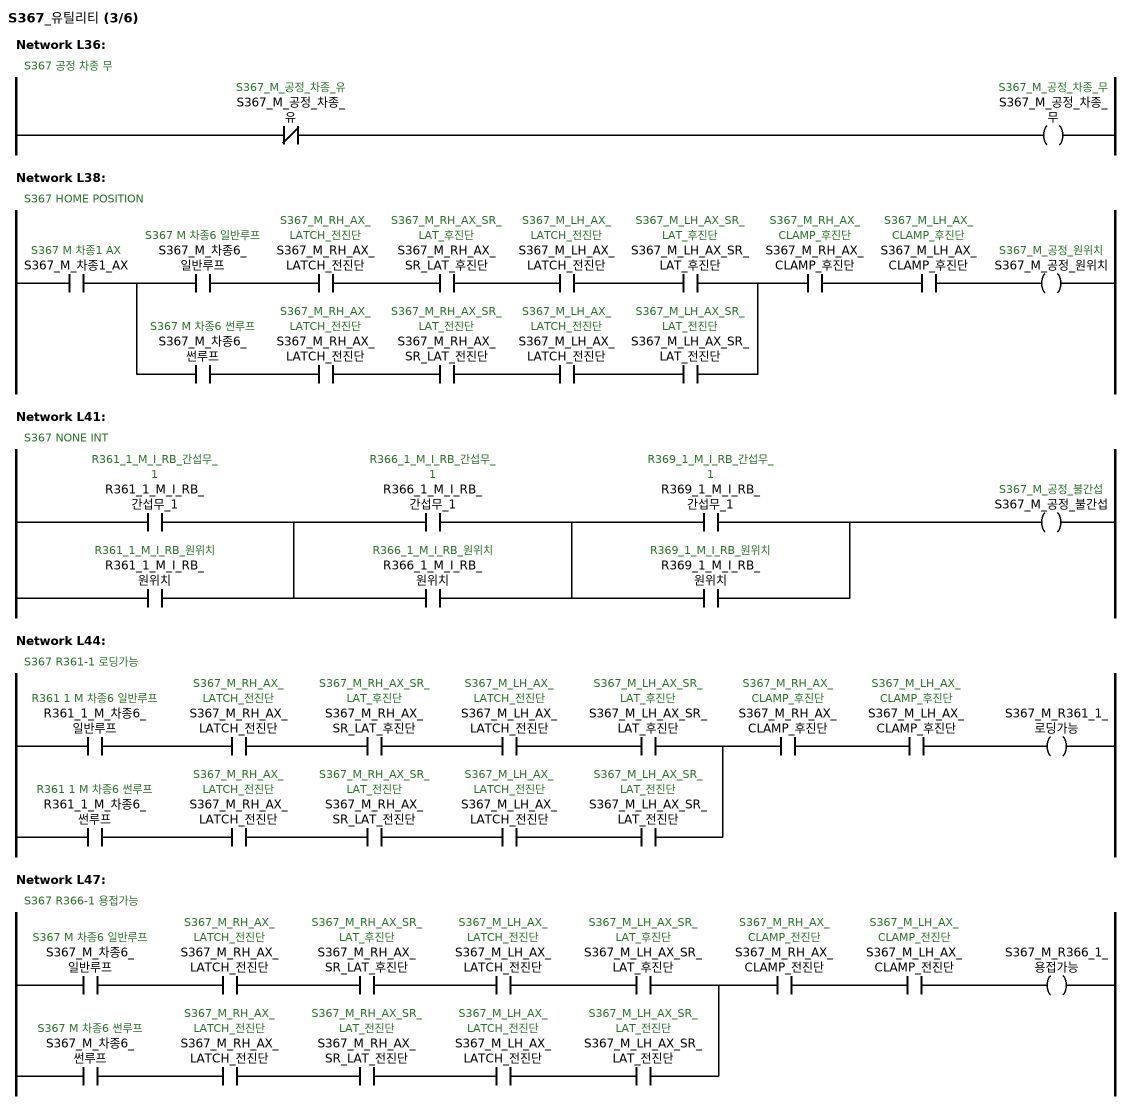
(* [picture p216: S367_유틸리티 rungs L36-L47] *)
(* S367 공정 차종 무 *)
(* Rung L36 *)
S367_M_공정_차종_무 := NOT S367_M_공정_차종_유;
(* S367 HOME POSITION *)
(* Rung L38 *)
S367_M_공정_원위치 := S367_M_차종1_AX AND ((S367_M_차종6_일반루프 AND S367_M_RH_AX_LATCH_전진단 AND S367_M_RH_AX_SR_LAT_후진단 AND S367_M_LH_AX_LATCH_전진단 AND S367_M_LH_AX_SR_LAT_후진단) OR (S367_M_차종6_썬루프 AND S367_M_RH_AX_LATCH_전진단 AND S367_M_RH_AX_SR_LAT_전진단 AND S367_M_LH_AX_LATCH_전진단 AND S367_M_LH_AX_SR_LAT_전진단)) AND S367_M_RH_AX_CLAMP_후진단 AND S367_M_LH_AX_CLAMP_후진단;
(* S367 NONE INT *)
(* Rung L41 *)
S367_M_공정_불간섭 := (R361_1_M_I_RB_간섭무_1 OR R361_1_M_I_RB_원위치) AND (R366_1_M_I_RB_간섭무_1 OR R366_1_M_I_RB_원위치) AND (R369_1_M_I_RB_간섭무_1 OR R369_1_M_I_RB_원위치);
(* S367 R361-1 로딩가능 *)
(* Rung L44 *)
S367_M_R361_1_로딩가능 := ((R361_1_M_차종6_일반루프 AND S367_M_RH_AX_LATCH_전진단 AND S367_M_RH_AX_SR_LAT_후진단 AND S367_M_LH_AX_LATCH_전진단 AND S367_M_LH_AX_SR_LAT_후진단) OR (R361_1_M_차종6_썬루프 AND S367_M_RH_AX_LATCH_전진단 AND S367_M_RH_AX_SR_LAT_전진단 AND S367_M_LH_AX_LATCH_전진단 AND S367_M_LH_AX_SR_LAT_전진단)) AND S367_M_RH_AX_CLAMP_후진단 AND S367_M_LH_AX_CLAMP_후진단;
(* S367 R366-1 용접가능 *)
(* Rung L47 *)
S367_M_R366_1_용접가능 := ((S367_M_차종6_일반루프 AND S367_M_RH_AX_LATCH_전진단 AND S367_M_RH_AX_SR_LAT_후진단 AND S367_M_LH_AX_LATCH_전진단 AND S367_M_LH_AX_SR_LAT_후진단) OR (S367_M_차종6_썬루프 AND S367_M_RH_AX_LATCH_전진단 AND S367_M_RH_AX_SR_LAT_전진단 AND S367_M_LH_AX_LATCH_전진단 AND S367_M_LH_AX_SR_LAT_전진단)) AND S367_M_RH_AX_CLAMP_전진단 AND S367_M_LH_AX_CLAMP_전진단;

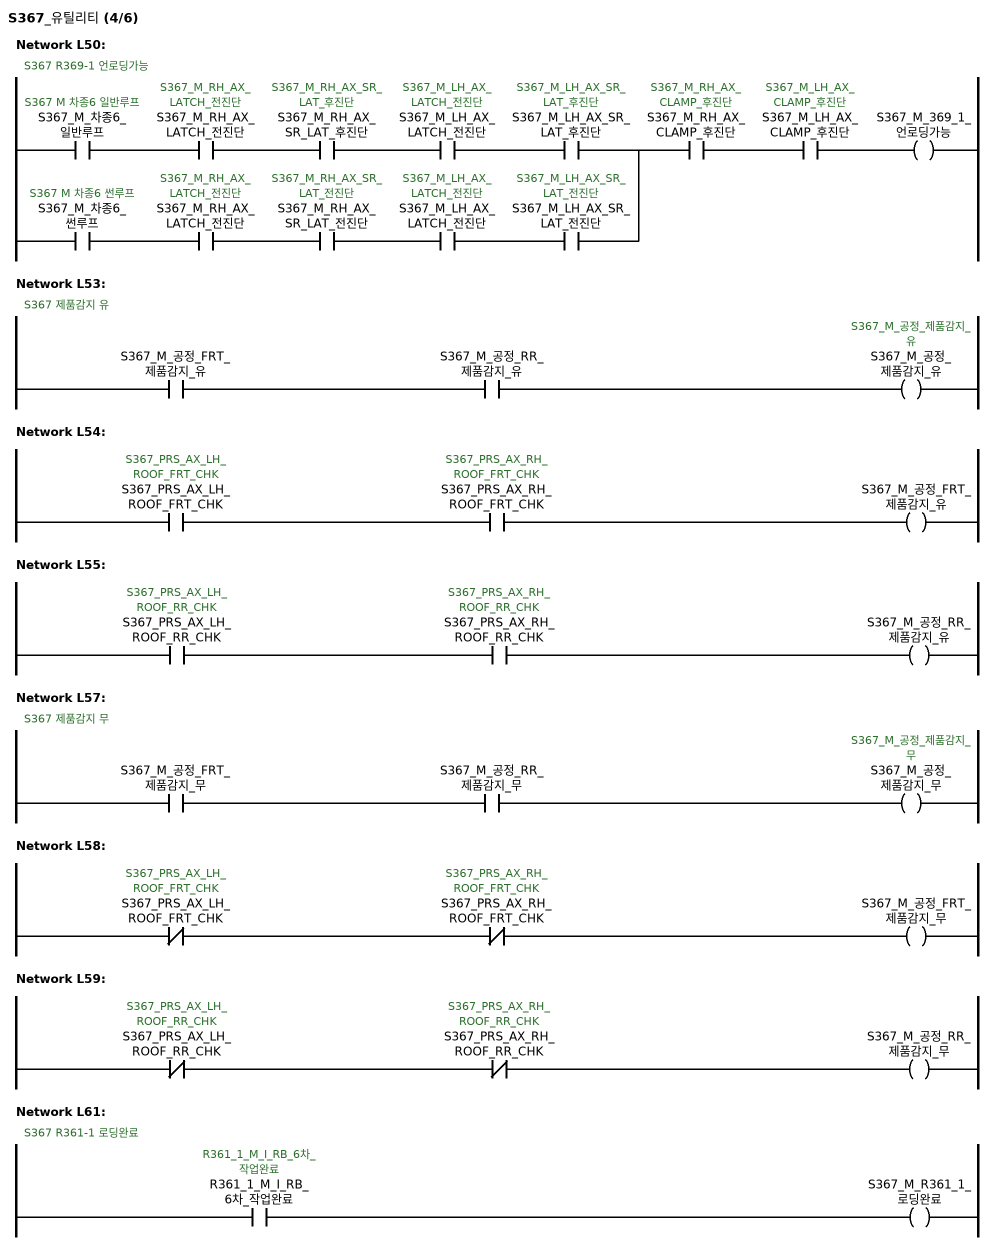
(* S367 R369-1 언로딩가능 *)
(* Rung L50 *)
S367_M_369_1_언로딩가능 := ((S367_M_차종6_일반루프 AND S367_M_RH_AX_LATCH_전진단 AND S367_M_RH_AX_SR_LAT_후진단 AND S367_M_LH_AX_LATCH_전진단 AND S367_M_LH_AX_SR_LAT_후진단) OR (S367_M_차종6_썬루프 AND S367_M_RH_AX_LATCH_전진단 AND S367_M_RH_AX_SR_LAT_전진단 AND S367_M_LH_AX_LATCH_전진단 AND S367_M_LH_AX_SR_LAT_전진단)) AND S367_M_RH_AX_CLAMP_후진단 AND S367_M_LH_AX_CLAMP_후진단;
(* S367 제품감지 유 *)
(* Rung L53 *)
S367_M_공정_제품감지_유 := S367_M_공정_FRT_제품감지_유 AND S367_M_공정_RR_제품감지_유;
(* Rung L54 *)
S367_M_공정_FRT_제품감지_유 := S367_PRS_AX_LH_ROOF_FRT_CHK AND S367_PRS_AX_RH_ROOF_FRT_CHK;
(* Rung L55 *)
S367_M_공정_RR_제품감지_유 := S367_PRS_AX_LH_ROOF_RR_CHK AND S367_PRS_AX_RH_ROOF_RR_CHK;
(* S367 제품감지 무 *)
(* Rung L57 *)
S367_M_공정_제품감지_무 := S367_M_공정_FRT_제품감지_무 AND S367_M_공정_RR_제품감지_무;
(* Rung L58 *)
S367_M_공정_FRT_제품감지_무 := NOT S367_PRS_AX_LH_ROOF_FRT_CHK AND NOT S367_PRS_AX_RH_ROOF_FRT_CHK;
(* Rung L59 *)
S367_M_공정_RR_제품감지_무 := NOT S367_PRS_AX_LH_ROOF_RR_CHK AND NOT S367_PRS_AX_RH_ROOF_RR_CHK;
(* S367 R361-1 로딩완료 *)
(* Rung L61 *)
S367_M_R361_1_로딩완료 := R361_1_M_I_RB_6차_작업완료;

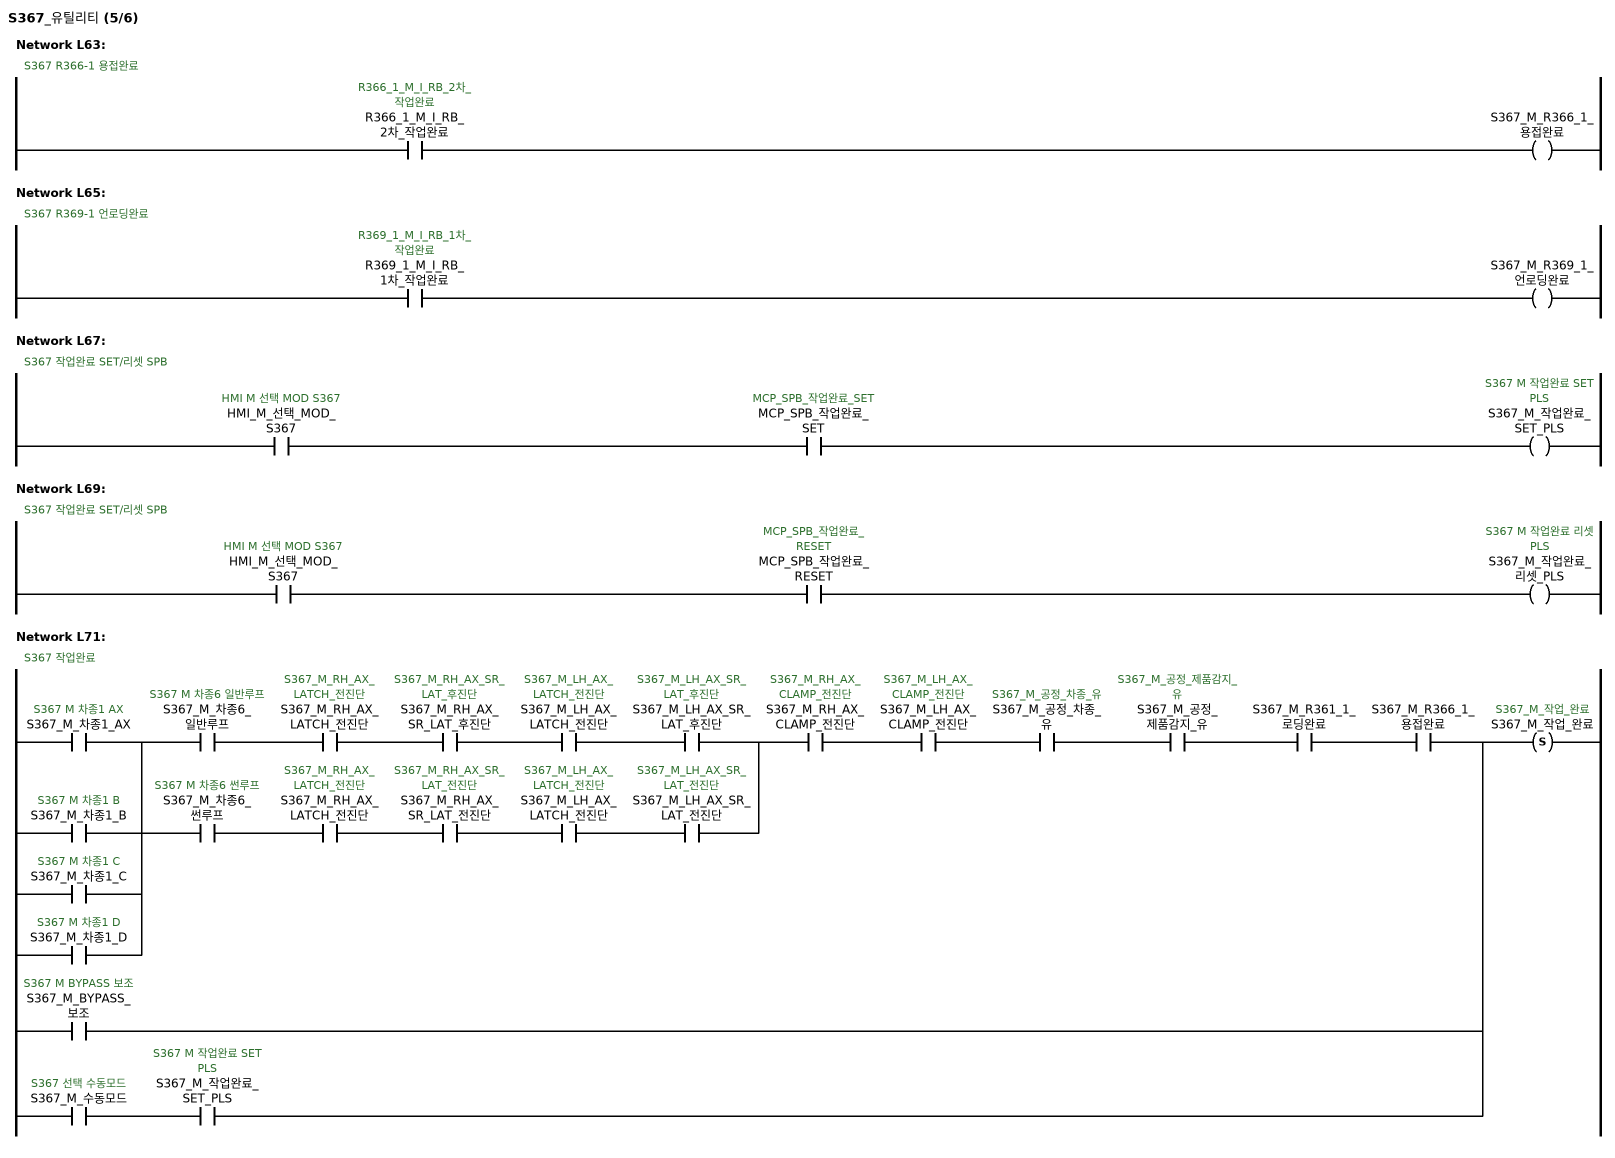
(* S367 R366-1 용접완료 *)
(* Rung L63 *)
S367_M_R366_1_용접완료 := R366_1_M_I_RB_2차_작업완료;
(* S367 R369-1 언로딩완료 *)
(* Rung L65 *)
S367_M_R369_1_언로딩완료 := R369_1_M_I_RB_1차_작업완료;
(* S367 작업완료 SET/리셋 SPB *)
(* Rung L67 *)
S367_M_작업완료_SET_PLS := HMI_M_선택_MOD_S367 AND MCP_SPB_작업완료_SET;
(* S367 작업완료 SET/리셋 SPB *)
(* Rung L69 *)
S367_M_작업완료_리셋_PLS := HMI_M_선택_MOD_S367 AND MCP_SPB_작업완료_RESET;
(* S367 작업완료 *)
(* Rung L71 *)
IF ((S367_M_차종1_AX OR S367_M_차종1_B OR S367_M_차종1_C OR S367_M_차종1_D) AND ((S367_M_차종6_일반루프 AND S367_M_RH_AX_LATCH_전진단 AND S367_M_RH_AX_SR_LAT_후진단 AND S367_M_LH_AX_LATCH_전진단 AND S367_M_LH_AX_SR_LAT_후진단) OR (S367_M_차종6_썬루프 AND S367_M_RH_AX_LATCH_전진단 AND S367_M_RH_AX_SR_LAT_전진단 AND S367_M_LH_AX_LATCH_전진단 AND S367_M_LH_AX_SR_LAT_전진단)) AND S367_M_RH_AX_CLAMP_전진단 AND S367_M_LH_AX_CLAMP_전진단 AND S367_M_공정_차종_유 AND S367_M_공정_제품감지_유 AND S367_M_R361_1_로딩완료 AND S367_M_R366_1_용접완료) OR S367_M_BYPASS_보조 OR (S367_M_수동모드 AND S367_M_작업완료_SET_PLS) THEN
    S367_M_작업_완료 := TRUE;
END_IF;

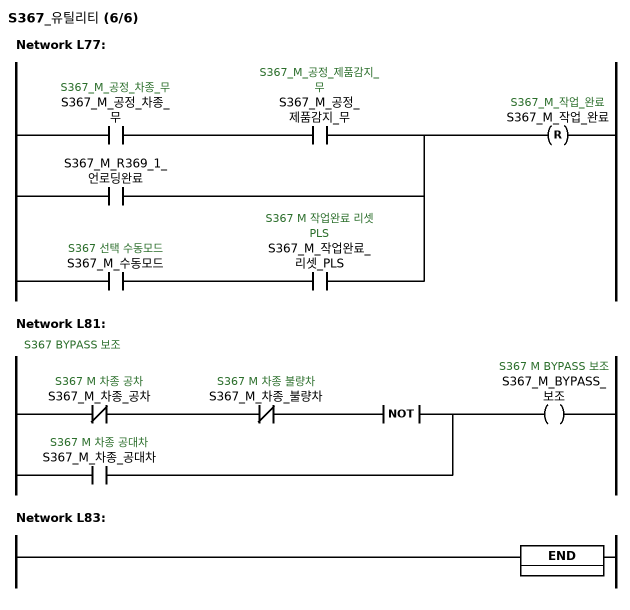
(* Rung L77 *)
IF (S367_M_공정_차종_무 AND S367_M_공정_제품감지_무) OR S367_M_R369_1_언로딩완료 OR (S367_M_수동모드 AND S367_M_작업완료_리셋_PLS) THEN
    S367_M_작업_완료 := FALSE;
END_IF;
(* S367 BYPASS 보조 *)
(* Rung L81 *)
S367_M_BYPASS_보조 := NOT (NOT S367_M_차종_공차 AND NOT S367_M_차종_불량차) OR S367_M_차종_공대차;
(* Rung L83 *)
END();
END_PROGRAM

PROGRAM S367_동작 (* task: 스캔 프로그램 *)
VAR_EXTERNAL RETAIN
    ALWAYS_ON : BOOL; (* AT %MW3.1 *) (* 항시 ON *)
    R361_1_M_차종1_AX : BOOL; (* AT %MW10001.0 *) (* R361 1 M 차종1 AX *)
    R361_1_M_차종6_썬루프 : BOOL; (* AT %MW10003.4 *) (* R361 1 M 차종6 썬루프 *)
    R361_1_M_차종_유 : BOOL; (* AT %MW1502.0 *)
    S367_HOME : BOOL; (* AT %MW3548.0 *) (* S367_HOME *)
    S367_M_LH_AX_CLAMP_전진_LS_이상 : BOOL; (* AT %MW3602.5 *) (* S367_M_LH_AX_CLAMP_전진_LS_이상 *)
    S367_M_LH_AX_CLAMP_전진_보조 : BOOL; (* AT %MW3602.1 *) (* S367_M_LH_AX_CLAMP_전진_보조 *)
    S367_M_LH_AX_CLAMP_전진단 : BOOL; (* AT %MW3602.3 *) (* S367_M_LH_AX_CLAMP_전진단 *)
    S367_M_LH_AX_CLAMP_조건 : BOOL; (* AT %MW3602.0 *) (* S367_M_LH_AX_CLAMP_조건 *)
    S367_M_LH_AX_CLAMP_후진_LS_이상 : BOOL; (* AT %MW3602.6 *) (* S367_M_LH_AX_CLAMP_후진_LS_이상 *)
    S367_M_LH_AX_CLAMP_후진_보조 : BOOL; (* AT %MW3602.2 *) (* S367_M_LH_AX_CLAMP_후진_보조 *)
    S367_M_LH_AX_CLAMP_후진단 : BOOL; (* AT %MW3602.4 *) (* S367_M_LH_AX_CLAMP_후진단 *)
    S367_M_LH_AX_LATCH_전진_LS_이상 : BOOL; (* AT %MW3600.5 *) (* S367_M_LH_AX_LATCH_전진_LS_이상 *)
    S367_M_LH_AX_LATCH_전진_보조 : BOOL; (* AT %MW3600.1 *) (* S367_M_LH_AX_LATCH_전진_보조 *)
    S367_M_LH_AX_LATCH_전진단 : BOOL; (* AT %MW3600.3 *) (* S367_M_LH_AX_LATCH_전진단 *)
    S367_M_LH_AX_LATCH_조건 : BOOL; (* AT %MW3600.0 *) (* S367_M_LH_AX_LATCH_조건 *)
    S367_M_LH_AX_LATCH_후진_LS_이상 : BOOL; (* AT %MW3600.6 *) (* S367_M_LH_AX_LATCH_후진_LS_이상 *)
    S367_M_LH_AX_LATCH_후진_보조 : BOOL; (* AT %MW3600.2 *) (* S367_M_LH_AX_LATCH_후진_보조 *)
    S367_M_LH_AX_LATCH_후진단 : BOOL; (* AT %MW3600.4 *) (* S367_M_LH_AX_LATCH_후진단 *)
    S367_M_LH_AX_SR_LAT_전진_LS_이상 : BOOL; (* AT %MW3601.5 *) (* S367_M_LH_AX_SR_LAT_전진_LS_이상 *)
    S367_M_LH_AX_SR_LAT_전진_보조 : BOOL; (* AT %MW3601.1 *) (* S367_M_LH_AX_SR_LAT_전진_보조 *)
    S367_M_LH_AX_SR_LAT_전진단 : BOOL; (* AT %MW3601.3 *) (* S367_M_LH_AX_SR_LAT_전진단 *)
    S367_M_LH_AX_SR_LAT_조건 : BOOL; (* AT %MW3601.0 *) (* S367_M_LH_AX_SR_LAT_조건 *)
    S367_M_LH_AX_SR_LAT_후진_LS_이상 : BOOL; (* AT %MW3601.6 *) (* S367_M_LH_AX_SR_LAT_후진_LS_이상 *)
    S367_M_LH_AX_SR_LAT_후진_보조 : BOOL; (* AT %MW3601.2 *) (* S367_M_LH_AX_SR_LAT_후진_보조 *)
    S367_M_LH_AX_SR_LAT_후진단 : BOOL; (* AT %MW3601.4 *) (* S367_M_LH_AX_SR_LAT_후진단 *)
    S367_M_R361_1_로딩완료 : BOOL; (* AT %MW3501.1 *)
    S367_M_RH_AX_CLAMP_전진_LS_이상 : BOOL; (* AT %MW3610.5 *) (* S367_M_RH_AX_CLAMP_전진_LS_이상 *)
    S367_M_RH_AX_CLAMP_전진_보조 : BOOL; (* AT %MW3610.1 *) (* S367_M_RH_AX_CLAMP_전진_보조 *)
    S367_M_RH_AX_CLAMP_전진단 : BOOL; (* AT %MW3610.3 *) (* S367_M_RH_AX_CLAMP_전진단 *)
    S367_M_RH_AX_CLAMP_조건 : BOOL; (* AT %MW3610.0 *) (* S367_M_RH_AX_CLAMP_조건 *)
    S367_M_RH_AX_CLAMP_후진_LS_이상 : BOOL; (* AT %MW3610.6 *) (* S367_M_RH_AX_CLAMP_후진_LS_이상 *)
    S367_M_RH_AX_CLAMP_후진_보조 : BOOL; (* AT %MW3610.2 *) (* S367_M_RH_AX_CLAMP_후진_보조 *)
    S367_M_RH_AX_CLAMP_후진단 : BOOL; (* AT %MW3610.4 *) (* S367_M_RH_AX_CLAMP_후진단 *)
    S367_M_RH_AX_LATCH_전진_LS_이상 : BOOL; (* AT %MW3608.5 *) (* S367_M_RH_AX_LATCH_전진_LS_이상 *)
    S367_M_RH_AX_LATCH_전진_보조 : BOOL; (* AT %MW3608.1 *) (* S367_M_RH_AX_LATCH_전진_보조 *)
    S367_M_RH_AX_LATCH_전진단 : BOOL; (* AT %MW3608.3 *) (* S367_M_RH_AX_LATCH_전진단 *)
    S367_M_RH_AX_LATCH_조건 : BOOL; (* AT %MW3608.0 *) (* S367_M_RH_AX_LATCH_조건 *)
    S367_M_RH_AX_LATCH_후진_LS_이상 : BOOL; (* AT %MW3608.6 *) (* S367_M_RH_AX_LATCH_후진_LS_이상 *)
    S367_M_RH_AX_LATCH_후진_보조 : BOOL; (* AT %MW3608.2 *) (* S367_M_RH_AX_LATCH_후진_보조 *)
    S367_M_RH_AX_LATCH_후진단 : BOOL; (* AT %MW3608.4 *) (* S367_M_RH_AX_LATCH_후진단 *)
    S367_M_RH_AX_SR_LAT_전진_LS_이상 : BOOL; (* AT %MW3609.5 *) (* S367_M_RH_AX_SR_LAT_전진_LS_이상 *)
    S367_M_RH_AX_SR_LAT_전진_보조 : BOOL; (* AT %MW3609.1 *) (* S367_M_RH_AX_SR_LAT_전진_보조 *)
    S367_M_RH_AX_SR_LAT_전진단 : BOOL; (* AT %MW3609.3 *) (* S367_M_RH_AX_SR_LAT_전진단 *)
    S367_M_RH_AX_SR_LAT_조건 : BOOL; (* AT %MW3609.0 *) (* S367_M_RH_AX_SR_LAT_조건 *)
    S367_M_RH_AX_SR_LAT_후진_LS_이상 : BOOL; (* AT %MW3609.6 *) (* S367_M_RH_AX_SR_LAT_후진_LS_이상 *)
    S367_M_RH_AX_SR_LAT_후진_보조 : BOOL; (* AT %MW3609.2 *) (* S367_M_RH_AX_SR_LAT_후진_보조 *)
    S367_M_RH_AX_SR_LAT_후진단 : BOOL; (* AT %MW3609.4 *) (* S367_M_RH_AX_SR_LAT_후진단 *)
    S367_M_공정_불간섭 : BOOL; (* AT %MW3504.1 *) (* S367_M_공정_불간섭 *)
    S367_M_공정_제품감지_무 : BOOL; (* AT %MW3501.6 *) (* S367_M_공정_제품감지_무 *)
    S367_M_공정_제품감지_유 : BOOL; (* AT %MW3501.5 *) (* S367_M_공정_제품감지_유 *)
    S367_M_공정_차종_무 : BOOL; (* AT %MW3502.1 *) (* S367_M_공정_차종_무 *)
    S367_M_공정_차종_유 : BOOL; (* AT %MW3502.0 *) (* S367_M_공정_차종_유 *)
    S367_M_동작_선택_1 : BOOL; (* AT %MW3540.0 *) (* S367_M_동작_선택_1 *)
    S367_M_동작_선택_10 : BOOL; (* AT %MW3540.9 *) (* S367_M_동작_선택_10 *)
    S367_M_동작_선택_11 : BOOL; (* AT %MW3540.10 *) (* S367_M_동작_선택_11 *)
    S367_M_동작_선택_2 : BOOL; (* AT %MW3540.1 *) (* S367_M_동작_선택_2 *)
    S367_M_동작_선택_3 : BOOL; (* AT %MW3540.2 *) (* S367_M_동작_선택_3 *)
    S367_M_동작_선택_9 : BOOL; (* AT %MW3540.8 *) (* S367_M_동작_선택_9 *)
    S367_M_수동모드 : BOOL; (* AT %MW3500.3 *) (* S367 선택 수동모드 *)
    S367_M_운전준비_ON : BOOL; (* AT %MW3500.0 *) (* S367 운전준비 ON *)
    S367_M_자동_운전중 : BOOL; (* AT %MW3500.4 *) (* S367 자동운전중 *)
    S367_M_작업_완료 : BOOL; (* AT %MW3501.0 *) (* S367_M_작업_완료 *)
    S367_M_차종1_AX : BOOL; (* AT %MW10181.0 *) (* S367 M 차종1 AX *)
    S367_전진_ON : BOOL; (* AT %MW3548.1 *) (* S367_전진_ON *)
    S367_후진_ON : BOOL; (* AT %MW3548.2 *) (* S367_후진_ON *)
    전체_M_이상_리셋 : BOOL; (* AT %MW308.2 *) (* ALL공정 PB 이상리셋 *)
END_VAR
VAR_EXTERNAL
    EGIS_CWS : BOOL;
    S367_M_LH_AX_CLAMP_전진_LAMP : WORD; (* AT %MW13104 *) (* S367_M_LH_AX_CLAMP_전진_LAMP *)
    S367_M_LH_AX_CLAMP_후진_LAMP : WORD; (* AT %MW13105 *) (* S367_M_LH_AX_CLAMP_후진_LAMP *)
    S367_M_LH_AX_LATCH_전진_LAMP : WORD; (* AT %MW13100 *) (* S367_M_LH_AX_LATCH_전진_LAMP *)
    S367_M_LH_AX_LATCH_후진_LAMP : WORD; (* AT %MW13101 *) (* S367_M_LH_AX_LATCH_후진_LAMP *)
    S367_M_LH_AX_SR_LAT_전진_LAMP : WORD; (* AT %MW13102 *) (* S367_M_LH_AX_SR_LAT_전진_LAMP *)
    S367_M_LH_AX_SR_LAT_후진_LAMP : WORD; (* AT %MW13103 *) (* S367_M_LH_AX_SR_LAT_후진_LAMP *)
    S367_M_RH_AX_CLAMP_전진_LAMP : WORD; (* AT %MW13120 *) (* S367_M_RH_AX_CLAMP_전진_LAMP *)
    S367_M_RH_AX_CLAMP_후진_LAMP : WORD; (* AT %MW13121 *) (* S367_M_RH_AX_CLAMP_후진_LAMP *)
    S367_M_RH_AX_LATCH_전진_LAMP : WORD; (* AT %MW13116 *) (* S367_M_RH_AX_LATCH_전진_LAMP *)
    S367_M_RH_AX_LATCH_후진_LAMP : WORD; (* AT %MW13117 *) (* S367_M_RH_AX_LATCH_후진_LAMP *)
    S367_M_RH_AX_SR_LAT_전진_LAMP : WORD; (* AT %MW13118 *) (* S367_M_RH_AX_SR_LAT_전진_LAMP *)
    S367_M_RH_AX_SR_LAT_후진_LAMP : WORD; (* AT %MW13119 *) (* S367_M_RH_AX_SR_LAT_후진_LAMP *)
    S367_RS_AX_LH_CLAMP_전진 : BOOL; (* AT %MW86210.8 *) (* S367_RS_AX_LH_CLAMP_전진 *)
    S367_RS_AX_LH_CLAMP_후진1 : BOOL; (* AT %MW86210.9 *) (* S367_RS_AX_LH_CLAMP_후진1 *)
    S367_RS_AX_LH_CLAMP_후진2 : BOOL; (* AT %MW86210.10 *) (* S367_RS_AX_LH_CLAMP_후진2 *)
    S367_RS_AX_LH_CLAMP_후진3 : BOOL; (* AT %MW86210.11 *) (* S367_RS_AX_LH_CLAMP_후진3 *)
    S367_RS_AX_LH_CLAMP_후진4 : BOOL; (* AT %MW86210.12 *) (* S367_RS_AX_LH_CLAMP_후진4 *)
    S367_RS_AX_LH_CLAMP_후진5 : BOOL; (* AT %MW86210.13 *) (* S367_RS_AX_LH_CLAMP_후진5 *)
    S367_RS_AX_LH_GR_LATCH_전진 : BOOL; (* AT %MW86210.0 *) (* S367_RS_AX_LH_GR_LATCH_전진 *)
    S367_RS_AX_LH_GR_LATCH_후진1 : BOOL; (* AT %MW86210.1 *) (* S367_RS_AX_LH_GR_LATCH_후진1 *)
    S367_RS_AX_LH_GR_LATCH_후진2 : BOOL; (* AT %MW86210.2 *) (* S367_RS_AX_LH_GR_LATCH_후진2 *)
    S367_RS_AX_LH_GR_LATCH_후진3 : BOOL; (* AT %MW86210.3 *) (* S367_RS_AX_LH_GR_LATCH_후진3 *)
    S367_RS_AX_LH_GR_LATCH_후진4 : BOOL; (* AT %MW86210.4 *) (* S367_RS_AX_LH_GR_LATCH_후진4 *)
    S367_RS_AX_LH_GR_LATCH_후진5 : BOOL; (* AT %MW86210.5 *) (* S367_RS_AX_LH_GR_LATCH_후진5 *)
    S367_RS_AX_LH_SR_LATCH_전진 : BOOL; (* AT %MW86211.0 *) (* S367_RS_AX_LH_SR_LATCH_전진 *)
    S367_RS_AX_LH_SR_LATCH_후진1 : BOOL; (* AT %MW86211.1 *) (* S367_RS_AX_LH_SR_LATCH_후진1 *)
    S367_RS_AX_LH_SR_LATCH_후진2 : BOOL; (* AT %MW86211.2 *) (* S367_RS_AX_LH_SR_LATCH_후진2 *)
    S367_RS_AX_LH_SR_LATCH_후진3 : BOOL; (* AT %MW86211.3 *) (* S367_RS_AX_LH_SR_LATCH_후진3 *)
    S367_RS_AX_RH_CLAMP_전진 : BOOL; (* AT %MW86200.8 *) (* S367_RS_AX_RH_CLAMP_전진 *)
    S367_RS_AX_RH_CLAMP_후진1 : BOOL; (* AT %MW86200.9 *) (* S367_RS_AX_RH_CLAMP_후진1 *)
    S367_RS_AX_RH_CLAMP_후진2 : BOOL; (* AT %MW86200.10 *) (* S367_RS_AX_RH_CLAMP_후진2 *)
    S367_RS_AX_RH_CLAMP_후진3 : BOOL; (* AT %MW86200.11 *) (* S367_RS_AX_RH_CLAMP_후진3 *)
    S367_RS_AX_RH_CLAMP_후진4 : BOOL; (* AT %MW86200.12 *) (* S367_RS_AX_RH_CLAMP_후진4 *)
    S367_RS_AX_RH_CLAMP_후진5 : BOOL; (* AT %MW86200.13 *) (* S367_RS_AX_RH_CLAMP_후진5 *)
    S367_RS_AX_RH_GR_LATCH_전진 : BOOL; (* AT %MW86200.0 *) (* S367_RS_AX_RH_GR_LATCH_전진 *)
    S367_RS_AX_RH_GR_LATCH_후진1 : BOOL; (* AT %MW86200.1 *) (* S367_RS_AX_RH_GR_LATCH_후진1 *)
    S367_RS_AX_RH_GR_LATCH_후진2 : BOOL; (* AT %MW86200.2 *) (* S367_RS_AX_RH_GR_LATCH_후진2 *)
    S367_RS_AX_RH_GR_LATCH_후진3 : BOOL; (* AT %MW86200.3 *) (* S367_RS_AX_RH_GR_LATCH_후진3 *)
    S367_RS_AX_RH_GR_LATCH_후진4 : BOOL; (* AT %MW86200.4 *) (* S367_RS_AX_RH_GR_LATCH_후진4 *)
    S367_RS_AX_RH_GR_LATCH_후진5 : BOOL; (* AT %MW86200.5 *) (* S367_RS_AX_RH_GR_LATCH_후진5 *)
    S367_RS_AX_RH_SR_LATCH_전진 : BOOL; (* AT %MW86201.0 *) (* S367_RS_AX_RH_SR_LATCH_전진 *)
    S367_RS_AX_RH_SR_LATCH_후진1 : BOOL; (* AT %MW86201.1 *) (* S367_RS_AX_RH_SR_LATCH_후진1 *)
    S367_RS_AX_RH_SR_LATCH_후진2 : BOOL; (* AT %MW86201.2 *) (* S367_RS_AX_RH_SR_LATCH_후진2 *)
    S367_RS_AX_RH_SR_LATCH_후진3 : BOOL; (* AT %MW86201.3 *) (* S367_RS_AX_RH_SR_LATCH_후진3 *)
    S367_SOL_AX_LH_CLAMP_전진 : BOOL; (* AT %MW96213.6 *) (* S367_SOL_AX_LH_CLAMP_전진 *)
    S367_SOL_AX_LH_CLAMP_후진 : BOOL; (* AT %MW96213.7 *) (* S367_SOL_AX_LH_CLAMP_후진 *)
    S367_SOL_AX_LH_GR_LATCH_전진 : BOOL; (* AT %MW96213.2 *) (* S367_SOL_AX_LH_GR_LATCH_전진 *)
    S367_SOL_AX_LH_GR_LATCH_후진 : BOOL; (* AT %MW96213.3 *) (* S367_SOL_AX_LH_GR_LATCH_후진 *)
    S367_SOL_AX_LH_SR_LATCH_전진 : BOOL; (* AT %MW96213.10 *) (* S367_SOL_AX_LH_SR_LATCH_전진 *)
    S367_SOL_AX_LH_SR_LATCH_후진 : BOOL; (* AT %MW96213.11 *) (* S367_SOL_AX_LH_SR_LATCH_후진 *)
    S367_SOL_AX_RH_CLAMP_전진 : BOOL; (* AT %MW96213.4 *) (* S367_SOL_AX_RH_CLAMP_전진 *)
    S367_SOL_AX_RH_CLAMP_후진 : BOOL; (* AT %MW96213.5 *) (* S367_SOL_AX_RH_CLAMP_후진 *)
    S367_SOL_AX_RH_GR_LATCH_전진 : BOOL; (* AT %MW96213.0 *) (* S367_SOL_AX_RH_GR_LATCH_전진 *)
    S367_SOL_AX_RH_GR_LATCH_후진 : BOOL; (* AT %MW96213.1 *) (* S367_SOL_AX_RH_GR_LATCH_후진 *)
    S367_SOL_AX_RH_SR_LATCH_전진 : BOOL; (* AT %MW96213.8 *) (* S367_SOL_AX_RH_SR_LATCH_전진 *)
    S367_SOL_AX_RH_SR_LATCH_후진 : BOOL; (* AT %MW96213.9 *) (* S367_SOL_AX_RH_SR_LATCH_후진 *)
END_VAR
VAR
    S367_LH_AX_CLAMP : ACT_6_CYL;
    S367_LH_AX_LATCH : ACT_6_CYL;
    S367_LH_AX_SR_LAT : ACT_6_CYL;
    S367_RH_AX_CLAMP : ACT_6_CYL;
    S367_RH_AX_LATCH : ACT_6_CYL;
    S368_RH_AX_SR_LAT : ACT_6_CYL;
END_VAR

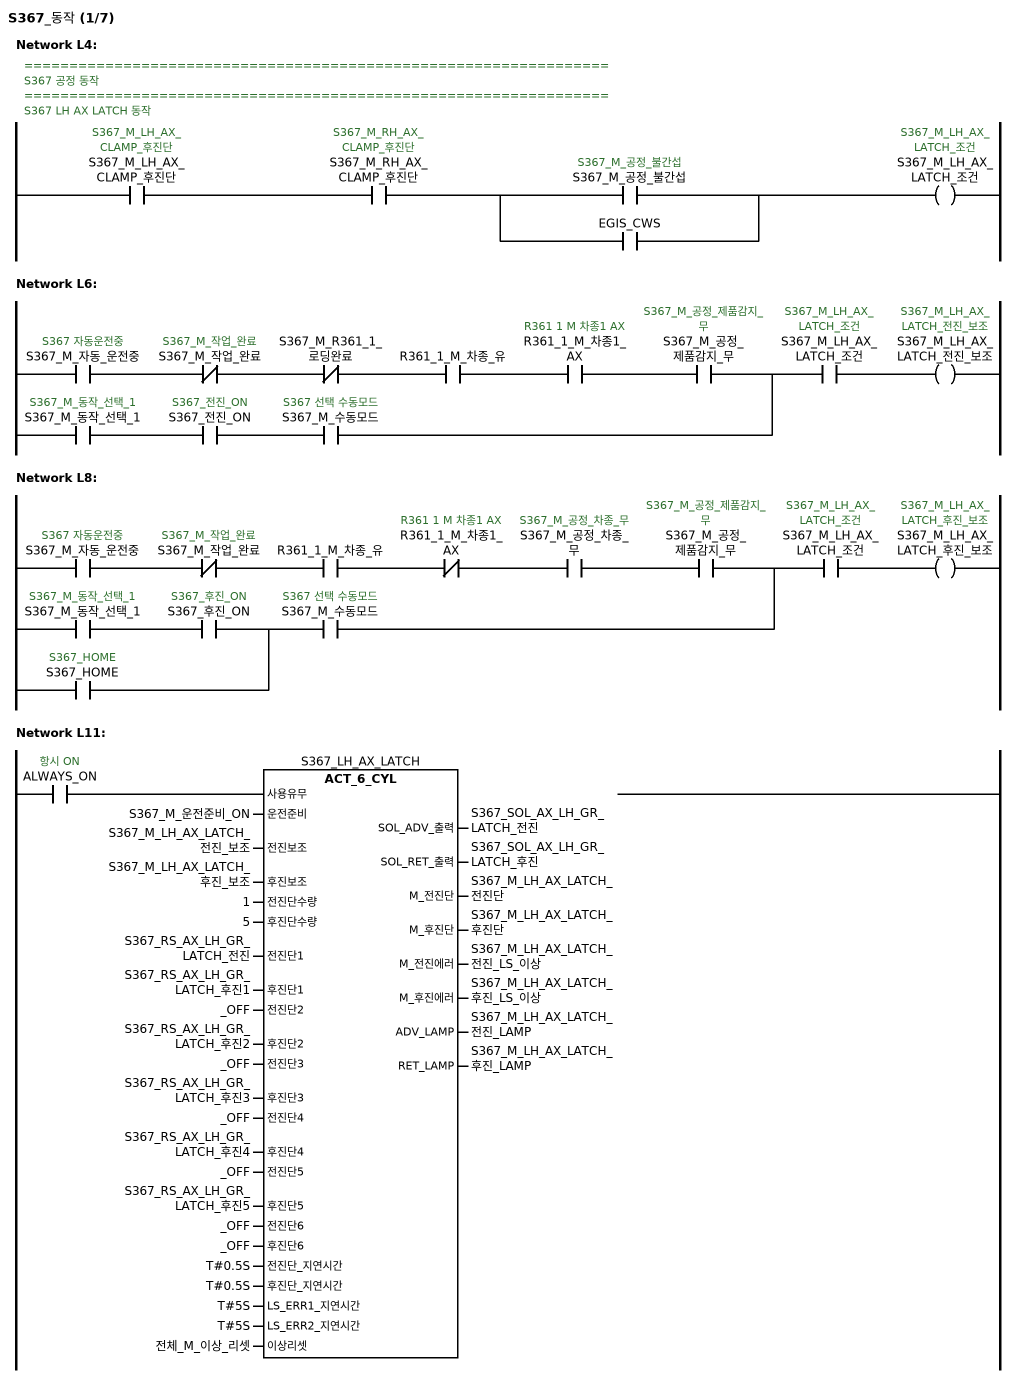
(* ================================================================= *)
(* S367 공정 동작 *)
(* ================================================================= *)
(* S367 LH AX LATCH 동작 *)
(* Rung L4 *)
S367_M_LH_AX_LATCH_조건 := S367_M_LH_AX_CLAMP_후진단 AND S367_M_RH_AX_CLAMP_후진단 AND (S367_M_공정_불간섭 OR EGIS_CWS);
(* Rung L6 *)
S367_M_LH_AX_LATCH_전진_보조 := ((S367_M_자동_운전중 AND NOT S367_M_작업_완료 AND NOT S367_M_R361_1_로딩완료 AND R361_1_M_차종_유 AND R361_1_M_차종1_AX AND S367_M_공정_제품감지_무) OR (S367_M_동작_선택_1 AND S367_전진_ON AND S367_M_수동모드)) AND S367_M_LH_AX_LATCH_조건;
(* Rung L8 *)
S367_M_LH_AX_LATCH_후진_보조 := ((S367_M_자동_운전중 AND NOT S367_M_작업_완료 AND R361_1_M_차종_유 AND NOT R361_1_M_차종1_AX AND S367_M_공정_차종_무 AND S367_M_공정_제품감지_무) OR (((S367_M_동작_선택_1 AND S367_후진_ON) OR S367_HOME) AND S367_M_수동모드)) AND S367_M_LH_AX_LATCH_조건;
(* Rung L11 *)
S367_LH_AX_LATCH(사용유무 := ALWAYS_ON, 운전준비 := S367_M_운전준비_ON, 전진보조 := S367_M_LH_AX_LATCH_전진_보조, 후진보조 := S367_M_LH_AX_LATCH_후진_보조, 전진단수량 := 1, 후진단수량 := 5, 전진단1 := S367_RS_AX_LH_GR_LATCH_전진, 후진단1 := S367_RS_AX_LH_GR_LATCH_후진1, 전진단2 := _OFF, 후진단2 := S367_RS_AX_LH_GR_LATCH_후진2, 전진단3 := _OFF, 후진단3 := S367_RS_AX_LH_GR_LATCH_후진3, 전진단4 := _OFF, 후진단4 := S367_RS_AX_LH_GR_LATCH_후진4, 전진단5 := _OFF, 후진단5 := S367_RS_AX_LH_GR_LATCH_후진5, 전진단6 := _OFF, 후진단6 := _OFF, 전진단_지연시간 := T#0.5S, 후진단_지연시간 := T#0.5S, LS_ERR1_지연시간 := T#5S, LS_ERR2_지연시간 := T#5S, 이상리셋 := 전체_M_이상_리셋, SOL_ADV_출력 => S367_SOL_AX_LH_GR_LATCH_전진, SOL_RET_출력 => S367_SOL_AX_LH_GR_LATCH_후진, M_전진단 => S367_M_LH_AX_LATCH_전진단, M_후진단 => S367_M_LH_AX_LATCH_후진단, M_전진에러 => S367_M_LH_AX_LATCH_전진_LS_이상, M_후진에러 => S367_M_LH_AX_LATCH_후진_LS_이상, ADV_LAMP => S367_M_LH_AX_LATCH_전진_LAMP, RET_LAMP => S367_M_LH_AX_LATCH_후진_LAMP);

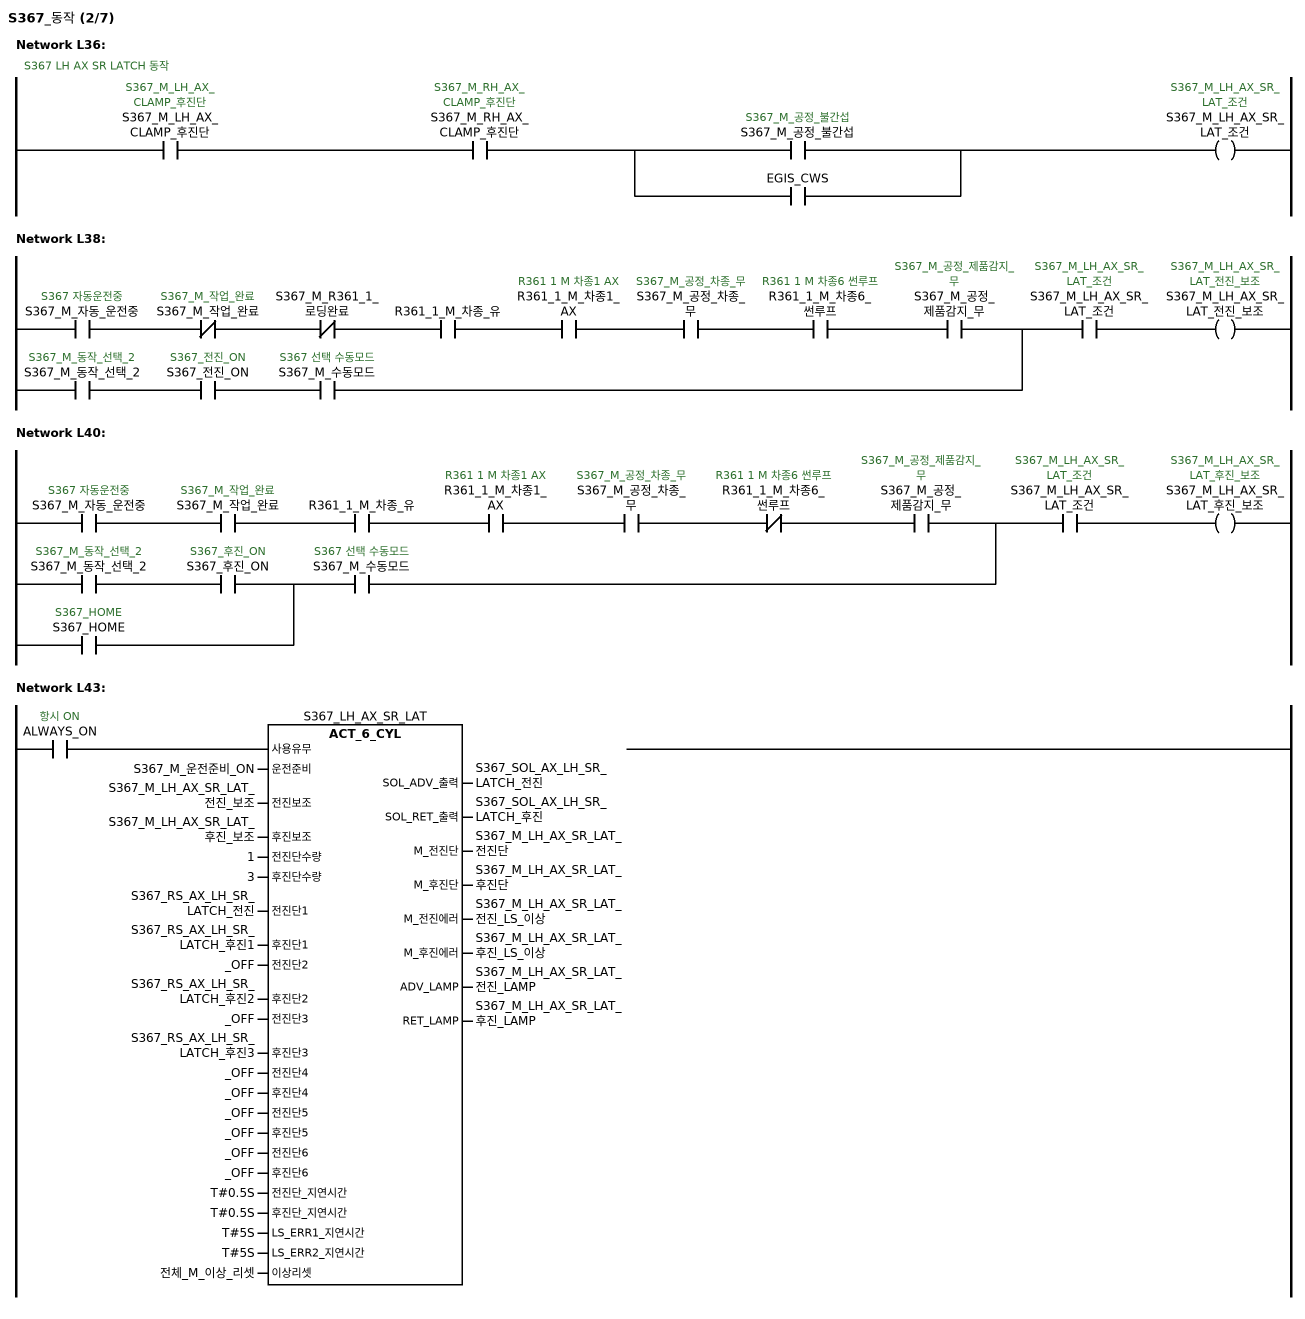
(* S367 LH AX SR LATCH 동작 *)
(* Rung L36 *)
S367_M_LH_AX_SR_LAT_조건 := S367_M_LH_AX_CLAMP_후진단 AND S367_M_RH_AX_CLAMP_후진단 AND (S367_M_공정_불간섭 OR EGIS_CWS);
(* Rung L38 *)
S367_M_LH_AX_SR_LAT_전진_보조 := ((S367_M_자동_운전중 AND NOT S367_M_작업_완료 AND NOT S367_M_R361_1_로딩완료 AND R361_1_M_차종_유 AND R361_1_M_차종1_AX AND S367_M_공정_차종_무 AND R361_1_M_차종6_썬루프 AND S367_M_공정_제품감지_무) OR (S367_M_동작_선택_2 AND S367_전진_ON AND S367_M_수동모드)) AND S367_M_LH_AX_SR_LAT_조건;
(* Rung L40 *)
S367_M_LH_AX_SR_LAT_후진_보조 := ((S367_M_자동_운전중 AND S367_M_작업_완료 AND R361_1_M_차종_유 AND R361_1_M_차종1_AX AND S367_M_공정_차종_무 AND NOT R361_1_M_차종6_썬루프 AND S367_M_공정_제품감지_무) OR (((S367_M_동작_선택_2 AND S367_후진_ON) OR S367_HOME) AND S367_M_수동모드)) AND S367_M_LH_AX_SR_LAT_조건;
(* Rung L43 *)
S367_LH_AX_SR_LAT(사용유무 := ALWAYS_ON, 운전준비 := S367_M_운전준비_ON, 전진보조 := S367_M_LH_AX_SR_LAT_전진_보조, 후진보조 := S367_M_LH_AX_SR_LAT_후진_보조, 전진단수량 := 1, 후진단수량 := 3, 전진단1 := S367_RS_AX_LH_SR_LATCH_전진, 후진단1 := S367_RS_AX_LH_SR_LATCH_후진1, 전진단2 := _OFF, 후진단2 := S367_RS_AX_LH_SR_LATCH_후진2, 전진단3 := _OFF, 후진단3 := S367_RS_AX_LH_SR_LATCH_후진3, 전진단4 := _OFF, 후진단4 := _OFF, 전진단5 := _OFF, 후진단5 := _OFF, 전진단6 := _OFF, 후진단6 := _OFF, 전진단_지연시간 := T#0.5S, 후진단_지연시간 := T#0.5S, LS_ERR1_지연시간 := T#5S, LS_ERR2_지연시간 := T#5S, 이상리셋 := 전체_M_이상_리셋, SOL_ADV_출력 => S367_SOL_AX_LH_SR_LATCH_전진, SOL_RET_출력 => S367_SOL_AX_LH_SR_LATCH_후진, M_전진단 => S367_M_LH_AX_SR_LAT_전진단, M_후진단 => S367_M_LH_AX_SR_LAT_후진단, M_전진에러 => S367_M_LH_AX_SR_LAT_전진_LS_이상, M_후진에러 => S367_M_LH_AX_SR_LAT_후진_LS_이상, ADV_LAMP => S367_M_LH_AX_SR_LAT_전진_LAMP, RET_LAMP => S367_M_LH_AX_SR_LAT_후진_LAMP);

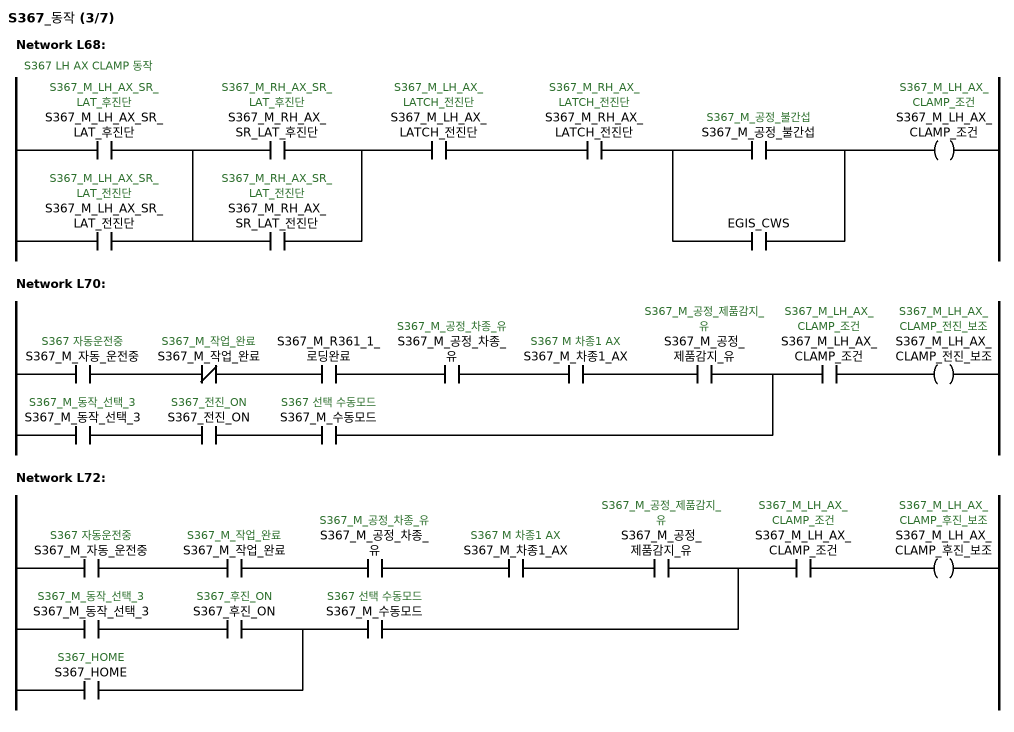
(* S367 LH AX CLAMP 동작 *)
(* Rung L68 *)
S367_M_LH_AX_CLAMP_조건 := (S367_M_LH_AX_SR_LAT_후진단 OR S367_M_LH_AX_SR_LAT_전진단) AND (S367_M_RH_AX_SR_LAT_후진단 OR S367_M_RH_AX_SR_LAT_전진단) AND S367_M_LH_AX_LATCH_전진단 AND S367_M_RH_AX_LATCH_전진단 AND (S367_M_공정_불간섭 OR EGIS_CWS);
(* Rung L70 *)
S367_M_LH_AX_CLAMP_전진_보조 := ((S367_M_자동_운전중 AND NOT S367_M_작업_완료 AND S367_M_R361_1_로딩완료 AND S367_M_공정_차종_유 AND S367_M_차종1_AX AND S367_M_공정_제품감지_유) OR (S367_M_동작_선택_3 AND S367_전진_ON AND S367_M_수동모드)) AND S367_M_LH_AX_CLAMP_조건;
(* Rung L72 *)
S367_M_LH_AX_CLAMP_후진_보조 := ((S367_M_자동_운전중 AND S367_M_작업_완료 AND S367_M_공정_차종_유 AND S367_M_차종1_AX AND S367_M_공정_제품감지_유) OR (((S367_M_동작_선택_3 AND S367_후진_ON) OR S367_HOME) AND S367_M_수동모드)) AND S367_M_LH_AX_CLAMP_조건;

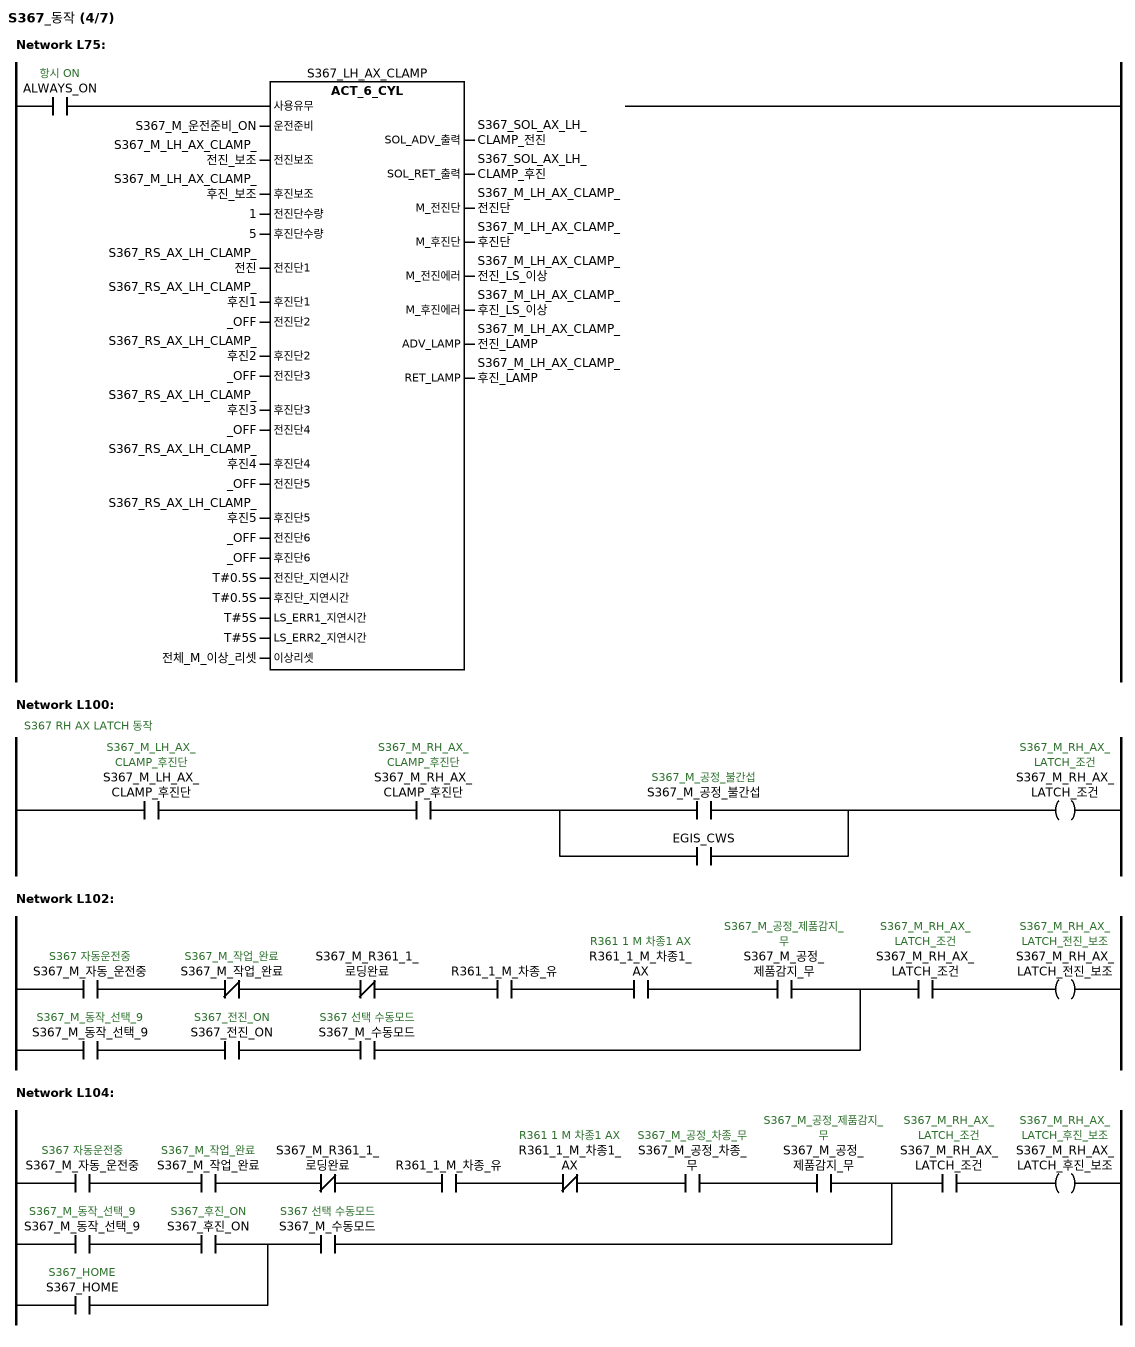
(* Rung L75 *)
S367_LH_AX_CLAMP(사용유무 := ALWAYS_ON, 운전준비 := S367_M_운전준비_ON, 전진보조 := S367_M_LH_AX_CLAMP_전진_보조, 후진보조 := S367_M_LH_AX_CLAMP_후진_보조, 전진단수량 := 1, 후진단수량 := 5, 전진단1 := S367_RS_AX_LH_CLAMP_전진, 후진단1 := S367_RS_AX_LH_CLAMP_후진1, 전진단2 := _OFF, 후진단2 := S367_RS_AX_LH_CLAMP_후진2, 전진단3 := _OFF, 후진단3 := S367_RS_AX_LH_CLAMP_후진3, 전진단4 := _OFF, 후진단4 := S367_RS_AX_LH_CLAMP_후진4, 전진단5 := _OFF, 후진단5 := S367_RS_AX_LH_CLAMP_후진5, 전진단6 := _OFF, 후진단6 := _OFF, 전진단_지연시간 := T#0.5S, 후진단_지연시간 := T#0.5S, LS_ERR1_지연시간 := T#5S, LS_ERR2_지연시간 := T#5S, 이상리셋 := 전체_M_이상_리셋, SOL_ADV_출력 => S367_SOL_AX_LH_CLAMP_전진, SOL_RET_출력 => S367_SOL_AX_LH_CLAMP_후진, M_전진단 => S367_M_LH_AX_CLAMP_전진단, M_후진단 => S367_M_LH_AX_CLAMP_후진단, M_전진에러 => S367_M_LH_AX_CLAMP_전진_LS_이상, M_후진에러 => S367_M_LH_AX_CLAMP_후진_LS_이상, ADV_LAMP => S367_M_LH_AX_CLAMP_전진_LAMP, RET_LAMP => S367_M_LH_AX_CLAMP_후진_LAMP);
(* S367 RH AX LATCH 동작 *)
(* Rung L100 *)
S367_M_RH_AX_LATCH_조건 := S367_M_LH_AX_CLAMP_후진단 AND S367_M_RH_AX_CLAMP_후진단 AND (S367_M_공정_불간섭 OR EGIS_CWS);
(* Rung L102 *)
S367_M_RH_AX_LATCH_전진_보조 := ((S367_M_자동_운전중 AND NOT S367_M_작업_완료 AND NOT S367_M_R361_1_로딩완료 AND R361_1_M_차종_유 AND R361_1_M_차종1_AX AND S367_M_공정_제품감지_무) OR (S367_M_동작_선택_9 AND S367_전진_ON AND S367_M_수동모드)) AND S367_M_RH_AX_LATCH_조건;
(* Rung L104 *)
S367_M_RH_AX_LATCH_후진_보조 := ((S367_M_자동_운전중 AND S367_M_작업_완료 AND NOT S367_M_R361_1_로딩완료 AND R361_1_M_차종_유 AND NOT R361_1_M_차종1_AX AND S367_M_공정_차종_무 AND S367_M_공정_제품감지_무) OR (((S367_M_동작_선택_9 AND S367_후진_ON) OR S367_HOME) AND S367_M_수동모드)) AND S367_M_RH_AX_LATCH_조건;

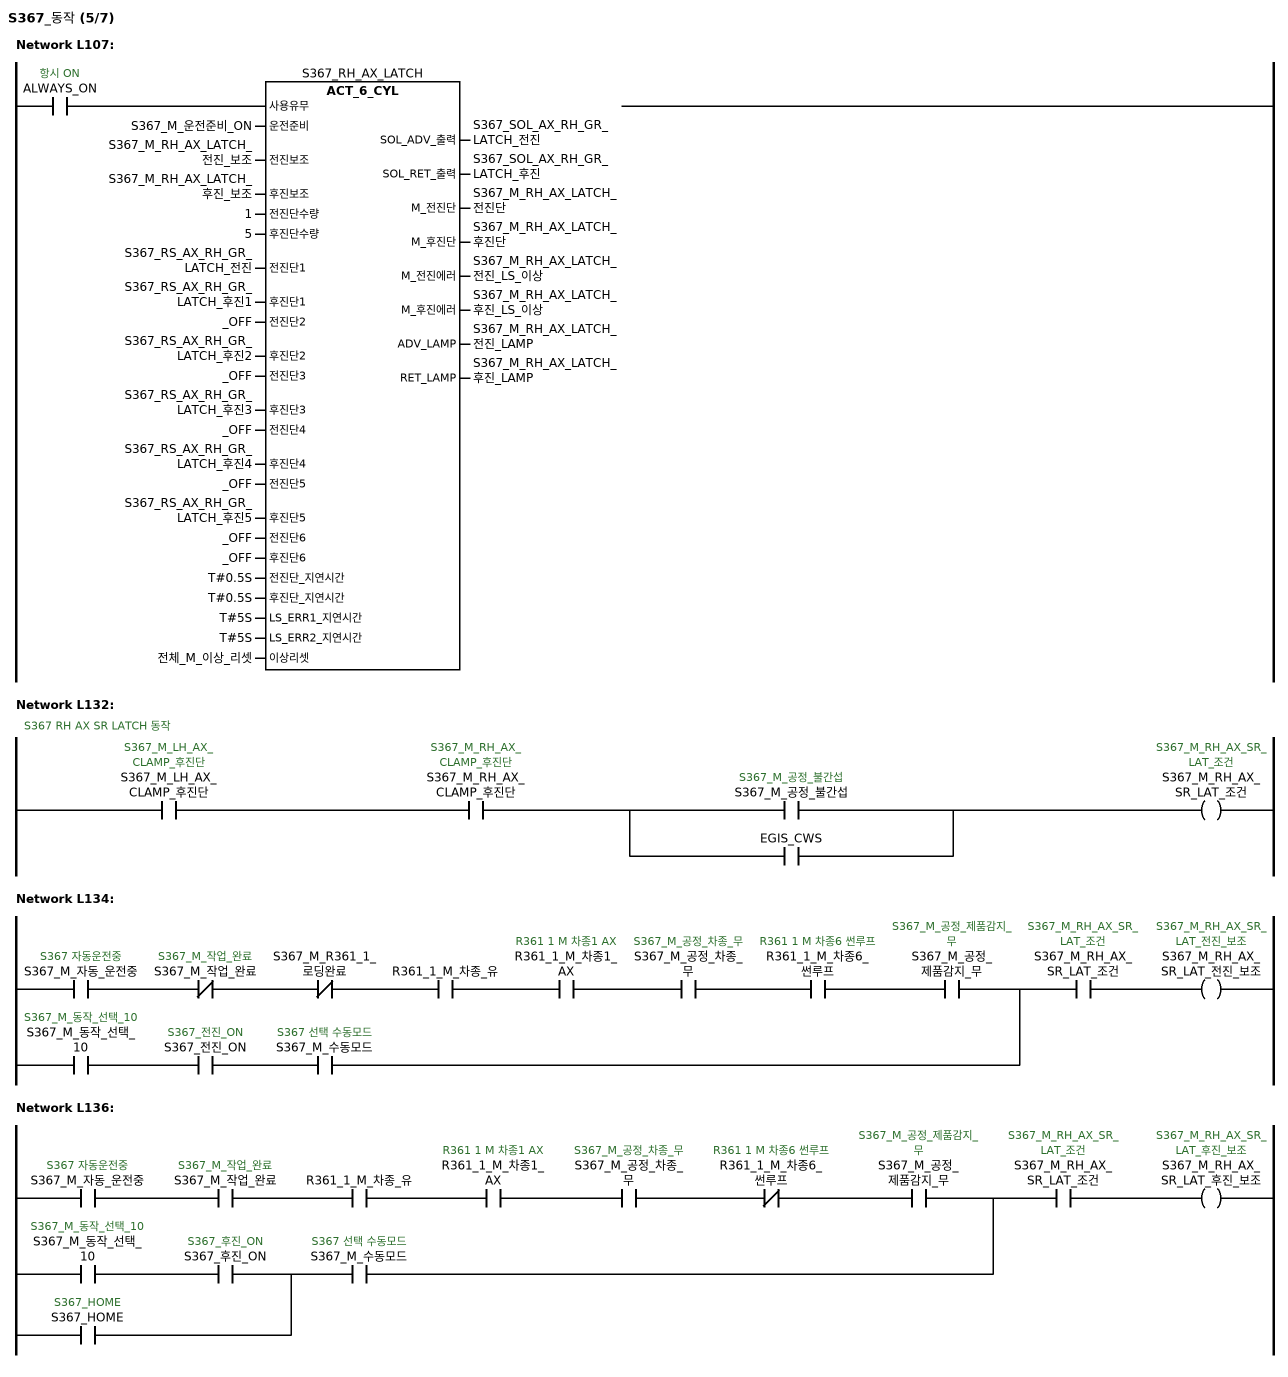
(* Rung L107 *)
S367_RH_AX_LATCH(사용유무 := ALWAYS_ON, 운전준비 := S367_M_운전준비_ON, 전진보조 := S367_M_RH_AX_LATCH_전진_보조, 후진보조 := S367_M_RH_AX_LATCH_후진_보조, 전진단수량 := 1, 후진단수량 := 5, 전진단1 := S367_RS_AX_RH_GR_LATCH_전진, 후진단1 := S367_RS_AX_RH_GR_LATCH_후진1, 전진단2 := _OFF, 후진단2 := S367_RS_AX_RH_GR_LATCH_후진2, 전진단3 := _OFF, 후진단3 := S367_RS_AX_RH_GR_LATCH_후진3, 전진단4 := _OFF, 후진단4 := S367_RS_AX_RH_GR_LATCH_후진4, 전진단5 := _OFF, 후진단5 := S367_RS_AX_RH_GR_LATCH_후진5, 전진단6 := _OFF, 후진단6 := _OFF, 전진단_지연시간 := T#0.5S, 후진단_지연시간 := T#0.5S, LS_ERR1_지연시간 := T#5S, LS_ERR2_지연시간 := T#5S, 이상리셋 := 전체_M_이상_리셋, SOL_ADV_출력 => S367_SOL_AX_RH_GR_LATCH_전진, SOL_RET_출력 => S367_SOL_AX_RH_GR_LATCH_후진, M_전진단 => S367_M_RH_AX_LATCH_전진단, M_후진단 => S367_M_RH_AX_LATCH_후진단, M_전진에러 => S367_M_RH_AX_LATCH_전진_LS_이상, M_후진에러 => S367_M_RH_AX_LATCH_후진_LS_이상, ADV_LAMP => S367_M_RH_AX_LATCH_전진_LAMP, RET_LAMP => S367_M_RH_AX_LATCH_후진_LAMP);
(* S367 RH AX SR LATCH 동작 *)
(* Rung L132 *)
S367_M_RH_AX_SR_LAT_조건 := S367_M_LH_AX_CLAMP_후진단 AND S367_M_RH_AX_CLAMP_후진단 AND (S367_M_공정_불간섭 OR EGIS_CWS);
(* Rung L134 *)
S367_M_RH_AX_SR_LAT_전진_보조 := ((S367_M_자동_운전중 AND NOT S367_M_작업_완료 AND NOT S367_M_R361_1_로딩완료 AND R361_1_M_차종_유 AND R361_1_M_차종1_AX AND S367_M_공정_차종_무 AND R361_1_M_차종6_썬루프 AND S367_M_공정_제품감지_무) OR (S367_M_동작_선택_10 AND S367_전진_ON AND S367_M_수동모드)) AND S367_M_RH_AX_SR_LAT_조건;
(* Rung L136 *)
S367_M_RH_AX_SR_LAT_후진_보조 := ((S367_M_자동_운전중 AND S367_M_작업_완료 AND R361_1_M_차종_유 AND R361_1_M_차종1_AX AND S367_M_공정_차종_무 AND NOT R361_1_M_차종6_썬루프 AND S367_M_공정_제품감지_무) OR (((S367_M_동작_선택_10 AND S367_후진_ON) OR S367_HOME) AND S367_M_수동모드)) AND S367_M_RH_AX_SR_LAT_조건;

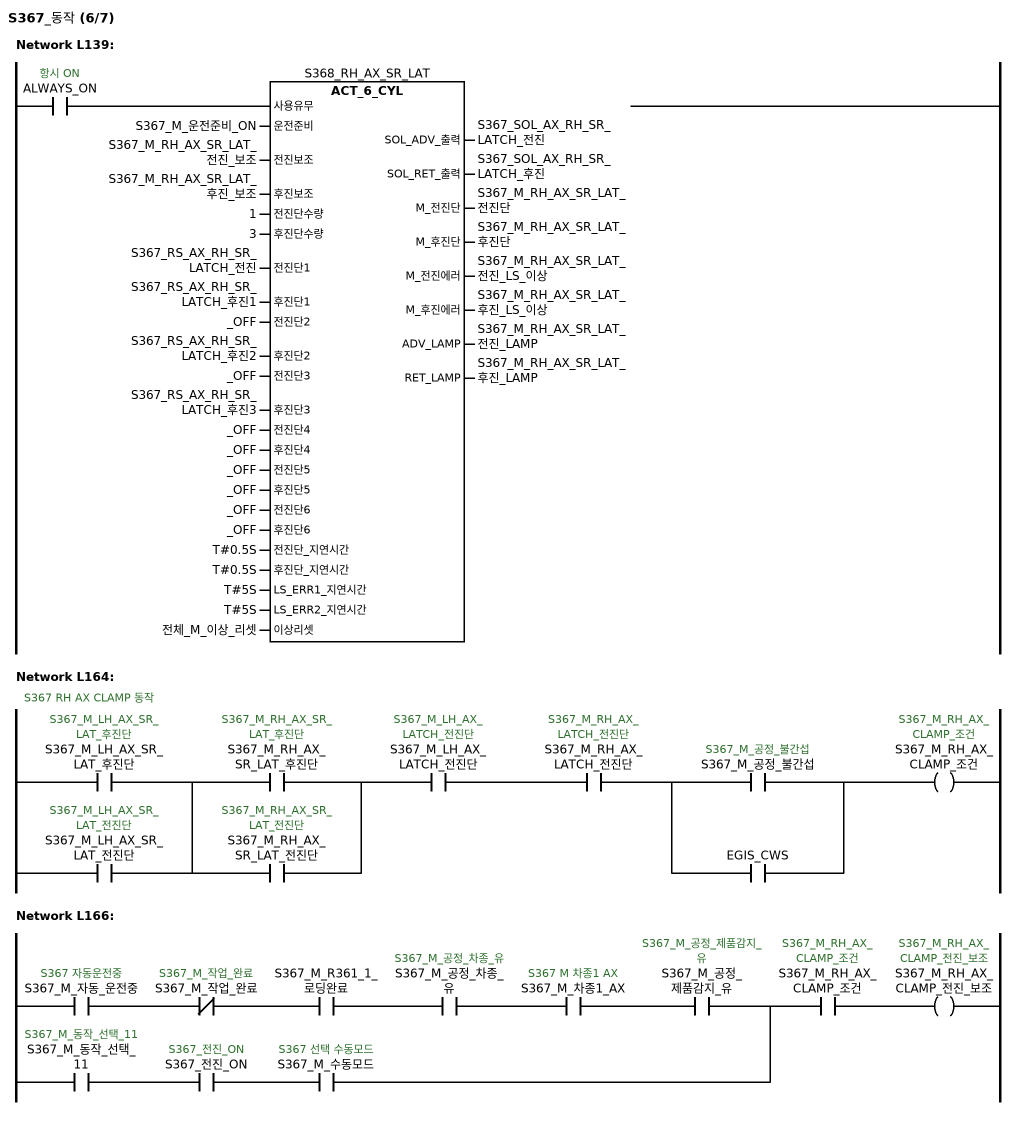
(* Rung L139 *)
S368_RH_AX_SR_LAT(사용유무 := ALWAYS_ON, 운전준비 := S367_M_운전준비_ON, 전진보조 := S367_M_RH_AX_SR_LAT_전진_보조, 후진보조 := S367_M_RH_AX_SR_LAT_후진_보조, 전진단수량 := 1, 후진단수량 := 3, 전진단1 := S367_RS_AX_RH_SR_LATCH_전진, 후진단1 := S367_RS_AX_RH_SR_LATCH_후진1, 전진단2 := _OFF, 후진단2 := S367_RS_AX_RH_SR_LATCH_후진2, 전진단3 := _OFF, 후진단3 := S367_RS_AX_RH_SR_LATCH_후진3, 전진단4 := _OFF, 후진단4 := _OFF, 전진단5 := _OFF, 후진단5 := _OFF, 전진단6 := _OFF, 후진단6 := _OFF, 전진단_지연시간 := T#0.5S, 후진단_지연시간 := T#0.5S, LS_ERR1_지연시간 := T#5S, LS_ERR2_지연시간 := T#5S, 이상리셋 := 전체_M_이상_리셋, SOL_ADV_출력 => S367_SOL_AX_RH_SR_LATCH_전진, SOL_RET_출력 => S367_SOL_AX_RH_SR_LATCH_후진, M_전진단 => S367_M_RH_AX_SR_LAT_전진단, M_후진단 => S367_M_RH_AX_SR_LAT_후진단, M_전진에러 => S367_M_RH_AX_SR_LAT_전진_LS_이상, M_후진에러 => S367_M_RH_AX_SR_LAT_후진_LS_이상, ADV_LAMP => S367_M_RH_AX_SR_LAT_전진_LAMP, RET_LAMP => S367_M_RH_AX_SR_LAT_후진_LAMP);
(* S367 RH AX CLAMP 동작 *)
(* Rung L164 *)
S367_M_RH_AX_CLAMP_조건 := (S367_M_LH_AX_SR_LAT_후진단 OR S367_M_LH_AX_SR_LAT_전진단) AND (S367_M_RH_AX_SR_LAT_후진단 OR S367_M_RH_AX_SR_LAT_전진단) AND S367_M_LH_AX_LATCH_전진단 AND S367_M_RH_AX_LATCH_전진단 AND (S367_M_공정_불간섭 OR EGIS_CWS);
(* Rung L166 *)
S367_M_RH_AX_CLAMP_전진_보조 := ((S367_M_자동_운전중 AND NOT S367_M_작업_완료 AND S367_M_R361_1_로딩완료 AND S367_M_공정_차종_유 AND S367_M_차종1_AX AND S367_M_공정_제품감지_유) OR (S367_M_동작_선택_11 AND S367_전진_ON AND S367_M_수동모드)) AND S367_M_RH_AX_CLAMP_조건;

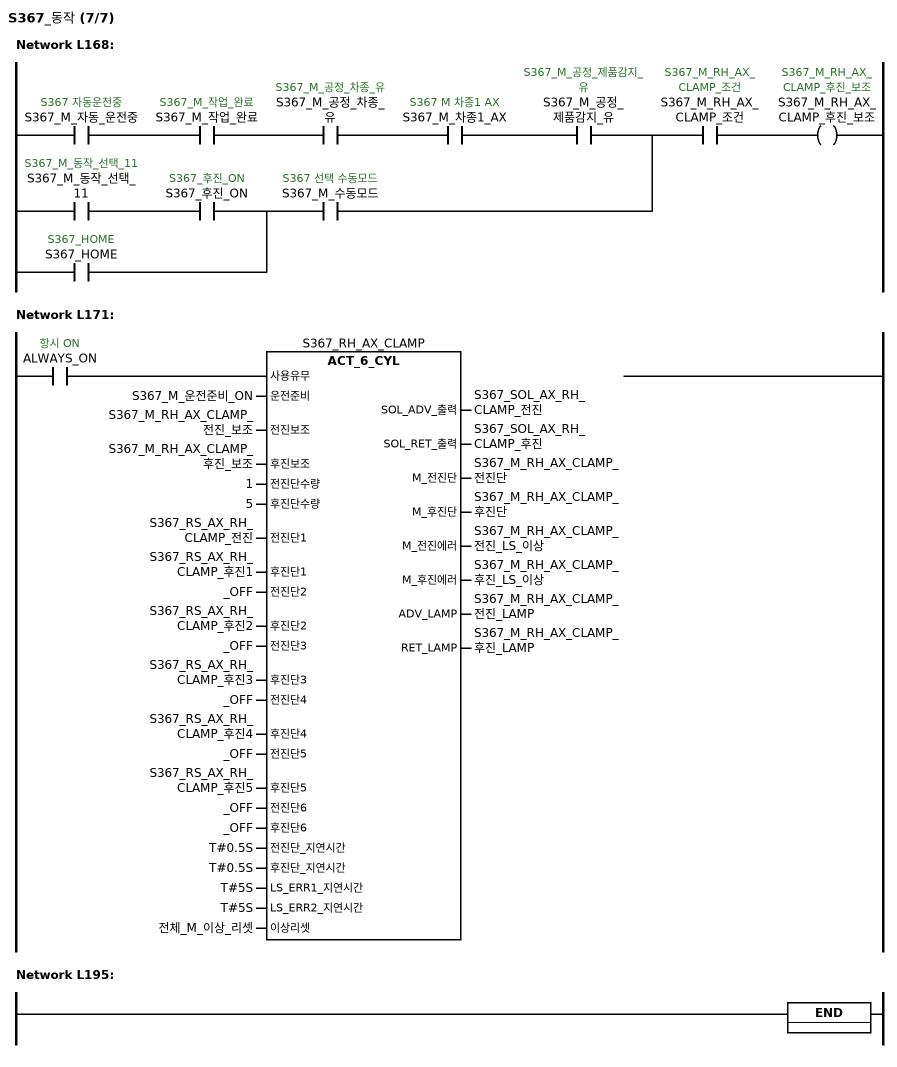
(* Rung L168 *)
S367_M_RH_AX_CLAMP_후진_보조 := ((S367_M_자동_운전중 AND S367_M_작업_완료 AND S367_M_공정_차종_유 AND S367_M_차종1_AX AND S367_M_공정_제품감지_유) OR (((S367_M_동작_선택_11 AND S367_후진_ON) OR S367_HOME) AND S367_M_수동모드)) AND S367_M_RH_AX_CLAMP_조건;
(* Rung L171 *)
S367_RH_AX_CLAMP(사용유무 := ALWAYS_ON, 운전준비 := S367_M_운전준비_ON, 전진보조 := S367_M_RH_AX_CLAMP_전진_보조, 후진보조 := S367_M_RH_AX_CLAMP_후진_보조, 전진단수량 := 1, 후진단수량 := 5, 전진단1 := S367_RS_AX_RH_CLAMP_전진, 후진단1 := S367_RS_AX_RH_CLAMP_후진1, 전진단2 := _OFF, 후진단2 := S367_RS_AX_RH_CLAMP_후진2, 전진단3 := _OFF, 후진단3 := S367_RS_AX_RH_CLAMP_후진3, 전진단4 := _OFF, 후진단4 := S367_RS_AX_RH_CLAMP_후진4, 전진단5 := _OFF, 후진단5 := S367_RS_AX_RH_CLAMP_후진5, 전진단6 := _OFF, 후진단6 := _OFF, 전진단_지연시간 := T#0.5S, 후진단_지연시간 := T#0.5S, LS_ERR1_지연시간 := T#5S, LS_ERR2_지연시간 := T#5S, 이상리셋 := 전체_M_이상_리셋, SOL_ADV_출력 => S367_SOL_AX_RH_CLAMP_전진, SOL_RET_출력 => S367_SOL_AX_RH_CLAMP_후진, M_전진단 => S367_M_RH_AX_CLAMP_전진단, M_후진단 => S367_M_RH_AX_CLAMP_후진단, M_전진에러 => S367_M_RH_AX_CLAMP_전진_LS_이상, M_후진에러 => S367_M_RH_AX_CLAMP_후진_LS_이상, ADV_LAMP => S367_M_RH_AX_CLAMP_전진_LAMP, RET_LAMP => S367_M_RH_AX_CLAMP_후진_LAMP);
(* Rung L195 *)
END();
END_PROGRAM

PROGRAM S367_이상 (* task: 스캔 프로그램 *)
VAR
    INST : TON;
    INST1 : TON;
    INST10 : TON;
    INST11 : TON;
    INST12 : TON;
    INST13 : TON;
    INST14 : TON;
    INST15 : TON;
    INST16 : TON;
    INST17 : TON;
    INST18 : TON;
    INST19 : TON;
    INST2 : TON;
    INST20 : TON;
    INST21 : TON;
    INST22 : TON;
    INST23 : TON;
    INST24 : TON;
    INST25 : TON;
    INST26 : TON;
    INST3 : TON;
    INST8 : TON;
    INST9 : TON;
END_VAR
VAR_EXTERNAL
    S367_6_20_PLC_BOX_CP_TRIP : BOOL; (* AT %MW86202.15 *) (* S367_6_20_PLC_BOX_CP_TRIP *)
    S367_6_21_PLC_BOX_CP_TRIP : BOOL; (* AT %MW86212.15 *) (* S367_6_21_PLC_BOX_CP_TRIP *)
    S367_공기압_AIR_CHECK : BOOL; (* AT %MW86202.14 *) (* S367_공기압_AIR_CHECK *)
    _0006_EB20_CFG_ER : BOOL; (* AT %MW186034.0 *) (* EB 구성 에러 *)
    _0006_EB20_DEER : BOOL; (* AT %MW186034.1 *) (* EB 운전 중 탈락 *)
    _0006_EB20_IO_DEER : BOOL; (* AT %MW186035.2 *) (* EB IO 탈락 에러 *)
    _0006_EB20_IO_TYER : BOOL; (* AT %MW186035.1 *) (* EB IO 타입 에러 *)
    _0006_EB21_CFG_ER : BOOL; (* AT %MW186040.0 *) (* EB 구성 에러 *)
    _0006_EB21_DEER : BOOL; (* AT %MW186040.1 *) (* EB 운전 중 탈락 *)
    _0006_EB21_IO_DEER : BOOL; (* AT %MW186041.2 *) (* EB IO 탈락 에러 *)
    _0006_EB21_IO_TYER : BOOL; (* AT %MW186041.1 *) (* EB IO 타입 에러 *)
    _0007_EB10_CFG_ER : BOOL; (* AT %MW187040.0 *) (* EB 구성 에러 *)
    _0007_EB10_DEER : BOOL; (* AT %MW187040.1 *) (* EB 운전 중 탈락 *)
    _0007_EB10_IO_DEER : BOOL; (* AT %MW187041.2 *) (* EB IO 탈락 에러 *)
    _0007_EB10_IO_TYER : BOOL; (* AT %MW187041.1 *) (* EB IO 타입 에러 *)
END_VAR
VAR_EXTERNAL RETAIN
    S367_LH_M_NODE_6_21_통신_이상 : BOOL; (* AT %MW3524.0 *)
    S367_M_LH_AX_CLAMP_전진_LS_이상 : BOOL; (* AT %MW3602.5 *) (* S367_M_LH_AX_CLAMP_전진_LS_이상 *)
    S367_M_LH_AX_CLAMP_후진_LS_이상 : BOOL; (* AT %MW3602.6 *) (* S367_M_LH_AX_CLAMP_후진_LS_이상 *)
    S367_M_LH_AX_LATCH_전진_LS_이상 : BOOL; (* AT %MW3600.5 *) (* S367_M_LH_AX_LATCH_전진_LS_이상 *)
    S367_M_LH_AX_LATCH_후진_LS_이상 : BOOL; (* AT %MW3600.6 *) (* S367_M_LH_AX_LATCH_후진_LS_이상 *)
    S367_M_LH_AX_SR_LAT_전진_LS_이상 : BOOL; (* AT %MW3601.5 *) (* S367_M_LH_AX_SR_LAT_전진_LS_이상 *)
    S367_M_LH_AX_SR_LAT_후진_LS_이상 : BOOL; (* AT %MW3601.6 *) (* S367_M_LH_AX_SR_LAT_후진_LS_이상 *)
    S367_M_LH_CP_OFF : BOOL; (* AT %MW3517.0 *) (* S367_M_LH_CP_OFF *)
    S367_M_R361_1_로딩완료 : BOOL; (* AT %MW3501.1 *)
    S367_M_RH_AX_CLAMP_전진_LS_이상 : BOOL; (* AT %MW3610.5 *) (* S367_M_RH_AX_CLAMP_전진_LS_이상 *)
    S367_M_RH_AX_CLAMP_후진_LS_이상 : BOOL; (* AT %MW3610.6 *) (* S367_M_RH_AX_CLAMP_후진_LS_이상 *)
    S367_M_RH_AX_LATCH_전진_LS_이상 : BOOL; (* AT %MW3608.5 *) (* S367_M_RH_AX_LATCH_전진_LS_이상 *)
    S367_M_RH_AX_LATCH_후진_LS_이상 : BOOL; (* AT %MW3608.6 *) (* S367_M_RH_AX_LATCH_후진_LS_이상 *)
    S367_M_RH_AX_SR_LAT_전진_LS_이상 : BOOL; (* AT %MW3609.5 *) (* S367_M_RH_AX_SR_LAT_전진_LS_이상 *)
    S367_M_RH_AX_SR_LAT_후진_LS_이상 : BOOL; (* AT %MW3609.6 *) (* S367_M_RH_AX_SR_LAT_후진_LS_이상 *)
    S367_M_RH_CP_OFF : BOOL; (* AT %MW3517.1 *) (* S367_M_RH_CP_OFF *)
    S367_M_공정_FRT_제품감지_무 : BOOL; (* AT %MW3501.8 *)
    S367_M_공정_FRT_제품감지_유 : BOOL; (* AT %MW3501.7 *)
    S367_M_공정_FRT_제품감지_이상 : BOOL; (* AT %MW3514.0 *) (* S367_M_LH_제품감지_이상 *)
    S367_M_공정_RR_제품감지_무 : BOOL; (* AT %MW3501.10 *)
    S367_M_공정_RR_제품감지_유 : BOOL; (* AT %MW3501.9 *)
    S367_M_공정_RR_제품감지_이상 : BOOL; (* AT %MW3514.1 *) (* S367_M_RH_제품감지_이상 *)
    S367_M_공정_불간섭 : BOOL; (* AT %MW3504.1 *) (* S367_M_공정_불간섭 *)
    S367_M_공정_제품감지_무 : BOOL; (* AT %MW3501.6 *) (* S367_M_공정_제품감지_무 *)
    S367_M_공정_제품감지_유 : BOOL; (* AT %MW3501.5 *) (* S367_M_공정_제품감지_유 *)
    S367_M_공정_차종_유 : BOOL; (* AT %MW3502.0 *) (* S367_M_공정_차종_유 *)
    S367_M_자동_운전중 : BOOL; (* AT %MW3500.4 *) (* S367 자동운전중 *)
    S367_M_총괄_CP_이상 : BOOL; (* AT %MW3509.7 *) (* S367 CP OFF 이상 *)
    S367_M_총괄_CT_이상 : BOOL; (* AT %MW3510.4 *) (* S367   TACK TIME 이상 *)
    S367_M_총괄_EOCR_이상 : BOOL; (* AT %MW3509.8 *) (* S367_M_총괄_EOCR_이상 *)
    S367_M_총괄_INV_이상 : BOOL; (* AT %MW3509.9 *) (* S367_M_총괄_INV_이상 *)
    S367_M_총괄_LS_이상 : BOOL; (* AT %MW3509.15 *) (* S367 LS 이상 *)
    S367_M_총괄_MATCH_이상 : BOOL; (* AT %MW3510.0 *) (* S367 매트SW 이상 *)
    S367_M_총괄_MC_이상 : BOOL; (* AT %MW3509.13 *) (* S367_M_총괄_MC_이상 *)
    S367_M_총괄_NFB_이상 : BOOL; (* AT %MW3509.11 *) (* S367_M_총괄_NFB_이상 *)
    S367_M_총괄_ROBOT_이상 : BOOL; (* AT %MW3510.1 *) (* S367 ROBOT 이상 *)
    S367_M_총괄_SAFETY_이상 : BOOL; (* AT %MW3509.2 *) (* S367_M_총괄_SAFETY_이상 *)
    S367_M_총괄_공기압_이상 : BOOL; (* AT %MW3509.3 *) (* S367 공기압 이상 *)
    S367_M_총괄_사양_이상 : BOOL; (* AT %MW3509.6 *) (* S367 사양 이상 *)
    S367_M_총괄_오버런_이상 : BOOL; (* AT %MW3509.12 *) (* S367_M_총괄_오버런_이상 *)
    S367_M_총괄_용접타점수_이상 : BOOL; (* AT %MW3510.2 *) (* S367 용접타점수 이상 *)
    S367_M_총괄_이상 : BOOL; (* AT %MW3509.0 *) (* S367_M_총괄_이상 *)
    S367_M_총괄_제품감지_이상 : BOOL; (* AT %MW3509.4 *) (* S367 제품감지 이상 *)
    S367_M_총괄_차종_이상 : BOOL; (* AT %MW3509.5 *) (* S367 차종 이상 *)
    S367_M_총괄_통신_이상 : BOOL; (* AT %MW3509.14 *) (* S367 통신이상 *)
    S367_RH_M_NODE_6_20_통신_이상 : BOOL; (* AT %MW3524.1 *)
    전체_M_이상_리셋 : BOOL; (* AT %MW308.2 *) (* ALL공정 PB 이상리셋 *)
END_VAR

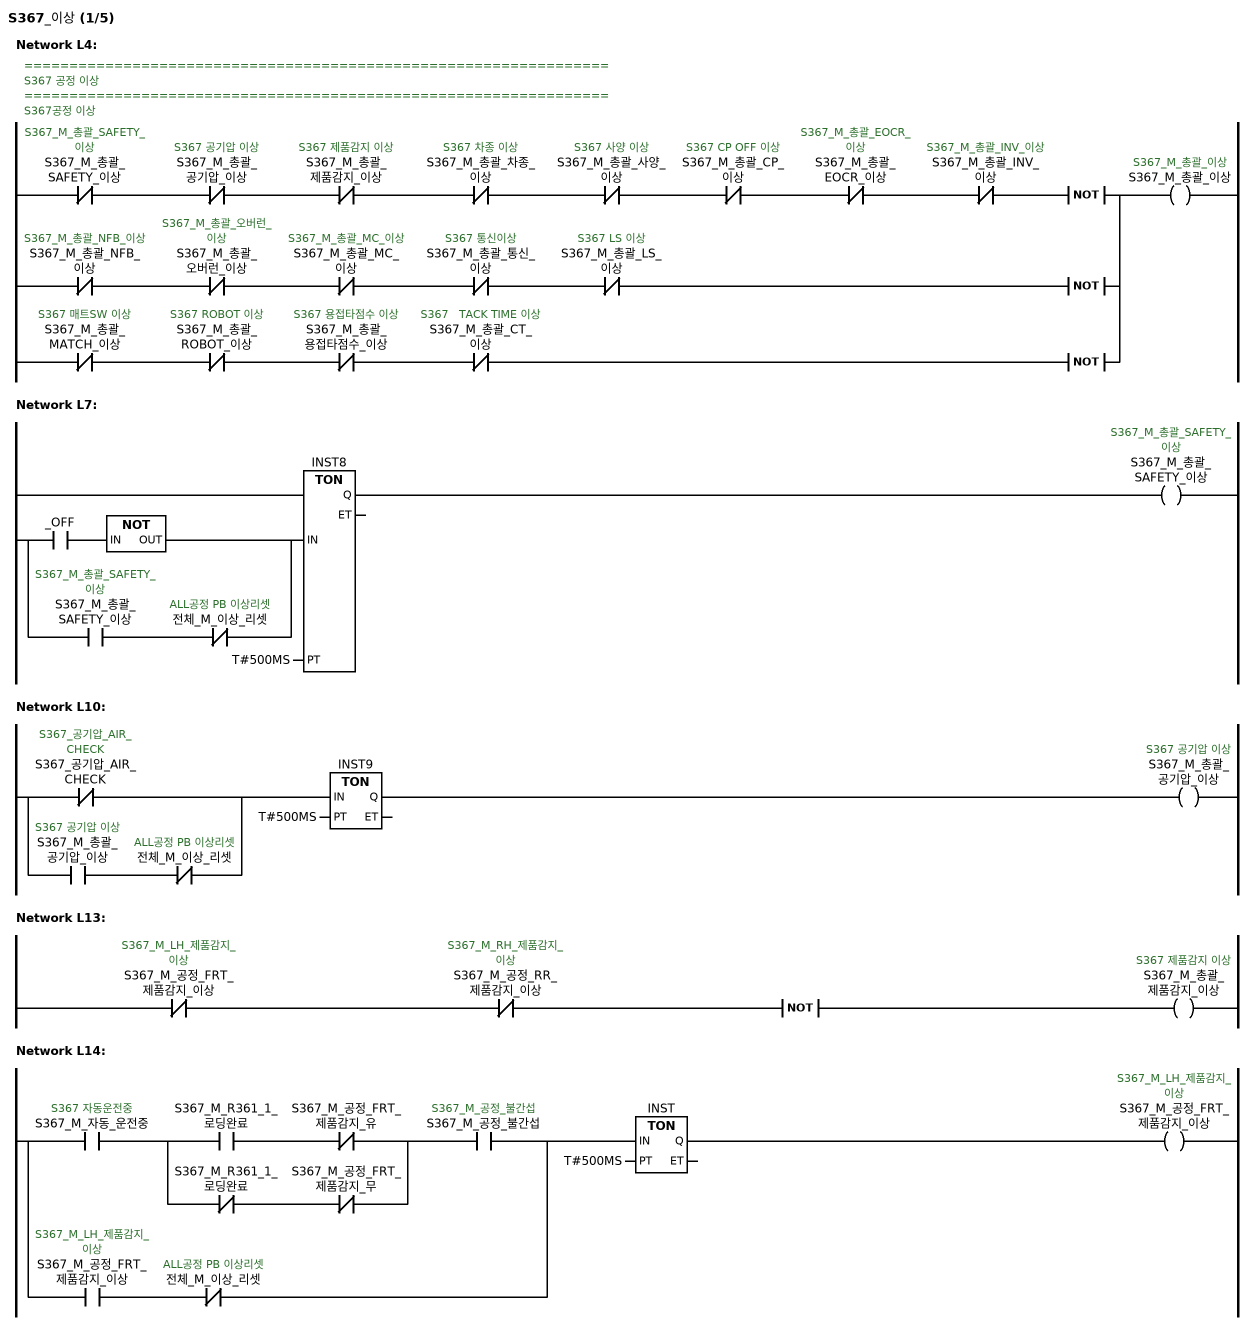
(* ================================================================= *)
(* S367 공정 이상 *)
(* ================================================================= *)
(* S367공정 이상 *)
(* Rung L4 *)
S367_M_총괄_이상 := NOT (NOT S367_M_총괄_SAFETY_이상 AND NOT S367_M_총괄_공기압_이상 AND NOT S367_M_총괄_제품감지_이상 AND NOT S367_M_총괄_차종_이상 AND NOT S367_M_총괄_사양_이상 AND NOT S367_M_총괄_CP_이상 AND NOT S367_M_총괄_EOCR_이상 AND NOT S367_M_총괄_INV_이상) OR NOT (NOT S367_M_총괄_NFB_이상 AND NOT S367_M_총괄_오버런_이상 AND NOT S367_M_총괄_MC_이상 AND NOT S367_M_총괄_통신_이상 AND NOT S367_M_총괄_LS_이상) OR NOT (NOT S367_M_총괄_MATCH_이상 AND NOT S367_M_총괄_ROBOT_이상 AND NOT S367_M_총괄_용접타점수_이상 AND NOT S367_M_총괄_CT_이상);
(* Rung L7 *)
INST8(IN := (NOT _OFF) OR (S367_M_총괄_SAFETY_이상 AND NOT 전체_M_이상_리셋), PT := T#500MS);
S367_M_총괄_SAFETY_이상 := INST8.Q;
(* Rung L10 *)
INST9(IN := NOT S367_공기압_AIR_CHECK OR (S367_M_총괄_공기압_이상 AND NOT 전체_M_이상_리셋), PT := T#500MS);
S367_M_총괄_공기압_이상 := INST9.Q;
(* Rung L13 *)
S367_M_총괄_제품감지_이상 := NOT (NOT S367_M_공정_FRT_제품감지_이상 AND NOT S367_M_공정_RR_제품감지_이상);
(* Rung L14 *)
INST(IN := (S367_M_자동_운전중 AND ((S367_M_R361_1_로딩완료 AND NOT S367_M_공정_FRT_제품감지_유) OR (NOT S367_M_R361_1_로딩완료 AND NOT S367_M_공정_FRT_제품감지_무)) AND S367_M_공정_불간섭) OR (S367_M_공정_FRT_제품감지_이상 AND NOT 전체_M_이상_리셋), PT := T#500MS);
S367_M_공정_FRT_제품감지_이상 := INST.Q;

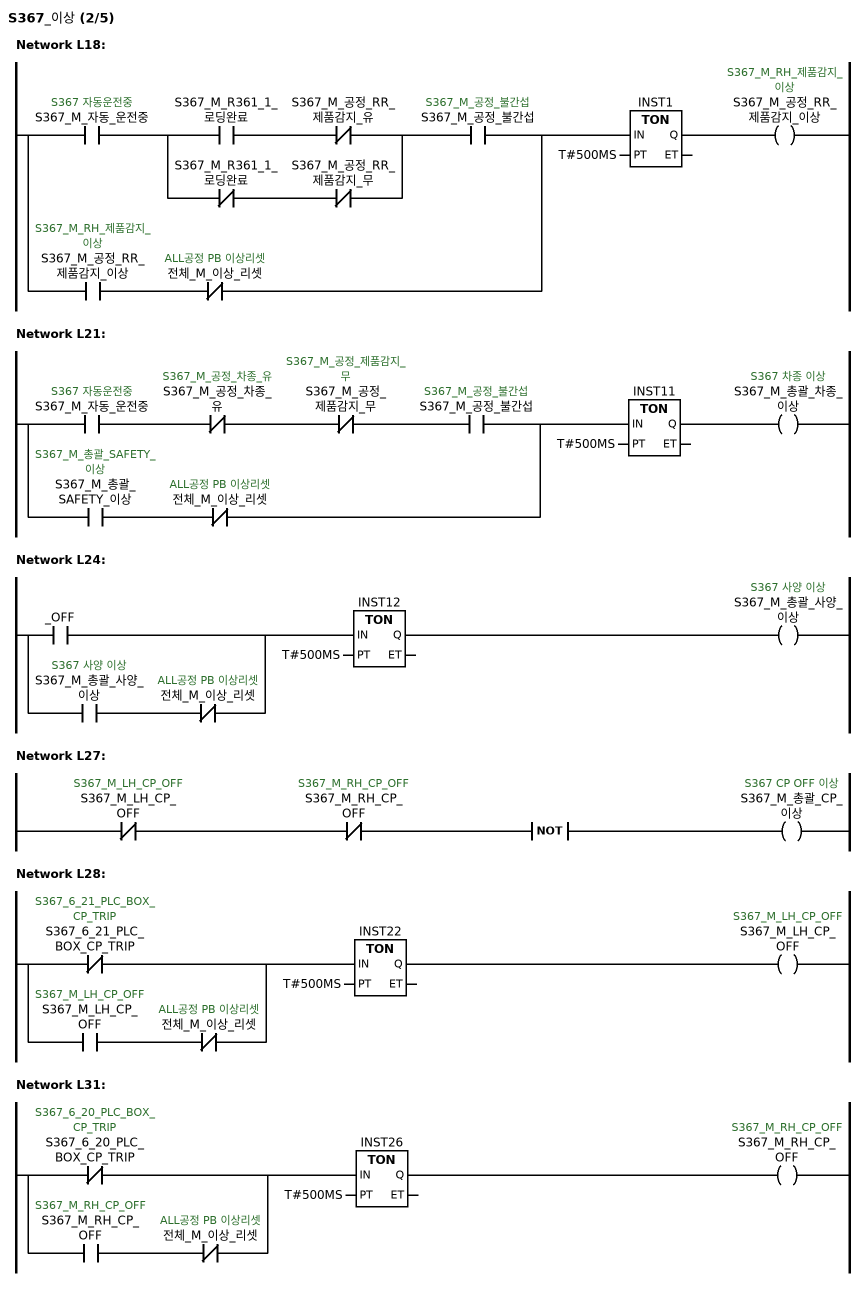
(* Rung L18 *)
INST1(IN := (S367_M_자동_운전중 AND ((S367_M_R361_1_로딩완료 AND NOT S367_M_공정_RR_제품감지_유) OR (NOT S367_M_R361_1_로딩완료 AND NOT S367_M_공정_RR_제품감지_무)) AND S367_M_공정_불간섭) OR (S367_M_공정_RR_제품감지_이상 AND NOT 전체_M_이상_리셋), PT := T#500MS);
S367_M_공정_RR_제품감지_이상 := INST1.Q;
(* Rung L21 *)
INST11(IN := (S367_M_자동_운전중 AND NOT S367_M_공정_차종_유 AND NOT S367_M_공정_제품감지_무 AND S367_M_공정_불간섭) OR (S367_M_총괄_SAFETY_이상 AND NOT 전체_M_이상_리셋), PT := T#500MS);
S367_M_총괄_차종_이상 := INST11.Q;
(* Rung L24 *)
INST12(IN := _OFF OR (S367_M_총괄_사양_이상 AND NOT 전체_M_이상_리셋), PT := T#500MS);
S367_M_총괄_사양_이상 := INST12.Q;
(* Rung L27 *)
S367_M_총괄_CP_이상 := NOT (NOT S367_M_LH_CP_OFF AND NOT S367_M_RH_CP_OFF);
(* Rung L28 *)
INST22(IN := NOT S367_6_21_PLC_BOX_CP_TRIP OR (S367_M_LH_CP_OFF AND NOT 전체_M_이상_리셋), PT := T#500MS);
S367_M_LH_CP_OFF := INST22.Q;
(* Rung L31 *)
INST26(IN := NOT S367_6_20_PLC_BOX_CP_TRIP OR (S367_M_RH_CP_OFF AND NOT 전체_M_이상_리셋), PT := T#500MS);
S367_M_RH_CP_OFF := INST26.Q;

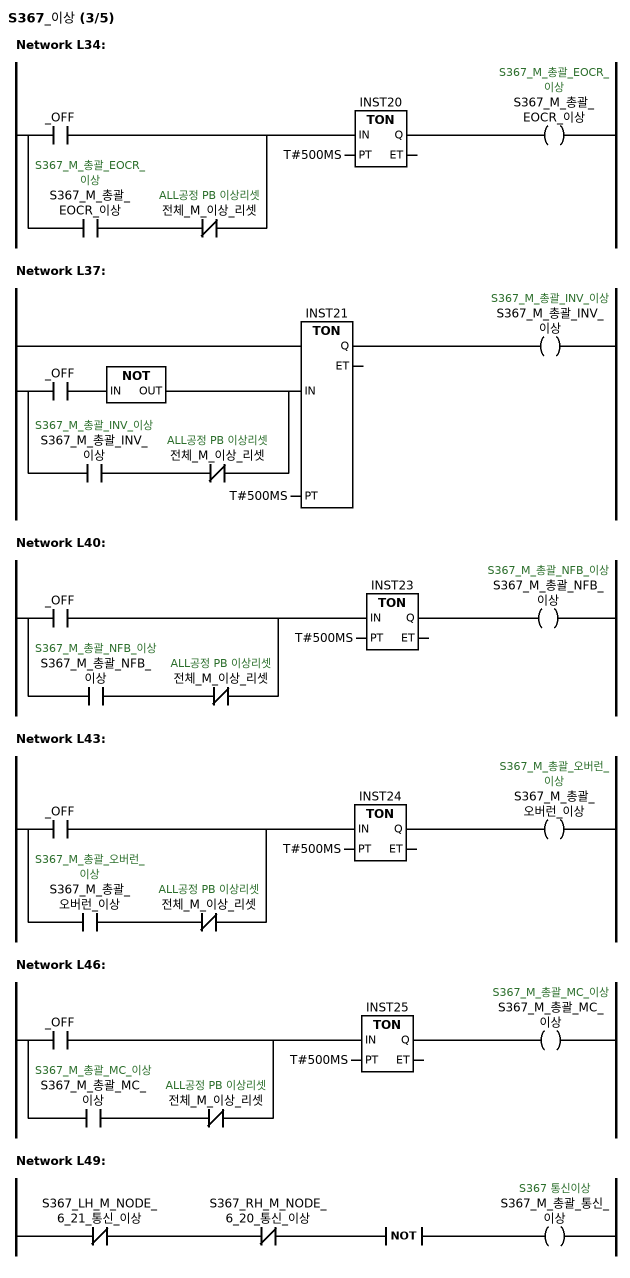
(* Rung L34 *)
INST20(IN := _OFF OR (S367_M_총괄_EOCR_이상 AND NOT 전체_M_이상_리셋), PT := T#500MS);
S367_M_총괄_EOCR_이상 := INST20.Q;
(* Rung L37 *)
INST21(IN := (NOT _OFF) OR (S367_M_총괄_INV_이상 AND NOT 전체_M_이상_리셋), PT := T#500MS);
S367_M_총괄_INV_이상 := INST21.Q;
(* Rung L40 *)
INST23(IN := _OFF OR (S367_M_총괄_NFB_이상 AND NOT 전체_M_이상_리셋), PT := T#500MS);
S367_M_총괄_NFB_이상 := INST23.Q;
(* Rung L43 *)
INST24(IN := _OFF OR (S367_M_총괄_오버런_이상 AND NOT 전체_M_이상_리셋), PT := T#500MS);
S367_M_총괄_오버런_이상 := INST24.Q;
(* Rung L46 *)
INST25(IN := _OFF OR (S367_M_총괄_MC_이상 AND NOT 전체_M_이상_리셋), PT := T#500MS);
S367_M_총괄_MC_이상 := INST25.Q;
(* Rung L49 *)
S367_M_총괄_통신_이상 := NOT (NOT S367_LH_M_NODE_6_21_통신_이상 AND NOT S367_RH_M_NODE_6_20_통신_이상);

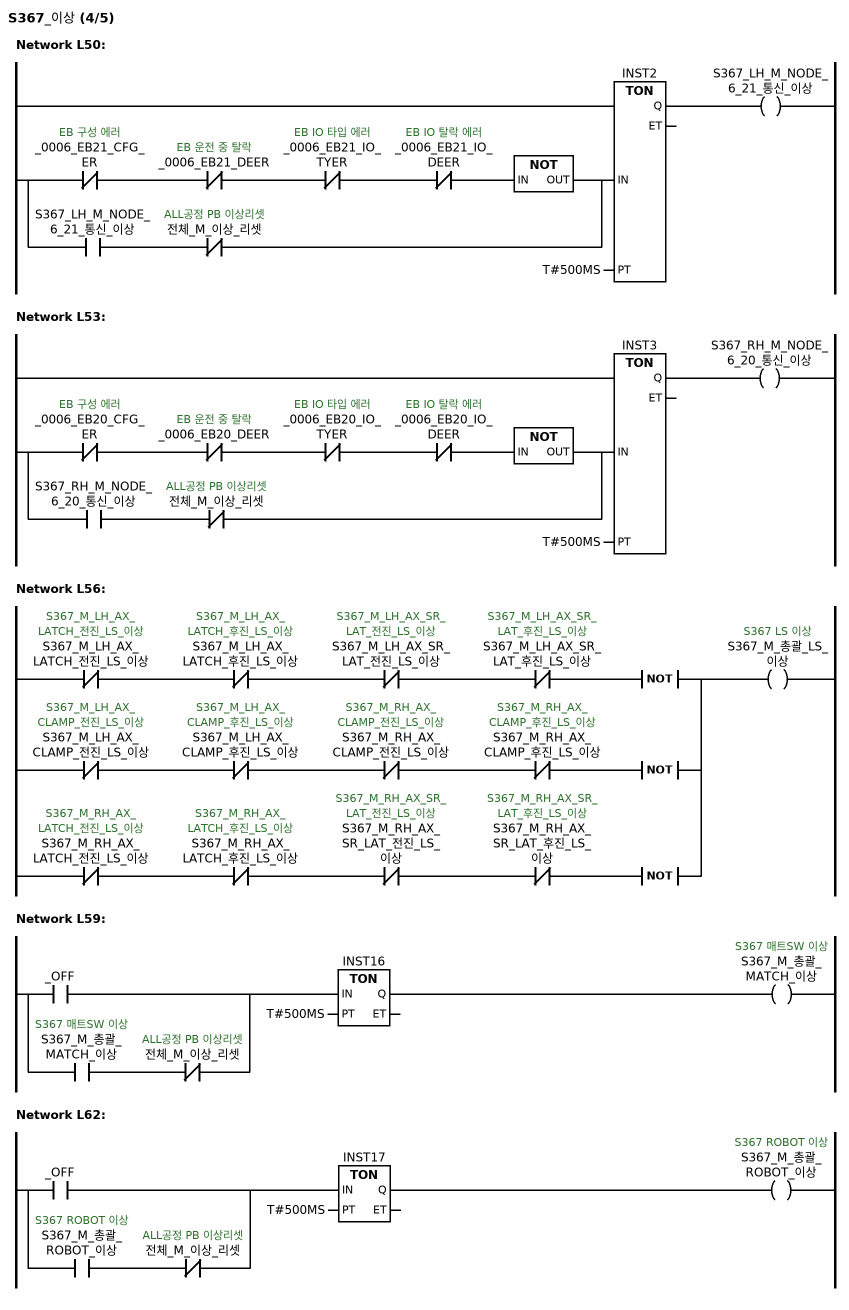
(* Rung L50 *)
INST2(IN := (NOT (NOT _0006_EB21_CFG_ER AND NOT _0006_EB21_DEER AND NOT _0006_EB21_IO_TYER AND NOT _0006_EB21_IO_DEER)) OR (S367_LH_M_NODE_6_21_통신_이상 AND NOT 전체_M_이상_리셋), PT := T#500MS);
S367_LH_M_NODE_6_21_통신_이상 := INST2.Q;
(* Rung L53 *)
INST3(IN := (NOT (NOT _0006_EB20_CFG_ER AND NOT _0006_EB20_DEER AND NOT _0006_EB20_IO_TYER AND NOT _0006_EB20_IO_DEER)) OR (S367_RH_M_NODE_6_20_통신_이상 AND NOT 전체_M_이상_리셋), PT := T#500MS);
S367_RH_M_NODE_6_20_통신_이상 := INST3.Q;
(* Rung L56 *)
S367_M_총괄_LS_이상 := NOT (NOT S367_M_LH_AX_LATCH_전진_LS_이상 AND NOT S367_M_LH_AX_LATCH_후진_LS_이상 AND NOT S367_M_LH_AX_SR_LAT_전진_LS_이상 AND NOT S367_M_LH_AX_SR_LAT_후진_LS_이상) OR NOT (NOT S367_M_LH_AX_CLAMP_전진_LS_이상 AND NOT S367_M_LH_AX_CLAMP_후진_LS_이상 AND NOT S367_M_RH_AX_CLAMP_전진_LS_이상 AND NOT S367_M_RH_AX_CLAMP_후진_LS_이상) OR NOT (NOT S367_M_RH_AX_LATCH_전진_LS_이상 AND NOT S367_M_RH_AX_LATCH_후진_LS_이상 AND NOT S367_M_RH_AX_SR_LAT_전진_LS_이상 AND NOT S367_M_RH_AX_SR_LAT_후진_LS_이상);
(* Rung L59 *)
INST16(IN := _OFF OR (S367_M_총괄_MATCH_이상 AND NOT 전체_M_이상_리셋), PT := T#500MS);
S367_M_총괄_MATCH_이상 := INST16.Q;
(* Rung L62 *)
INST17(IN := _OFF OR (S367_M_총괄_ROBOT_이상 AND NOT 전체_M_이상_리셋), PT := T#500MS);
S367_M_총괄_ROBOT_이상 := INST17.Q;

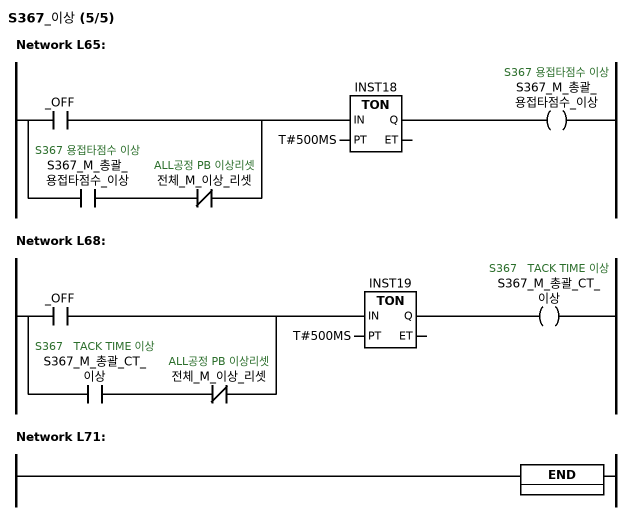
(* Rung L65 *)
INST18(IN := _OFF OR (S367_M_총괄_용접타점수_이상 AND NOT 전체_M_이상_리셋), PT := T#500MS);
S367_M_총괄_용접타점수_이상 := INST18.Q;
(* Rung L68 *)
INST19(IN := _OFF OR (S367_M_총괄_CT_이상 AND NOT 전체_M_이상_리셋), PT := T#500MS);
S367_M_총괄_CT_이상 := INST19.Q;
(* Rung L71 *)
END();
END_PROGRAM

PROGRAM S368_유틸리티 (* task: 스캔 프로그램 *)
VAR_EXTERNAL
    EGIS_CWS : BOOL;
    HOP_PBL_365_8_자동_운전 : BOOL; (* AT %MW87500.7 *) (* HOP_PBL_365_8_자동_운전 *)
    HOP_PBL_운전준비_ON : BOOL; (* AT %MW87500.0 *) (* HOP_PBL_운전준비_ON *)
    HOP_SSP_365_8_수동_선택 : BOOL; (* AT %MW87500.6 *) (* HOP_SSP_365_8_수동_선택 *)
    HOP_SSP_365_8_자동_선택 : BOOL; (* AT %MW87500.5 *) (* HOP_SSP_365_8_자동_선택 *)
    MCP_PBL_365_8_자동_운전 : BOOL; (* AT %MW87630.7 *) (* MCP PBL 365~8 자동기동 *)
    MCP_PBL_운전준비_ON : BOOL; (* AT %MW87630.0 *) (* MCP_PBL_운전준비_ON *)
    MCP_SPB_작업완료_RESET : BOOL; (* AT %MW87631.6 *) (* MCP_SPB_작업완료_RESET *)
    MCP_SPB_작업완료_SET : BOOL; (* AT %MW87631.7 *) (* MCP_SPB_작업완료_SET *)
    MCP_SSP_365_8_수동_선택 : BOOL; (* AT %MW87630.5 *) (* MCP_SSP_365_8_수동_선택 *)
    MCP_SSP_365_8_자동_선택 : BOOL; (* AT %MW87630.6 *) (* MCP_SSP_365_8_자동_선택 *)
    R361_1_M_I_RB_5차_작업완료 : BOOL; (* AT %MW20011.6 *) (* R361_1_M_I_RB_5차_작업완료 *)
    R366_1_M_I_RB_간섭무_1 : BOOL; (* AT %MW20062.0 *) (* R366_1_M_I_RB_간섭무_1 *)
    R366_1_M_I_RB_원위치 : BOOL; (* AT %MW20060.3 *) (* R366_1_M_I_RB_원위치 *)
    R368_1_M_I_RB_1차_작업완료 : BOOL; (* AT %MW20071.2 *) (* R368_1_M_I_RB_1차_작업완료 *)
    R368_1_M_I_RB_2차_작업완료 : BOOL; (* AT %MW20071.3 *) (* R368_1_M_I_RB_2차_작업완료 *)
    R368_1_M_I_RB_간섭무_1 : BOOL; (* AT %MW20072.0 *) (* R368_1_M_I_RB_간섭무_1 *)
    R368_1_M_I_RB_원위치 : BOOL; (* AT %MW20070.3 *) (* R368_1_M_I_RB_원위치 *)
    R369_1_M_I_RB_2차_작업완료 : BOOL; (* AT %MW20081.3 *) (* R369_1_M_I_RB_2차_작업완료 *)
    R369_1_M_I_RB_3차_작업완료 : BOOL; (* AT %MW20081.4 *) (* R369_1_M_I_RB_3차_작업완료 *)
    R369_1_M_I_RB_간섭무_1 : BOOL; (* AT %MW20082.0 *) (* R369_1_M_I_RB_간섭무_1 *)
    R369_1_M_I_RB_원위치 : BOOL; (* AT %MW20080.3 *) (* R369_1_M_I_RB_원위치 *)
    S368_PRS_AX_LH_HANGER_CHECK : BOOL; (* AT %MW86312.2 *) (* S368_PRS_AX_LH_HANGER_CHECK *)
    S368_PRS_AX_LH_ROOF_FRT_CHECK : BOOL; (* AT %MW86312.0 *) (* S368_PRS_AX_LH_ROOF_FRT_CHECK *)
    S368_PRS_AX_LH_ROOF_RR_CHECK : BOOL; (* AT %MW86312.1 *) (* S368_PRS_AX_LH_ROOF_RR_CHECK *)
    S368_PRS_AX_RH_HANGER_CHECK : BOOL; (* AT %MW86302.2 *) (* S368_PRS_AX_RH_HANGER_CHECK *)
    S368_PRS_AX_RH_ROOF_FRT_CHECK : BOOL; (* AT %MW86302.0 *) (* S368_PRS_AX_RH_ROOF_FRT_CHECK *)
    S368_PRS_AX_RH_ROOF_RR_CHECK : BOOL; (* AT %MW86302.1 *) (* S368_PRS_AX_RH_ROOF_RR_CHECK *)
END_VAR
VAR_EXTERNAL RETAIN
    HMI_M_선택_MOD_S367 : BOOL; (* AT %MW6.5 *) (* HMI M 선택 MOD S367 *)
    HMI_M_선택_MOD_S368 : BOOL; (* AT %MW6.6 *) (* HMI M 선택 MOD S368 *)
    S362_M_총괄_이상 : BOOL; (* AT %MW1009.0 *) (* S362_M_총괄_이상 *)
    S367_M_공정_차종_무 : BOOL; (* AT %MW3502.1 *) (* S367_M_공정_차종_무 *)
    S367_M_공정_차종_유 : BOOL; (* AT %MW3502.0 *) (* S367_M_공정_차종_유 *)
    S367_M_작업완료_SET_PLS : BOOL; (* AT %MW3500.8 *) (* S367 M 작업완료 SET PLS *)
    S367_M_작업완료_리셋_PLS : BOOL; (* AT %MW3500.9 *) (* S367 M 작업완료 리셋 PLS *)
    S368_M_BYPASS_보조 : BOOL; (* AT %MW4003.15 *) (* S368 M BYPASS 보조 *)
    S368_M_HANGER_CLP_전진단 : BOOL; (* AT %MW4111.3 *) (* S368_M_HANGER_CLP_전진단 *)
    S368_M_HANGER_CLP_후진단 : BOOL; (* AT %MW4111.4 *) (* S368_M_HANGER_CLP_후진단 *)
    S368_M_HANGER_급전급기_전진단 : BOOL; (* AT %MW4103.3 *)
    S368_M_HANGER_급전급기_후진단 : BOOL; (* AT %MW4103.4 *)
    S368_M_LH_AX_CLAMP_전진단 : BOOL; (* AT %MW4102.3 *) (* S368_M_LH_AX_CLAMP_전진단 *)
    S368_M_LH_AX_CLAMP_후진단 : BOOL; (* AT %MW4102.4 *) (* S368_M_LH_AX_CLAMP_후진단 *)
    S368_M_LH_AX_LATCH_전진단 : BOOL; (* AT %MW4100.3 *) (* S368_M_LH_AX_LATCH_전진단 *)
    S368_M_LH_AX_SR_LAT_전진단 : BOOL; (* AT %MW4101.3 *) (* S368_M_LH_AX_SR_LAT_전진단 *)
    S368_M_R368_1_해밍가능 : BOOL; (* AT %MW4004.10 *)
    S368_M_R368_1_행거안착가능 : BOOL; (* AT %MW4004.9 *)
    S368_M_R368_1_행거안착완료 : BOOL; (* AT %MW4001.2 *)
    S368_M_R368_1_헤밍완료 : BOOL; (* AT %MW4001.3 *)
    S368_M_R369_1_안착가능 : BOOL; (* AT %MW4004.8 *)
    S368_M_R369_1_안착완료 : BOOL; (* AT %MW4001.1 *)
    S368_M_R369_1_언로딩완료 : BOOL; (* AT %MW4001.4 *)
    S368_M_RH_AX_CLAMP_전진단 : BOOL; (* AT %MW4110.3 *) (* S368_M_RH_AX_CLAMP_전진단 *)
    S368_M_RH_AX_CLAMP_후진단 : BOOL; (* AT %MW4110.4 *) (* S368_M_RH_AX_CLAMP_후진단 *)
    S368_M_RH_AX_LATCH_전진단 : BOOL; (* AT %MW4108.3 *) (* S368_M_RH_AX_LATCH_전진단 *)
    S368_M_RH_AX_SR_LAT_전진단 : BOOL; (* AT %MW4109.3 *) (* S368_M_RH_AX_SR_LAT_전진단 *)
    S368_M_SEQ : WORD; (* AT %MW10200 *) (* S368 M SEQ *)
    S368_M_공정_FRT_제품감지_무 : BOOL; (* AT %MW4001.8 *)
    S368_M_공정_FRT_제품감지_유 : BOOL; (* AT %MW4001.7 *)
    S368_M_공정_HANGER_감지_무 : BOOL; (* AT %MW4001.12 *)
    S368_M_공정_HANGER_감지_유 : BOOL; (* AT %MW4001.11 *)
    S368_M_공정_RR_제품감지_무 : BOOL; (* AT %MW4001.10 *)
    S368_M_공정_RR_제품감지_유 : BOOL; (* AT %MW4001.9 *)
    S368_M_공정_불간섭 : BOOL; (* AT %MW4004.1 *) (* S368_M_공정_불간섭 *)
    S368_M_공정_원위치 : BOOL; (* AT %MW4004.0 *) (* S368_M_공정_원위치 *)
    S368_M_공정_제품감지_무 : BOOL; (* AT %MW4001.6 *) (* S368_M_공정_제품감지_무 *)
    S368_M_공정_제품감지_유 : BOOL; (* AT %MW4001.5 *) (* S368_M_공정_제품감지_유 *)
    S368_M_공정_차종_무 : BOOL; (* AT %MW4002.1 *) (* S368_M_공정_차종_무 *)
    S368_M_공정_차종_유 : BOOL; (* AT %MW4002.0 *) (* S368_M_공정_차종_유 *)
    S368_M_수동모드 : BOOL; (* AT %MW4000.3 *) (* S368 선택 수동모드 *)
    S368_M_운전준비_ON : BOOL; (* AT %MW4000.0 *) (* S368 운전준비 ON *)
    S368_M_자동_START : BOOL; (* AT %MW4000.5 *) (* S368 자동운전중 *)
    S368_M_자동_운전중 : BOOL; (* AT %MW4000.4 *) (* S368 자동운전중 *)
    S368_M_자동모드 : BOOL; (* AT %MW4000.1 *) (* S368 선택 자동모드 *)
    S368_M_작업_완료 : BOOL; (* AT %MW4001.0 *) (* S368_M_작업_완료 *)
    S368_M_작업완료_SET_PLS : BOOL; (* AT %MW4000.8 *) (* S368 M 작업완료 SET PLS *)
    S368_M_작업완료_리셋_PLS : BOOL; (* AT %MW4000.9 *) (* S368 M 작업완료 리셋 PLS *)
    S368_M_차종1_AX : BOOL; (* AT %MW10201.0 *) (* S368 M 차종1 AX *)
    S368_M_차종1_B : BOOL; (* AT %MW10201.1 *) (* S368 M 차종1 B *)
    S368_M_차종1_C : BOOL; (* AT %MW10201.2 *) (* S368 M 차종1 C *)
    S368_M_차종1_D : BOOL; (* AT %MW10201.3 *) (* S368 M 차종1 D *)
    S368_M_차종1_E : BOOL; (* AT %MW10201.4 *) (* S368 M 차종1 E *)
    S368_M_차종1_F : BOOL; (* AT %MW10201.5 *) (* S368 M 차종1 F *)
    S368_M_차종1_G : BOOL; (* AT %MW10201.6 *) (* S368 M 차종1 G *)
    S368_M_차종1_H : BOOL; (* AT %MW10201.7 *) (* S368 M 차종1 H *)
    S368_M_차종2_3DR : BOOL; (* AT %MW10201.8 *) (* S368 M 차종2 3DR *)
    S368_M_차종2_4DR : BOOL; (* AT %MW10201.9 *) (* S368 M 차종2 4DR *)
    S368_M_차종2_5DR : BOOL; (* AT %MW10201.10 *) (* S368 M 차종2 5DR *)
    S368_M_차종2_SP1 : BOOL; (* AT %MW10201.12 *) (* S368 M 차종2 SP1 *)
    S368_M_차종2_SP2 : BOOL; (* AT %MW10201.13 *) (* S368 M 차종2 SP2 *)
    S368_M_차종2_WGN : BOOL; (* AT %MW10201.11 *) (* S368 M 차종2 WGN *)
    S368_M_차종3_LHD : BOOL; (* AT %MW10201.14 *) (* S368 M 차종3 LHD *)
    S368_M_차종3_RHD : BOOL; (* AT %MW10201.15 *) (* S368 M 차종3 RHD *)
    S368_M_차종4_EEC : BOOL; (* AT %MW10202.3 *) (* S368 M 차종4 EEC *)
    S368_M_차종4_SP1 : BOOL; (* AT %MW10202.8 *) (* S368 M 차종4 SP1 *)
    S368_M_차종4_SP2 : BOOL; (* AT %MW10202.9 *) (* S368 M 차종4 SP2 *)
    S368_M_차종4_SP3 : BOOL; (* AT %MW10202.11 *) (* S368 M 차종4 SP3 *)
    S368_M_차종4_SP4 : BOOL; (* AT %MW10202.12 *) (* S368 M 차종4 SP4 *)
    S368_M_차종4_SP5 : BOOL; (* AT %MW10202.13 *) (* S368 M 차종4 SP5 *)
    S368_M_차종4_SP6 : BOOL; (* AT %MW10202.14 *) (* S368 M 차종4 SP6 *)
    S368_M_차종4_SP7 : BOOL; (* AT %MW10202.15 *) (* S368 M 차종4 SP7 *)
    S368_M_차종4_내수 : BOOL; (* AT %MW10202.0 *) (* S368 M 차종4 내수 *)
    S368_M_차종4_러시아 : BOOL; (* AT %MW10202.10 *) (* S368 M 차종4 러시아 *)
    S368_M_차종4_북미 : BOOL; (* AT %MW10202.2 *) (* S368 M 차종4 북미 *)
    S368_M_차종4_브라질 : BOOL; (* AT %MW10202.7 *) (* S368 M 차종4 브라질 *)
    S368_M_차종4_수출 : BOOL; (* AT %MW10202.1 *) (* S368 M 차종4 수출 *)
    S368_M_차종4_중국 : BOOL; (* AT %MW10202.6 *) (* S368 M 차종4 중국 *)
    S368_M_차종4_중동 : BOOL; (* AT %MW10202.5 *) (* S368 M 차종4 중동 *)
    S368_M_차종4_호주 : BOOL; (* AT %MW10202.4 *) (* S368 M 차종4 호주 *)
    S368_M_차종5_AT : BOOL; (* AT %MW10203.1 *) (* S368 M 차종5 AT *)
    S368_M_차종5_MT : BOOL; (* AT %MW10203.0 *) (* S368 M 차종5 MT *)
    S368_M_차종5_SP1 : BOOL; (* AT %MW10203.2 *) (* S368 M 차종5 SP1 *)
    S368_M_차종6_DSROOF : BOOL; (* AT %MW10203.6 *) (* S368 M 차종6 DSROOF *)
    S368_M_차종6_SP1 : BOOL; (* AT %MW10203.7 *) (* S368 M 차종6 SP1 *)
    S368_M_차종6_썬루프 : BOOL; (* AT %MW10203.4 *) (* S368 M 차종6 썬루프 *)
    S368_M_차종6_일반루프 : BOOL; (* AT %MW10203.3 *) (* S368 M 차종6 일반루프 *)
    S368_M_차종6_파노라마루프 : BOOL; (* AT %MW10203.5 *) (* S368 M 차종6 파노라마루프 *)
    S368_M_차종7_DSL : BOOL; (* AT %MW10203.9 *) (* S368 M 차종7 DSL *)
    S368_M_차종7_GSL : BOOL; (* AT %MW10203.8 *) (* S368 M 차종7 GSL *)
    S368_M_차종7_SP1 : BOOL; (* AT %MW10203.10 *) (* S368 M 차종7 SP1 *)
    S368_M_차종7_SP2 : BOOL; (* AT %MW10203.11 *) (* S368 M 차종7 SP2 *)
    S368_M_차종7_SP3 : BOOL; (* AT %MW10203.12 *) (* S368 M 차종7 SP3 *)
    S368_M_차종7_SP4 : BOOL; (* AT %MW10203.13 *) (* S368 M 차종7 SP4 *)
    S368_M_차종7_SP5 : BOOL; (* AT %MW10203.14 *) (* S368 M 차종7 SP5 *)
    S368_M_차종7_SP6 : BOOL; (* AT %MW10203.15 *) (* S368 M 차종7 SP6 *)
    S368_M_차종8_2WD : BOOL; (* AT %MW10204.0 *) (* S368 M 차종8 2WD *)
    S368_M_차종8_4WD : BOOL; (* AT %MW10204.1 *) (* S368 M 차종8 4WD *)
    S368_M_차종8_SP1 : BOOL; (* AT %MW10204.2 *) (* S368 M 차종8 SP1 *)
    S368_M_차종9_MPI : BOOL; (* AT %MW10204.3 *) (* S368 M 차종9 MPI *)
    S368_M_차종9_SP1 : BOOL; (* AT %MW10204.5 *) (* S368 M 차종9 SP1 *)
    S368_M_차종9_SP10 : BOOL; (* AT %MW10204.14 *) (* S368 M 차종9 SP10 *)
    S368_M_차종9_SP11 : BOOL; (* AT %MW10204.15 *) (* S368 M 차종9 SP11 *)
    S368_M_차종9_SP2 : BOOL; (* AT %MW10204.6 *) (* S368 M 차종9 SP2 *)
    S368_M_차종9_SP3 : BOOL; (* AT %MW10204.7 *) (* S368 M 차종9 SP3 *)
    S368_M_차종9_SP4 : BOOL; (* AT %MW10204.8 *) (* S368 M 차종9 SP4 *)
    S368_M_차종9_SP5 : BOOL; (* AT %MW10204.9 *) (* S368 M 차종9 SP5 *)
    S368_M_차종9_SP6 : BOOL; (* AT %MW10204.10 *) (* S368 M 차종9 SP6 *)
    S368_M_차종9_SP7 : BOOL; (* AT %MW10204.11 *) (* S368 M 차종9 SP7 *)
    S368_M_차종9_SP8 : BOOL; (* AT %MW10204.12 *) (* S368 M 차종9 SP8 *)
    S368_M_차종9_SP9 : BOOL; (* AT %MW10204.13 *) (* S368 M 차종9 SP9 *)
    S368_M_차종9_T_GDI : BOOL; (* AT %MW10204.4 *) (* S368 M 차종9 T GDI *)
    S368_M_차종_OPT1_R_RACK_무 : BOOL; (* AT %MW10205.3 *) (* S368 M 차종 OPT1 R RACK 무 *)
    S368_M_차종_OPT1_R_RACK_유 : BOOL; (* AT %MW10205.2 *) (* S368 M 차종 OPT1 R RACK 유 *)
    S368_M_차종_OPT1_S_REP_EATER_무 : BOOL; (* AT %MW10205.7 *) (* S368 M 차종 OPT1 S REP EATER 무 *)
    S368_M_차종_OPT1_S_REP_EATER_유 : BOOL; (* AT %MW10205.6 *) (* S368 M 차종 OPT1 S REP EATER 유 *)
    S368_M_차종_OPT1_VAN_무 : BOOL; (* AT %MW10205.9 *) (* S368 M 차종 OPT1 VAN 무 *)
    S368_M_차종_OPT1_VAN_유 : BOOL; (* AT %MW10205.8 *) (* S368 M 차종 OPT1 VAN 유 *)
    S368_M_차종_OPT1_슬라이딩_무 : BOOL; (* AT %MW10205.1 *) (* S368 M 차종 OPT1 슬라이딩 무 *)
    S368_M_차종_OPT1_슬라이딩_유 : BOOL; (* AT %MW10205.0 *) (* S368 M 차종 OPT1 슬라이딩 유 *)
    S368_M_차종_OPT1_폴딩_무 : BOOL; (* AT %MW10205.5 *) (* S368 M 차종 OPT1 폴딩 무 *)
    S368_M_차종_OPT1_폴딩_유 : BOOL; (* AT %MW10205.4 *) (* S368 M 차종 OPT1 폴딩 유 *)
    S368_M_차종_공대차 : BOOL; (* AT %MW10210.12 *) (* S368 M 차종 공대차 *)
    S368_M_차종_공차 : BOOL; (* AT %MW10210.10 *) (* S368 M 차종 공차 *)
    S368_M_차종_불량차 : BOOL; (* AT %MW10210.11 *) (* S368 M 차종 불량차 *)
    S368_M_총괄_이상 : BOOL; (* AT %MW4009.0 *) (* S368_M_총괄_이상 *)
    전체_M_GATE_자동기동 : BOOL; (* AT %MW308.1 *) (* 전체_M_자동_운전 *)
    전체_라인_M_총괄_SAFETY_이상 : BOOL; (* AT %MW300.2 *) (* ALL공정 SAFETY  이상총괄 *)
    전체_라인_M_총괄_공기압_이상 : BOOL; (* AT %MW300.3 *) (* ALL공정 공기압 이상총괄 *)
    전체_라인_M_총괄_비상정지_이상 : BOOL; (* AT %MW300.1 *) (* ALL공정 비상정지 이상총괄 *)
    전체_라인_M_총괄_이상 : BOOL; (* AT %MW300.0 *) (* ALL공정 총괄이상 *)
END_VAR
VAR
    S368_READY : TON;
    T368_AUTO : TON;
END_VAR
VAR
    _t1 : BOOL;
END_VAR

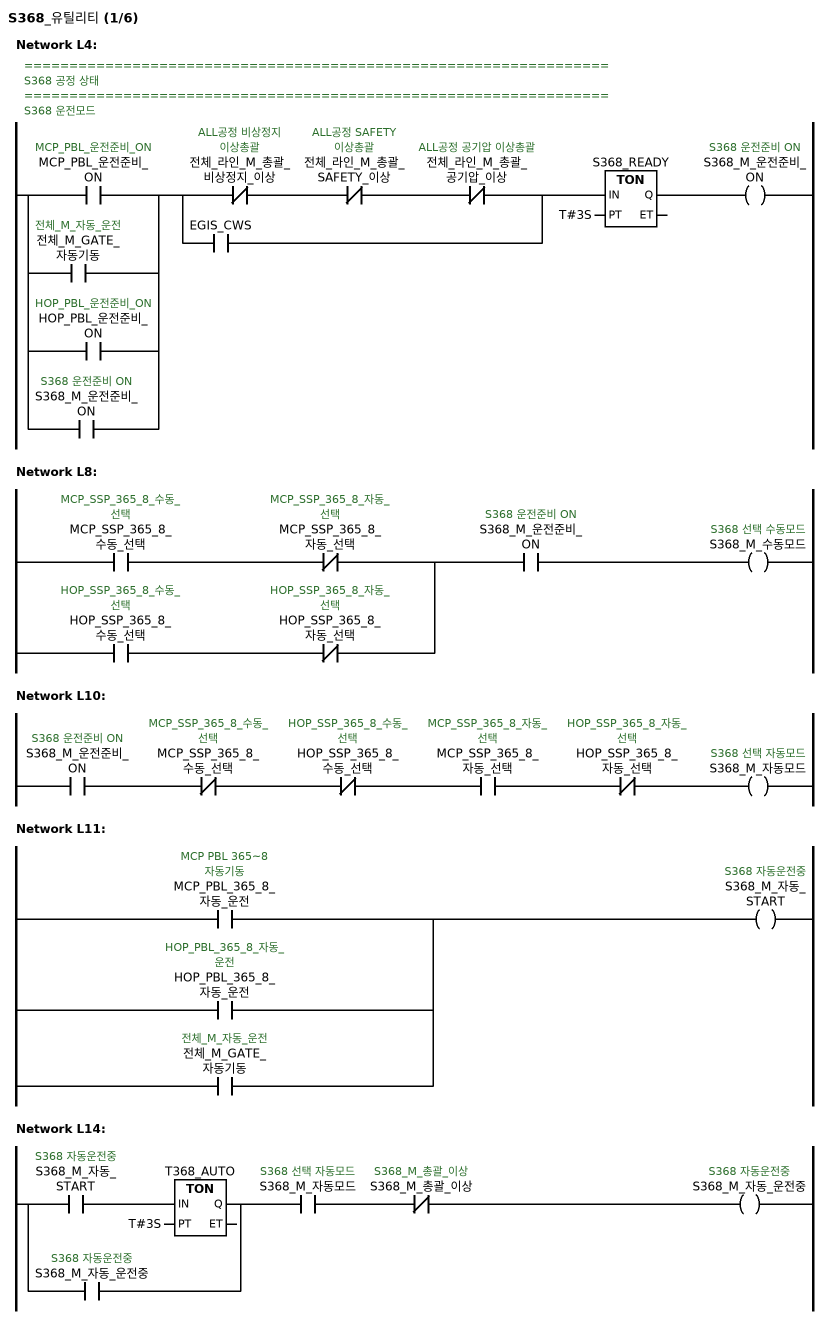
(* ================================================================= *)
(* S368 공정 상태 *)
(* ================================================================= *)
(* S368 운전모드 *)
(* Rung L4 *)
S368_READY(IN := (MCP_PBL_운전준비_ON OR 전체_M_GATE_자동기동 OR HOP_PBL_운전준비_ON OR S368_M_운전준비_ON) AND ((NOT 전체_라인_M_총괄_비상정지_이상 AND NOT 전체_라인_M_총괄_SAFETY_이상 AND NOT 전체_라인_M_총괄_공기압_이상) OR EGIS_CWS), PT := T#3S);
S368_M_운전준비_ON := S368_READY.Q;
(* Rung L8 *)
S368_M_수동모드 := ((MCP_SSP_365_8_수동_선택 AND NOT MCP_SSP_365_8_자동_선택) OR (HOP_SSP_365_8_수동_선택 AND NOT HOP_SSP_365_8_자동_선택)) AND S368_M_운전준비_ON;
(* Rung L10 *)
S368_M_자동모드 := S368_M_운전준비_ON AND NOT MCP_SSP_365_8_수동_선택 AND NOT HOP_SSP_365_8_수동_선택 AND MCP_SSP_365_8_자동_선택 AND NOT HOP_SSP_365_8_자동_선택;
(* Rung L11 *)
S368_M_자동_START := MCP_PBL_365_8_자동_운전 OR HOP_PBL_365_8_자동_운전 OR 전체_M_GATE_자동기동;
(* Rung L14 *)
T368_AUTO(IN := S368_M_자동_START, PT := T#3S);
S368_M_자동_운전중 := (T368_AUTO.Q OR S368_M_자동_운전중) AND S368_M_자동모드 AND NOT S368_M_총괄_이상;

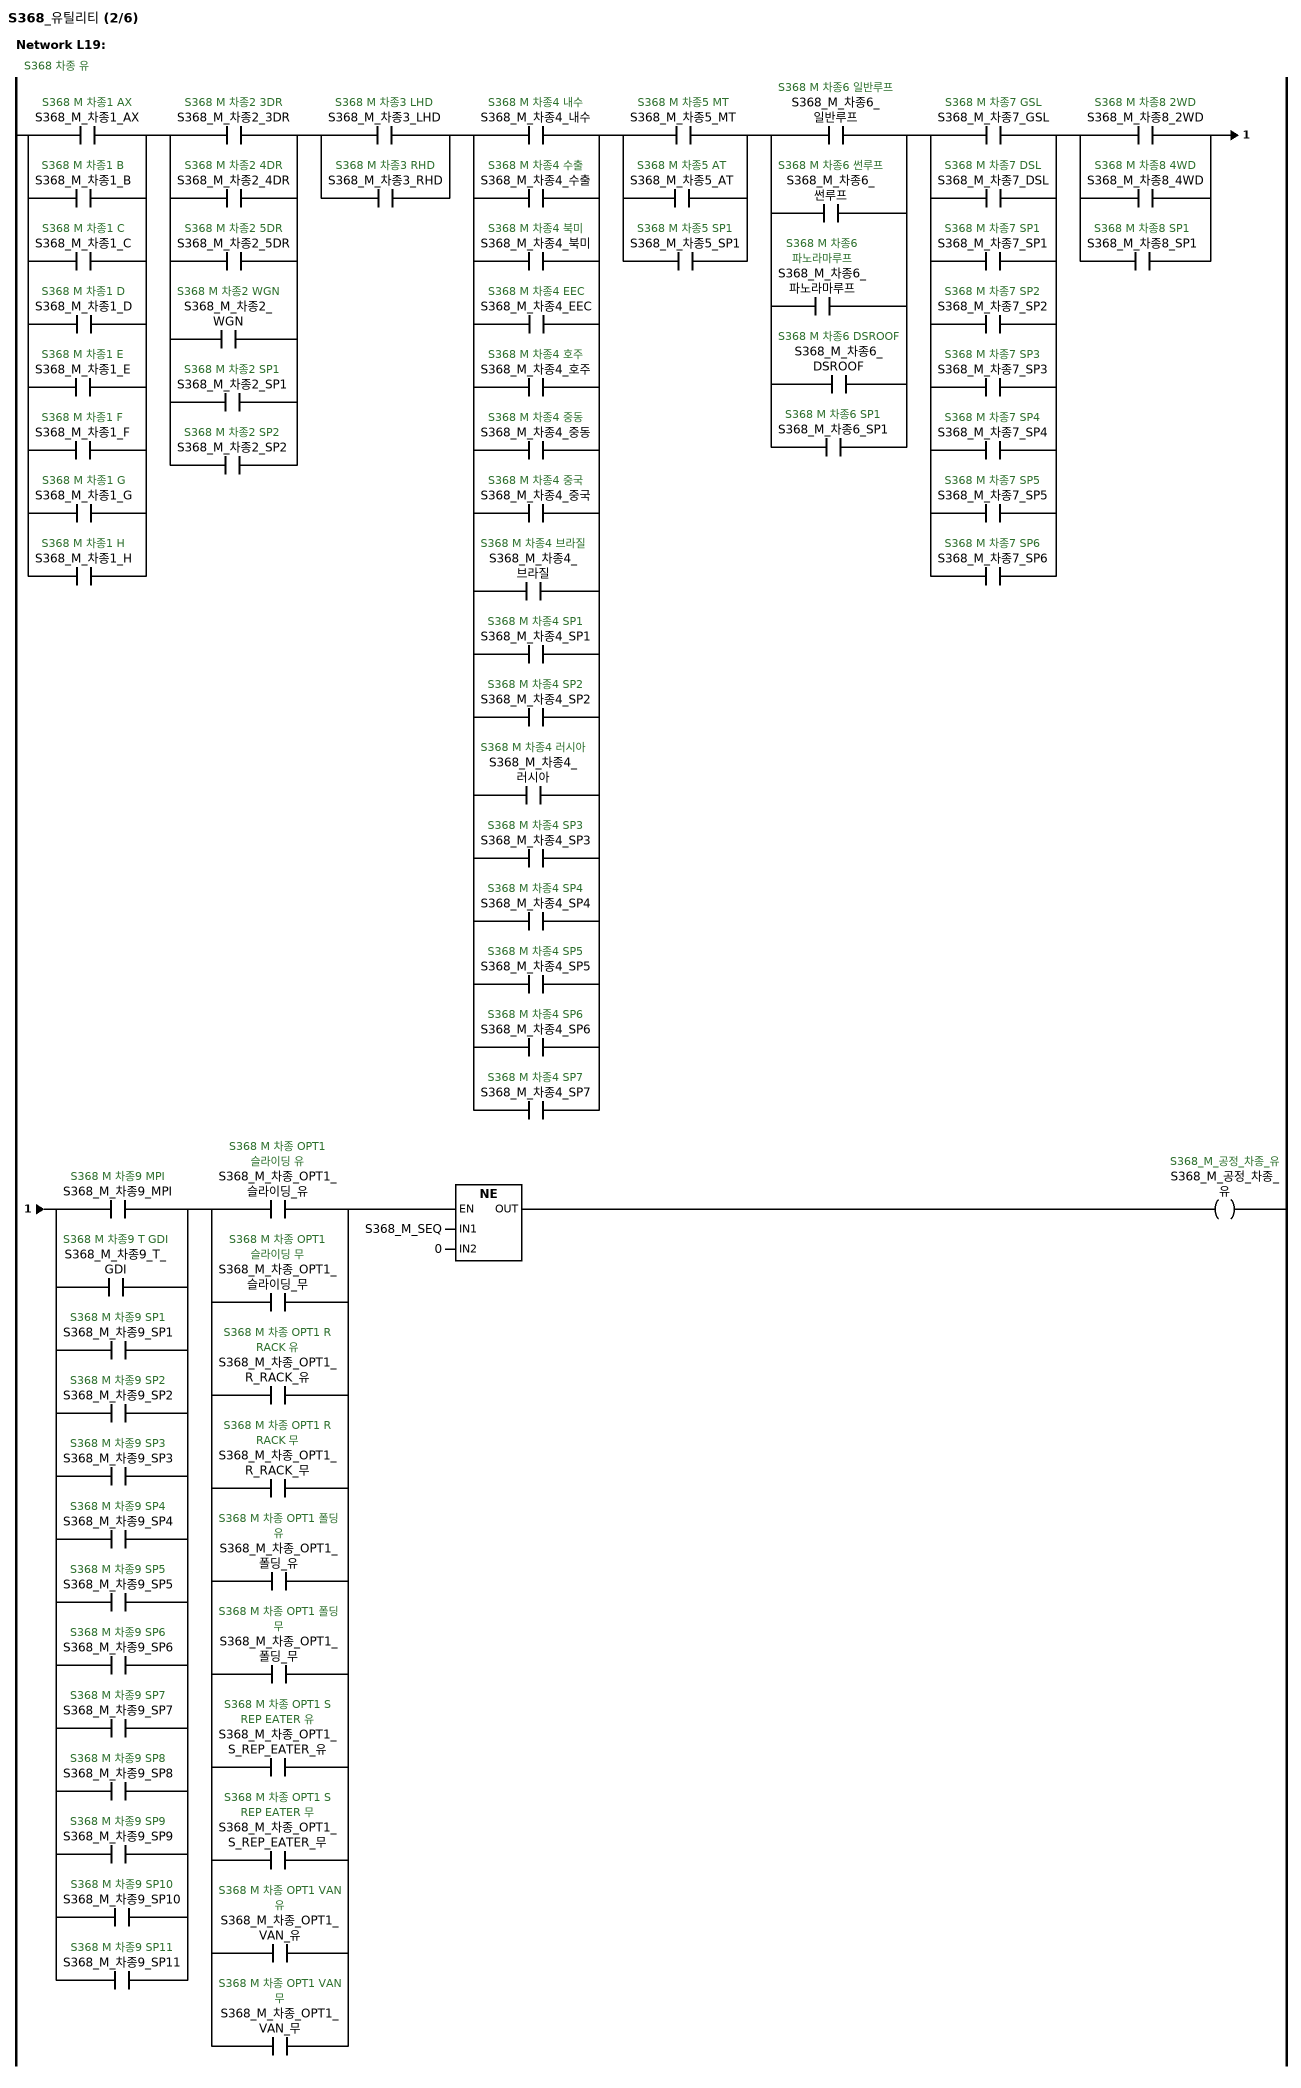
(* S368 차종 유 *)
(* Rung L19 *)
IF (S368_M_차종1_AX OR S368_M_차종1_B OR S368_M_차종1_C OR S368_M_차종1_D OR S368_M_차종1_E OR S368_M_차종1_F OR S368_M_차종1_G OR S368_M_차종1_H) AND (S368_M_차종2_3DR OR S368_M_차종2_4DR OR S368_M_차종2_5DR OR S368_M_차종2_WGN OR S368_M_차종2_SP1 OR S368_M_차종2_SP2) AND (S368_M_차종3_LHD OR S368_M_차종3_RHD) AND (S368_M_차종4_내수 OR S368_M_차종4_수출 OR S368_M_차종4_북미 OR S368_M_차종4_EEC OR S368_M_차종4_호주 OR S368_M_차종4_중동 OR S368_M_차종4_중국 OR S368_M_차종4_브라질 OR S368_M_차종4_SP1 OR S368_M_차종4_SP2 OR S368_M_차종4_러시아 OR S368_M_차종4_SP3 OR S368_M_차종4_SP4 OR S368_M_차종4_SP5 OR S368_M_차종4_SP6 OR S368_M_차종4_SP7) AND (S368_M_차종5_MT OR S368_M_차종5_AT OR S368_M_차종5_SP1) AND (S368_M_차종6_일반루프 OR S368_M_차종6_썬루프 OR S368_M_차종6_파노라마루프 OR S368_M_차종6_DSROOF OR S368_M_차종6_SP1) AND (S368_M_차종7_GSL OR S368_M_차종7_DSL OR S368_M_차종7_SP1 OR S368_M_차종7_SP2 OR S368_M_차종7_SP3 OR S368_M_차종7_SP4 OR S368_M_차종7_SP5 OR S368_M_차종7_SP6) AND (S368_M_차종8_2WD OR S368_M_차종8_4WD OR S368_M_차종8_SP1) AND (S368_M_차종9_MPI OR S368_M_차종9_T_GDI OR S368_M_차종9_SP1 OR S368_M_차종9_SP2 OR S368_M_차종9_SP3 OR S368_M_차종9_SP4 OR S368_M_차종9_SP5 OR S368_M_차종9_SP6 OR S368_M_차종9_SP7 OR S368_M_차종9_SP8 OR S368_M_차종9_SP9 OR S368_M_차종9_SP10 OR S368_M_차종9_SP11) AND (S368_M_차종_OPT1_슬라이딩_유 OR S368_M_차종_OPT1_슬라이딩_무 OR S368_M_차종_OPT1_R_RACK_유 OR S368_M_차종_OPT1_R_RACK_무 OR S368_M_차종_OPT1_폴딩_유 OR S368_M_차종_OPT1_폴딩_무 OR S368_M_차종_OPT1_S_REP_EATER_유 OR S368_M_차종_OPT1_S_REP_EATER_무 OR S368_M_차종_OPT1_VAN_유 OR S368_M_차종_OPT1_VAN_무) THEN
    _t1 := S368_M_SEQ <> 0;
END_IF;
S368_M_공정_차종_유 := _t1;

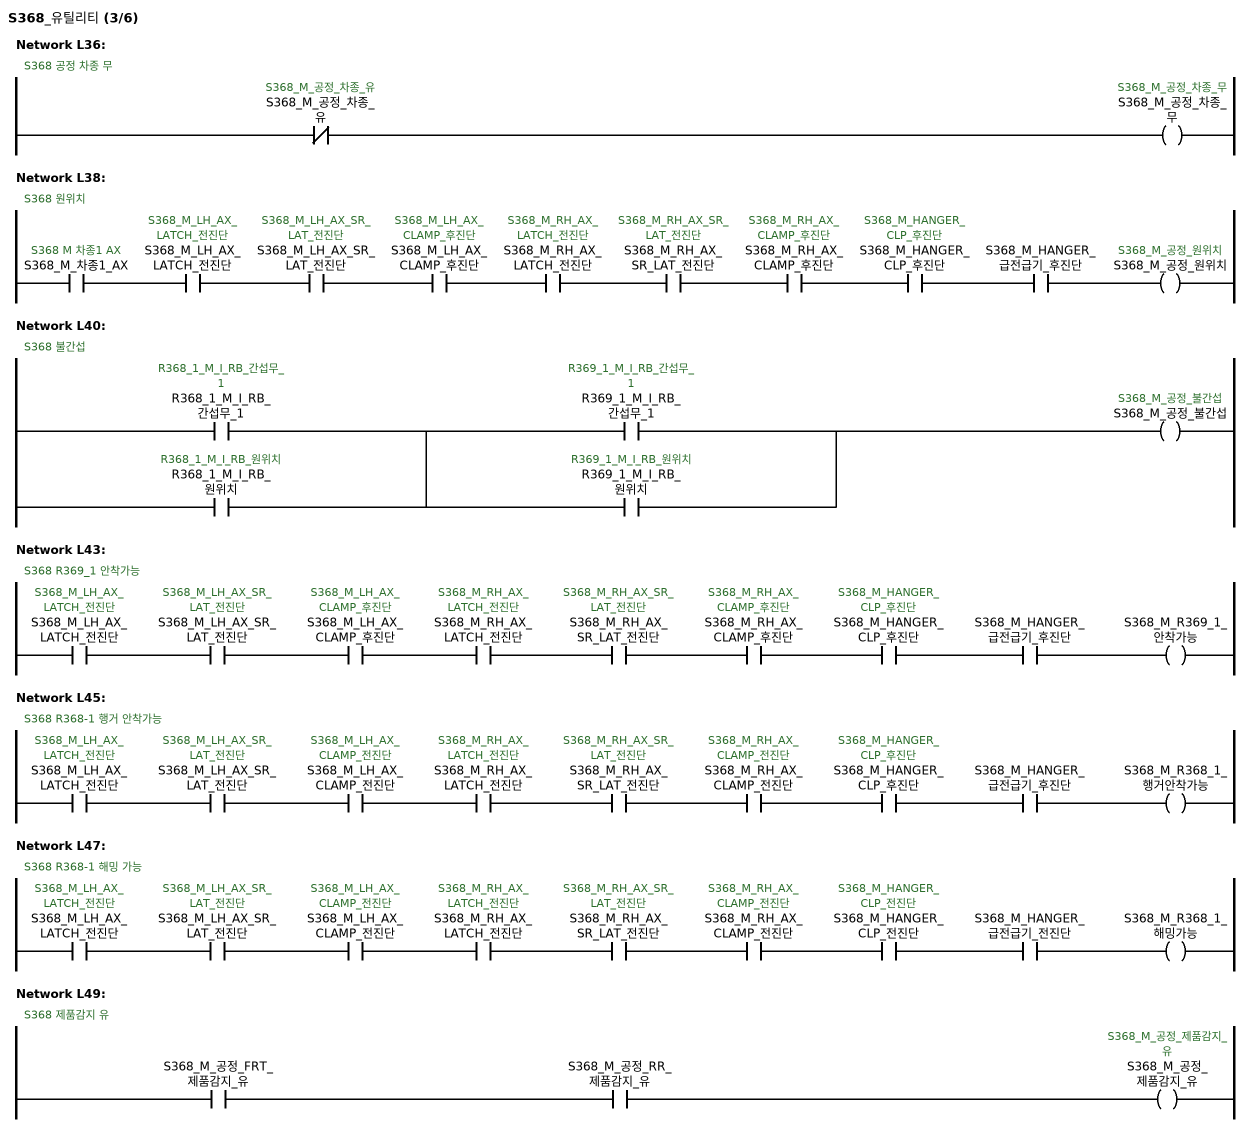
(* S368 공정 차종 무 *)
(* Rung L36 *)
S368_M_공정_차종_무 := NOT S368_M_공정_차종_유;
(* S368 원위치 *)
(* Rung L38 *)
S368_M_공정_원위치 := S368_M_차종1_AX AND S368_M_LH_AX_LATCH_전진단 AND S368_M_LH_AX_SR_LAT_전진단 AND S368_M_LH_AX_CLAMP_후진단 AND S368_M_RH_AX_LATCH_전진단 AND S368_M_RH_AX_SR_LAT_전진단 AND S368_M_RH_AX_CLAMP_후진단 AND S368_M_HANGER_CLP_후진단 AND S368_M_HANGER_급전급기_후진단;
(* S368 불간섭 *)
(* Rung L40 *)
S368_M_공정_불간섭 := (R368_1_M_I_RB_간섭무_1 OR R368_1_M_I_RB_원위치) AND (R369_1_M_I_RB_간섭무_1 OR R369_1_M_I_RB_원위치);
(* S368 R369_1 안착가능 *)
(* Rung L43 *)
S368_M_R369_1_안착가능 := S368_M_LH_AX_LATCH_전진단 AND S368_M_LH_AX_SR_LAT_전진단 AND S368_M_LH_AX_CLAMP_후진단 AND S368_M_RH_AX_LATCH_전진단 AND S368_M_RH_AX_SR_LAT_전진단 AND S368_M_RH_AX_CLAMP_후진단 AND S368_M_HANGER_CLP_후진단 AND S368_M_HANGER_급전급기_후진단;
(* S368 R368-1 행거 안착가능 *)
(* Rung L45 *)
S368_M_R368_1_행거안착가능 := S368_M_LH_AX_LATCH_전진단 AND S368_M_LH_AX_SR_LAT_전진단 AND S368_M_LH_AX_CLAMP_전진단 AND S368_M_RH_AX_LATCH_전진단 AND S368_M_RH_AX_SR_LAT_전진단 AND S368_M_RH_AX_CLAMP_전진단 AND S368_M_HANGER_CLP_후진단 AND S368_M_HANGER_급전급기_후진단;
(* S368 R368-1 해밍 가능 *)
(* Rung L47 *)
S368_M_R368_1_해밍가능 := S368_M_LH_AX_LATCH_전진단 AND S368_M_LH_AX_SR_LAT_전진단 AND S368_M_LH_AX_CLAMP_전진단 AND S368_M_RH_AX_LATCH_전진단 AND S368_M_RH_AX_SR_LAT_전진단 AND S368_M_RH_AX_CLAMP_전진단 AND S368_M_HANGER_CLP_전진단 AND S368_M_HANGER_급전급기_전진단;
(* S368 제품감지 유 *)
(* Rung L49 *)
S368_M_공정_제품감지_유 := S368_M_공정_FRT_제품감지_유 AND S368_M_공정_RR_제품감지_유;

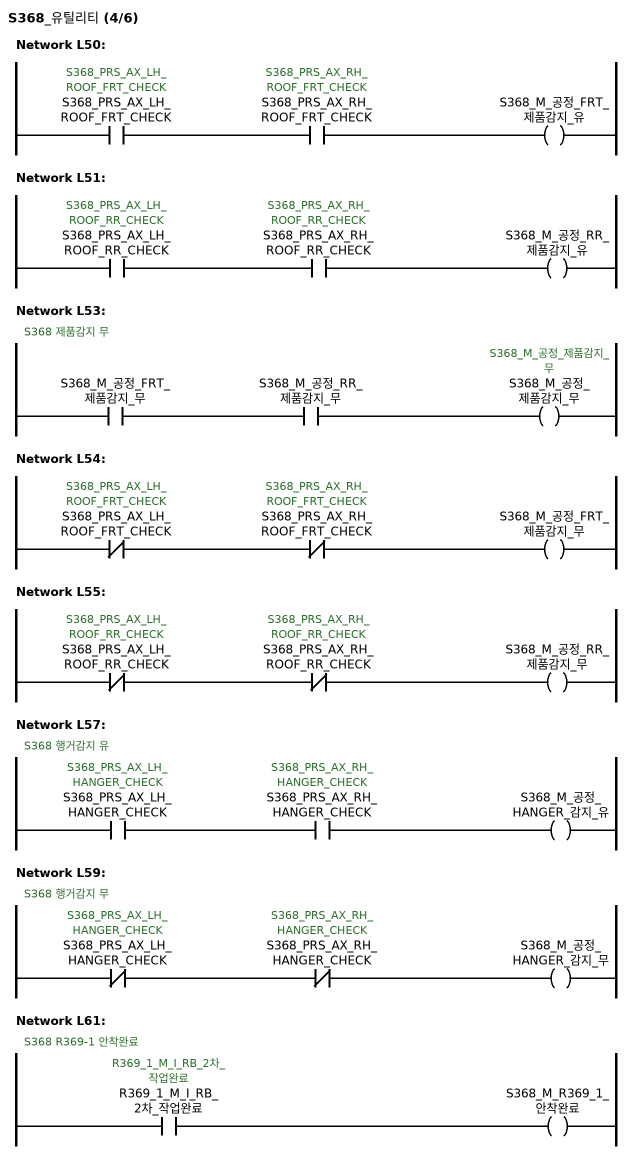
(* Rung L50 *)
S368_M_공정_FRT_제품감지_유 := S368_PRS_AX_LH_ROOF_FRT_CHECK AND S368_PRS_AX_RH_ROOF_FRT_CHECK;
(* Rung L51 *)
S368_M_공정_RR_제품감지_유 := S368_PRS_AX_LH_ROOF_RR_CHECK AND S368_PRS_AX_RH_ROOF_RR_CHECK;
(* S368 제품감지 무 *)
(* Rung L53 *)
S368_M_공정_제품감지_무 := S368_M_공정_FRT_제품감지_무 AND S368_M_공정_RR_제품감지_무;
(* Rung L54 *)
S368_M_공정_FRT_제품감지_무 := NOT S368_PRS_AX_LH_ROOF_FRT_CHECK AND NOT S368_PRS_AX_RH_ROOF_FRT_CHECK;
(* Rung L55 *)
S368_M_공정_RR_제품감지_무 := NOT S368_PRS_AX_LH_ROOF_RR_CHECK AND NOT S368_PRS_AX_RH_ROOF_RR_CHECK;
(* S368 행거감지 유 *)
(* Rung L57 *)
S368_M_공정_HANGER_감지_유 := S368_PRS_AX_LH_HANGER_CHECK AND S368_PRS_AX_RH_HANGER_CHECK;
(* S368 행거감지 무 *)
(* Rung L59 *)
S368_M_공정_HANGER_감지_무 := NOT S368_PRS_AX_LH_HANGER_CHECK AND NOT S368_PRS_AX_RH_HANGER_CHECK;
(* S368 R369-1 안착완료 *)
(* Rung L61 *)
S368_M_R369_1_안착완료 := R369_1_M_I_RB_2차_작업완료;

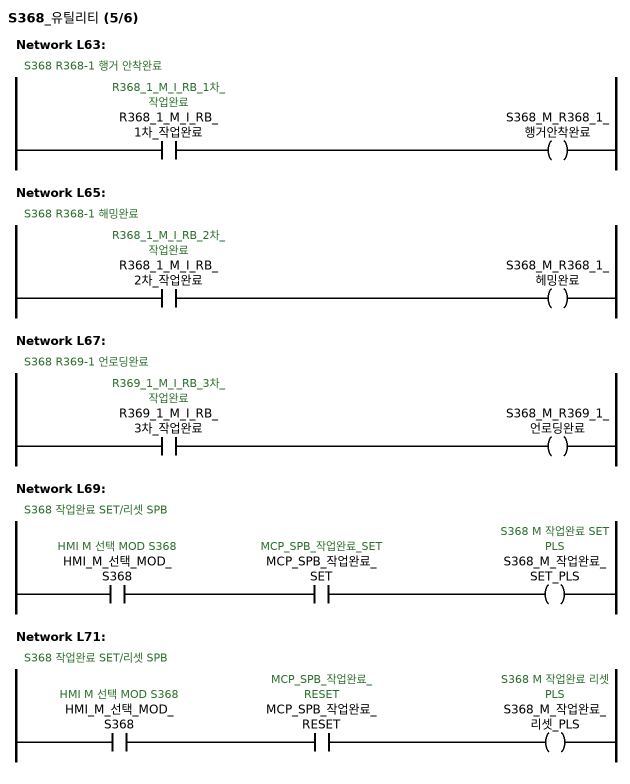
(* S368 R368-1 행거 안착완료 *)
(* Rung L63 *)
S368_M_R368_1_행거안착완료 := R368_1_M_I_RB_1차_작업완료;
(* S368 R368-1 해밍완료 *)
(* Rung L65 *)
S368_M_R368_1_헤밍완료 := R368_1_M_I_RB_2차_작업완료;
(* S368 R369-1 언로딩완료 *)
(* Rung L67 *)
S368_M_R369_1_언로딩완료 := R369_1_M_I_RB_3차_작업완료;
(* S368 작업완료 SET/리셋 SPB *)
(* Rung L69 *)
S368_M_작업완료_SET_PLS := HMI_M_선택_MOD_S368 AND MCP_SPB_작업완료_SET;
(* S368 작업완료 SET/리셋 SPB *)
(* Rung L71 *)
S368_M_작업완료_리셋_PLS := HMI_M_선택_MOD_S368 AND MCP_SPB_작업완료_RESET;

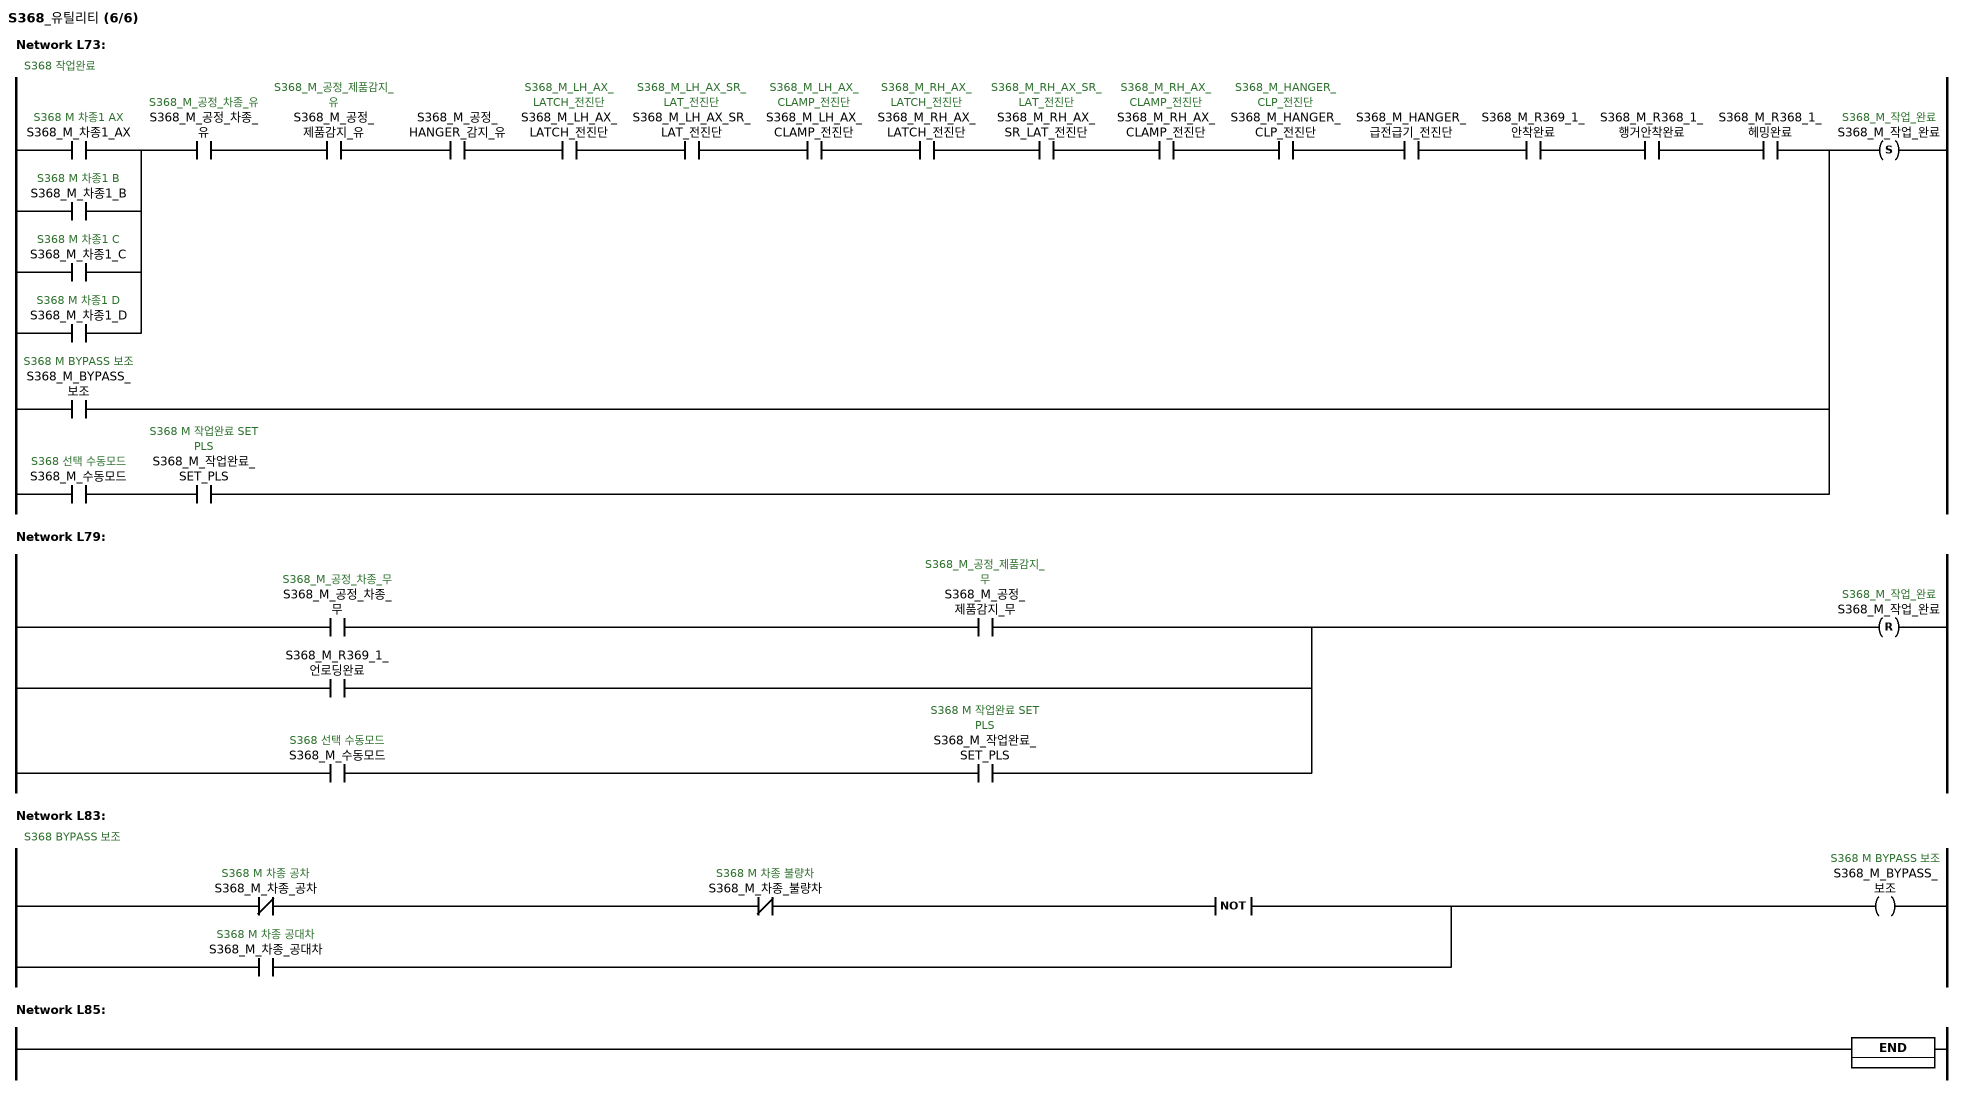
(* S368 작업완료 *)
(* Rung L73 *)
IF ((S368_M_차종1_AX OR S368_M_차종1_B OR S368_M_차종1_C OR S368_M_차종1_D) AND S368_M_공정_차종_유 AND S368_M_공정_제품감지_유 AND S368_M_공정_HANGER_감지_유 AND S368_M_LH_AX_LATCH_전진단 AND S368_M_LH_AX_SR_LAT_전진단 AND S368_M_LH_AX_CLAMP_전진단 AND S368_M_RH_AX_LATCH_전진단 AND S368_M_RH_AX_SR_LAT_전진단 AND S368_M_RH_AX_CLAMP_전진단 AND S368_M_HANGER_CLP_전진단 AND S368_M_HANGER_급전급기_전진단 AND S368_M_R369_1_안착완료 AND S368_M_R368_1_행거안착완료 AND S368_M_R368_1_헤밍완료) OR S368_M_BYPASS_보조 OR (S368_M_수동모드 AND S368_M_작업완료_SET_PLS) THEN
    S368_M_작업_완료 := TRUE;
END_IF;
(* Rung L79 *)
IF (S368_M_공정_차종_무 AND S368_M_공정_제품감지_무) OR S368_M_R369_1_언로딩완료 OR (S368_M_수동모드 AND S368_M_작업완료_SET_PLS) THEN
    S368_M_작업_완료 := FALSE;
END_IF;
(* S368 BYPASS 보조 *)
(* Rung L83 *)
S368_M_BYPASS_보조 := NOT (NOT S368_M_차종_공차 AND NOT S368_M_차종_불량차) OR S368_M_차종_공대차;
(* Rung L85 *)
END();
END_PROGRAM

PROGRAM S368_동작 (* task: 스캔 프로그램 *)
VAR_EXTERNAL RETAIN
    ALWAYS_ON : BOOL; (* AT %MW3.1 *) (* 항시 ON *)
    R361_1_M_차종_유 : BOOL; (* AT %MW1502.0 *)
    R369_1_M_차종1_AX : BOOL; (* AT %MW10061.0 *) (* R369 1 M 차종1 AX *)
    R369_1_M_차종_유 : BOOL; (* AT %MW4502.2 *)
    S367_M_R361_1_로딩완료 : BOOL; (* AT %MW3501.1 *)
    S367_M_공정_제품감지_무 : BOOL; (* AT %MW3501.6 *) (* S367_M_공정_제품감지_무 *)
    S367_M_작업_완료 : BOOL; (* AT %MW3501.0 *) (* S367_M_작업_완료 *)
    S368_HOME : BOOL; (* AT %MW4048.0 *) (* S368_HOME *)
    S368_M_HANGER_CLP_전진_LS_이상 : BOOL; (* AT %MW4111.5 *) (* S368_M_HANGER_CLP_전진_LS_이상 *)
    S368_M_HANGER_CLP_전진_보조 : BOOL; (* AT %MW4111.1 *) (* S368_M_HANGER_CLP_전진_보조 *)
    S368_M_HANGER_CLP_전진단 : BOOL; (* AT %MW4111.3 *) (* S368_M_HANGER_CLP_전진단 *)
    S368_M_HANGER_CLP_조건 : BOOL; (* AT %MW4111.0 *) (* S368_M_HANGER_CLP_조건 *)
    S368_M_HANGER_CLP_후진_LS_이상 : BOOL; (* AT %MW4111.6 *) (* S368_M_HANGER_CLP_후진_LS_이상 *)
    S368_M_HANGER_CLP_후진_보조 : BOOL; (* AT %MW4111.2 *) (* S368_M_HANGER_CLP_후진_보조 *)
    S368_M_HANGER_CLP_후진단 : BOOL; (* AT %MW4111.4 *) (* S368_M_HANGER_CLP_후진단 *)
    S368_M_HANGER_급전급기_ADV_AUX : BOOL; (* AT %MW4103.1 *)
    S368_M_HANGER_급전급기_COND : BOOL; (* AT %MW4103.0 *)
    S368_M_HANGER_급전급기_RET_AUX : BOOL; (* AT %MW4103.2 *)
    S368_M_HANGER_급전급기_전진_LS_이상 : BOOL; (* AT %MW4103.5 *)
    S368_M_HANGER_급전급기_전진단 : BOOL; (* AT %MW4103.3 *)
    S368_M_HANGER_급전급기_후진_LS_이상 : BOOL; (* AT %MW4103.6 *)
    S368_M_HANGER_급전급기_후진단 : BOOL; (* AT %MW4103.4 *)
    S368_M_LH_AX_CLAMP_전진_LS_이상 : BOOL; (* AT %MW4102.5 *) (* S368_M_LH_AX_CLAMP_전진_LS_이상 *)
    S368_M_LH_AX_CLAMP_전진_보조 : BOOL; (* AT %MW4102.1 *) (* S368_M_LH_AX_CLAMP_전진_보조 *)
    S368_M_LH_AX_CLAMP_전진단 : BOOL; (* AT %MW4102.3 *) (* S368_M_LH_AX_CLAMP_전진단 *)
    S368_M_LH_AX_CLAMP_조건 : BOOL; (* AT %MW4102.0 *) (* S368_M_LH_AX_CLAMP_조건 *)
    S368_M_LH_AX_CLAMP_후진_LS_이상 : BOOL; (* AT %MW4102.6 *) (* S368_M_LH_AX_CLAMP_후진_LS_이상 *)
    S368_M_LH_AX_CLAMP_후진_보조 : BOOL; (* AT %MW4102.2 *) (* S368_M_LH_AX_CLAMP_후진_보조 *)
    S368_M_LH_AX_CLAMP_후진단 : BOOL; (* AT %MW4102.4 *) (* S368_M_LH_AX_CLAMP_후진단 *)
    S368_M_LH_AX_LATCH_전진_LS_이상 : BOOL; (* AT %MW4100.5 *) (* S368_M_LH_AX_LATCH_전진_LS_이상 *)
    S368_M_LH_AX_LATCH_전진_보조 : BOOL; (* AT %MW4100.1 *) (* S368_M_LH_AX_LATCH_전진_보조 *)
    S368_M_LH_AX_LATCH_전진단 : BOOL; (* AT %MW4100.3 *) (* S368_M_LH_AX_LATCH_전진단 *)
    S368_M_LH_AX_LATCH_조건 : BOOL; (* AT %MW4100.0 *) (* S368_M_LH_AX_LATCH_조건 *)
    S368_M_LH_AX_LATCH_후진_LS_이상 : BOOL; (* AT %MW4100.6 *) (* S368_M_LH_AX_LATCH_후진_LS_이상 *)
    S368_M_LH_AX_LATCH_후진_보조 : BOOL; (* AT %MW4100.2 *) (* S368_M_LH_AX_LATCH_후진_보조 *)
    S368_M_LH_AX_LATCH_후진단 : BOOL; (* AT %MW4100.4 *) (* S368_M_LH_AX_LATCH_후진단 *)
    S368_M_LH_AX_SR_LAT_전진_LS_이상 : BOOL; (* AT %MW4101.5 *) (* S368_M_LH_AX_SR_LAT_전진_LS_이상 *)
    S368_M_LH_AX_SR_LAT_전진_보조 : BOOL; (* AT %MW4101.1 *) (* S368_M_LH_AX_SR_LAT_전진_보조 *)
    S368_M_LH_AX_SR_LAT_전진단 : BOOL; (* AT %MW4101.3 *) (* S368_M_LH_AX_SR_LAT_전진단 *)
    S368_M_LH_AX_SR_LAT_조건 : BOOL; (* AT %MW4101.0 *) (* S368_M_LH_AX_SR_LAT_조건 *)
    S368_M_LH_AX_SR_LAT_후진_LS_이상 : BOOL; (* AT %MW4101.6 *) (* S368_M_LH_AX_SR_LAT_후진_LS_이상 *)
    S368_M_LH_AX_SR_LAT_후진_보조 : BOOL; (* AT %MW4101.2 *) (* S368_M_LH_AX_SR_LAT_후진_보조 *)
    S368_M_LH_AX_SR_LAT_후진단 : BOOL; (* AT %MW4101.4 *) (* S368_M_LH_AX_SR_LAT_후진단 *)
    S368_M_R368_1_행거안착완료 : BOOL; (* AT %MW4001.2 *)
    S368_M_R369_1_안착완료 : BOOL; (* AT %MW4001.1 *)
    S368_M_RH_AX_CLAMP_전진_LS_이상 : BOOL; (* AT %MW4110.5 *) (* S368_M_RH_AX_CLAMP_전진_LS_이상 *)
    S368_M_RH_AX_CLAMP_전진_보조 : BOOL; (* AT %MW4110.1 *) (* S368_M_RH_AX_CLAMP_전진_보조 *)
    S368_M_RH_AX_CLAMP_전진단 : BOOL; (* AT %MW4110.3 *) (* S368_M_RH_AX_CLAMP_전진단 *)
    S368_M_RH_AX_CLAMP_조건 : BOOL; (* AT %MW4110.0 *) (* S368_M_RH_AX_CLAMP_조건 *)
    S368_M_RH_AX_CLAMP_후진_LS_이상 : BOOL; (* AT %MW4110.6 *) (* S368_M_RH_AX_CLAMP_후진_LS_이상 *)
    S368_M_RH_AX_CLAMP_후진_보조 : BOOL; (* AT %MW4110.2 *) (* S368_M_RH_AX_CLAMP_후진_보조 *)
    S368_M_RH_AX_CLAMP_후진단 : BOOL; (* AT %MW4110.4 *) (* S368_M_RH_AX_CLAMP_후진단 *)
    S368_M_RH_AX_LATCH_전진_LS_이상 : BOOL; (* AT %MW4108.5 *) (* S368_M_RH_AX_LATCH_전진_LS_이상 *)
    S368_M_RH_AX_LATCH_전진_보조 : BOOL; (* AT %MW4108.1 *) (* S368_M_RH_AX_LATCH_전진_보조 *)
    S368_M_RH_AX_LATCH_전진단 : BOOL; (* AT %MW4108.3 *) (* S368_M_RH_AX_LATCH_전진단 *)
    S368_M_RH_AX_LATCH_조건 : BOOL; (* AT %MW4108.0 *) (* S368_M_RH_AX_LATCH_조건 *)
    S368_M_RH_AX_LATCH_후진_LS_이상 : BOOL; (* AT %MW4108.6 *) (* S368_M_RH_AX_LATCH_후진_LS_이상 *)
    S368_M_RH_AX_LATCH_후진_보조 : BOOL; (* AT %MW4108.2 *) (* S368_M_RH_AX_LATCH_후진_보조 *)
    S368_M_RH_AX_LATCH_후진단 : BOOL; (* AT %MW4108.4 *) (* S368_M_RH_AX_LATCH_후진단 *)
    S368_M_RH_AX_SR_LAT_전진_LS_이상 : BOOL; (* AT %MW4109.5 *) (* S368_M_RH_AX_SR_LAT_전진_LS_이상 *)
    S368_M_RH_AX_SR_LAT_전진_보조 : BOOL; (* AT %MW4109.1 *) (* S368_M_RH_AX_SR_LAT_전진_보조 *)
    S368_M_RH_AX_SR_LAT_전진단 : BOOL; (* AT %MW4109.3 *) (* S368_M_RH_AX_SR_LAT_전진단 *)
    S368_M_RH_AX_SR_LAT_조건 : BOOL; (* AT %MW4109.0 *) (* S368_M_RH_AX_SR_LAT_조건 *)
    S368_M_RH_AX_SR_LAT_후진_LS_이상 : BOOL; (* AT %MW4109.6 *) (* S368_M_RH_AX_SR_LAT_후진_LS_이상 *)
    S368_M_RH_AX_SR_LAT_후진_보조 : BOOL; (* AT %MW4109.2 *) (* S368_M_RH_AX_SR_LAT_후진_보조 *)
    S368_M_RH_AX_SR_LAT_후진단 : BOOL; (* AT %MW4109.4 *) (* S368_M_RH_AX_SR_LAT_후진단 *)
    S368_M_공정_HANGER_감지_유 : BOOL; (* AT %MW4001.11 *)
    S368_M_공정_불간섭 : BOOL; (* AT %MW4004.1 *) (* S368_M_공정_불간섭 *)
    S368_M_공정_제품감지_무 : BOOL; (* AT %MW4001.6 *) (* S368_M_공정_제품감지_무 *)
    S368_M_공정_제품감지_유 : BOOL; (* AT %MW4001.5 *) (* S368_M_공정_제품감지_유 *)
    S368_M_공정_차종_무 : BOOL; (* AT %MW4002.1 *) (* S368_M_공정_차종_무 *)
    S368_M_공정_차종_유 : BOOL; (* AT %MW4002.0 *) (* S368_M_공정_차종_유 *)
    S368_M_동작_선택_1 : BOOL; (* AT %MW4040.0 *) (* S368_M_동작_선택_1 *)
    S368_M_동작_선택_10 : BOOL; (* AT %MW4040.9 *) (* S368_M_동작_선택_10 *)
    S368_M_동작_선택_11 : BOOL; (* AT %MW4040.10 *) (* S368_M_동작_선택_11 *)
    S368_M_동작_선택_12 : BOOL; (* AT %MW4040.11 *) (* S368_M_동작_선택_12 *)
    S368_M_동작_선택_2 : BOOL; (* AT %MW4040.1 *) (* S368_M_동작_선택_2 *)
    S368_M_동작_선택_3 : BOOL; (* AT %MW4040.2 *) (* S368_M_동작_선택_3 *)
    S368_M_동작_선택_4 : BOOL; (* AT %MW4040.3 *) (* S368_M_동작_선택_4 *)
    S368_M_동작_선택_9 : BOOL; (* AT %MW4040.8 *) (* S368_M_동작_선택_9 *)
    S368_M_수동모드 : BOOL; (* AT %MW4000.3 *) (* S368 선택 수동모드 *)
    S368_M_운전준비_ON : BOOL; (* AT %MW4000.0 *) (* S368 운전준비 ON *)
    S368_M_자동_운전중 : BOOL; (* AT %MW4000.4 *) (* S368 자동운전중 *)
    S368_M_작업_완료 : BOOL; (* AT %MW4001.0 *) (* S368_M_작업_완료 *)
    S368_M_차종1_AX : BOOL; (* AT %MW10201.0 *) (* S368 M 차종1 AX *)
    S368_전진_ON : BOOL; (* AT %MW4048.1 *) (* S368_전진_ON *)
    S368_후진_ON : BOOL; (* AT %MW4048.2 *) (* S368_후진_ON *)
    전체_M_이상_리셋 : BOOL; (* AT %MW308.2 *) (* ALL공정 PB 이상리셋 *)
END_VAR
VAR_EXTERNAL
    EGIS_CWS : BOOL;
    S368L_RS_HANGER_급기_전진단 : BOOL; (* AT %MW86311.13 *)
    S368L_RS_HANGER_급기_후진단 : BOOL; (* AT %MW86311.14 *)
    S368L_RS_HANGER_급전_전진단 : BOOL; (* AT %MW86311.11 *)
    S368L_RS_HANGER_급전_후진단 : BOOL; (* AT %MW86311.12 *)
    S368L_SOL_HANGER_급전급기_전진 : BOOL; (* AT %MW96313.8 *)
    S368L_SOL_HANGER_급전급기_후진 : BOOL; (* AT %MW96313.9 *)
    S368_M_HANGER_CLP_전진_LAMP : WORD; (* AT %MW13622 *) (* S368_M_HANGER_CLP_전진_LAMP *)
    S368_M_HANGER_CLP_후진_LAMP : WORD; (* AT %MW13623 *) (* S368_M_HANGER_CLP_후진_LAMP *)
    S368_M_HANGER_급전급기_ADV_LAMP : WORD; (* AT %MW13606 *) (* S368_M_LH_HANG_CLP_전진_LAMP *)
    S368_M_HANGER_급전급기_RET_LAMP : WORD; (* AT %MW13607 *) (* S368_M_LH_HANG_CLP_후진_LAMP *)
    S368_M_LH_AX_CLAMP_전진_LAMP : WORD; (* AT %MW13604 *) (* S368_M_LH_AX_CLAMP_전진_LAMP *)
    S368_M_LH_AX_CLAMP_후진_LAMP : WORD; (* AT %MW13605 *) (* S368_M_LH_AX_CLAMP_후진_LAMP *)
    S368_M_LH_AX_LATCH_전진_LAMP : WORD; (* AT %MW13600 *) (* S368_M_LH_AX_LATCH_전진_LAMP *)
    S368_M_LH_AX_LATCH_후진_LAMP : WORD; (* AT %MW13601 *) (* S368_M_LH_AX_LATCH_후진_LAMP *)
    S368_M_LH_AX_SR_LAT_전진_LAMP : WORD; (* AT %MW13602 *) (* S368_M_LH_AX_SR_LAT_전진_LAMP *)
    S368_M_LH_AX_SR_LAT_후진_LAMP : WORD; (* AT %MW13603 *) (* S368_M_LH_AX_SR_LAT_후진_LAMP *)
    S368_M_RH_AX_CLAMP_전진_LAMP : WORD; (* AT %MW13620 *) (* S368_M_RH_AX_CLAMP_전진_LAMP *)
    S368_M_RH_AX_CLAMP_후진_LAMP : WORD; (* AT %MW13621 *) (* S368_M_RH_AX_CLAMP_후진_LAMP *)
    S368_M_RH_AX_LATCH_전진_LAMP : WORD; (* AT %MW13616 *) (* S368_M_RH_AX_LATCH_전진_LAMP *)
    S368_M_RH_AX_LATCH_후진_LAMP : WORD; (* AT %MW13617 *) (* S368_M_RH_AX_LATCH_후진_LAMP *)
    S368_M_RH_AX_SR_LAT_전진_LAMP : WORD; (* AT %MW13618 *) (* S368_M_RH_AX_SR_LAT_전진_LAMP *)
    S368_M_RH_AX_SR_LAT_후진_LAMP : WORD; (* AT %MW13619 *) (* S368_M_RH_AX_SR_LAT_후진_LAMP *)
    S368_RS_AX_HANGER_CLP_전진 : BOOL; (* AT %MW86301.8 *) (* S368_RS_AX_HANGER_CLP_전진 *)
    S368_RS_AX_HANGER_CLP_후진1 : BOOL; (* AT %MW86301.9 *) (* S368_RS_AX_HANGER_CLP_후진1 *)
    S368_RS_AX_HANGER_CLP_후진2 : BOOL; (* AT %MW86301.10 *) (* S368_RS_AX_HANGER_CLP_후진2 *)
    S368_RS_AX_LH_CLAMP_전진 : BOOL; (* AT %MW86310.8 *) (* S368_RS_AX_LH_CLAMP_전진 *)
    S368_RS_AX_LH_CLAMP_후진1 : BOOL; (* AT %MW86310.9 *) (* S368_RS_AX_LH_CLAMP_후진1 *)
    S368_RS_AX_LH_CLAMP_후진2 : BOOL; (* AT %MW86310.10 *) (* S368_RS_AX_LH_CLAMP_후진2 *)
    S368_RS_AX_LH_CLAMP_후진3 : BOOL; (* AT %MW86310.11 *) (* S368_RS_AX_LH_CLAMP_후진3 *)
    S368_RS_AX_LH_CLAMP_후진4 : BOOL; (* AT %MW86310.12 *) (* S368_RS_AX_LH_CLAMP_후진4 *)
    S368_RS_AX_LH_CLAMP_후진5 : BOOL; (* AT %MW86310.13 *) (* S368_RS_AX_LH_CLAMP_후진5 *)
    S368_RS_AX_LH_GR_LATCH_전진 : BOOL; (* AT %MW86310.0 *) (* S368_RS_AX_LH_GR_LATCH_전진 *)
    S368_RS_AX_LH_GR_LATCH_후진1 : BOOL; (* AT %MW86310.1 *) (* S368_RS_AX_LH_GR_LATCH_후진1 *)
    S368_RS_AX_LH_GR_LATCH_후진2 : BOOL; (* AT %MW86310.2 *) (* S368_RS_AX_LH_GR_LATCH_후진2 *)
    S368_RS_AX_LH_GR_LATCH_후진3 : BOOL; (* AT %MW86310.3 *) (* S368_RS_AX_LH_GR_LATCH_후진3 *)
    S368_RS_AX_LH_GR_LATCH_후진4 : BOOL; (* AT %MW86310.4 *) (* S368_RS_AX_LH_GR_LATCH_후진4 *)
    S368_RS_AX_LH_GR_LATCH_후진5 : BOOL; (* AT %MW86310.5 *) (* S368_RS_AX_LH_GR_LATCH_후진5 *)
    S368_RS_AX_LH_HANG_CLP_후진1 : BOOL; (* AT %MW86311.8 *) (* S368_RS_AX_LH_HANG_CLP_후진1 *)
    S368_RS_AX_LH_HANG_CLP_후진2 : BOOL; (* AT %MW86311.9 *) (* S368_RS_AX_LH_HANG_CLP_후진2 *)
    S368_RS_AX_LH_SR_LATCH_전진 : BOOL; (* AT %MW86311.0 *) (* S368_RS_AX_LH_SR_LATCH_전진 *)
    S368_RS_AX_LH_SR_LATCH_후진1 : BOOL; (* AT %MW86311.1 *) (* S368_RS_AX_LH_SR_LATCH_후진1 *)
    S368_RS_AX_LH_SR_LATCH_후진2 : BOOL; (* AT %MW86311.2 *) (* S368_RS_AX_LH_SR_LATCH_후진2 *)
    S368_RS_AX_LH_SR_LATCH_후진3 : BOOL; (* AT %MW86311.3 *) (* S368_RS_AX_LH_SR_LATCH_후진3 *)
    S368_RS_AX_LH_SR_LATCH_후진4 : BOOL; (* AT %MW86311.4 *) (* S368_RS_AX_LH_SR_LATCH_후진4 *)
    S368_RS_AX_RH_CLAMP_전진 : BOOL; (* AT %MW86300.8 *) (* S368_RS_AX_RH_CLAMP_전진 *)
    S368_RS_AX_RH_CLAMP_후진1 : BOOL; (* AT %MW86300.9 *) (* S368_RS_AX_RH_CLAMP_후진1 *)
    S368_RS_AX_RH_CLAMP_후진2 : BOOL; (* AT %MW86300.10 *) (* S368_RS_AX_RH_CLAMP_후진2 *)
    S368_RS_AX_RH_CLAMP_후진3 : BOOL; (* AT %MW86300.11 *) (* S368_RS_AX_RH_CLAMP_후진3 *)
    S368_RS_AX_RH_CLAMP_후진4 : BOOL; (* AT %MW86300.12 *) (* S368_RS_AX_RH_CLAMP_후진4 *)
    S368_RS_AX_RH_CLAMP_후진5 : BOOL; (* AT %MW86300.13 *) (* S368_RS_AX_RH_CLAMP_후진5 *)
    S368_RS_AX_RH_GR_LATCH_전진 : BOOL; (* AT %MW86300.0 *) (* S368_RS_AX_RH_GR_LATCH_전진 *)
    S368_RS_AX_RH_GR_LATCH_후진1 : BOOL; (* AT %MW86300.1 *) (* S368_RS_AX_RH_GR_LATCH_후진1 *)
    S368_RS_AX_RH_GR_LATCH_후진2 : BOOL; (* AT %MW86300.2 *) (* S368_RS_AX_RH_GR_LATCH_후진2 *)
    S368_RS_AX_RH_GR_LATCH_후진3 : BOOL; (* AT %MW86300.3 *) (* S368_RS_AX_RH_GR_LATCH_후진3 *)
    S368_RS_AX_RH_GR_LATCH_후진4 : BOOL; (* AT %MW86300.4 *) (* S368_RS_AX_RH_GR_LATCH_후진4 *)
    S368_RS_AX_RH_GR_LATCH_후진5 : BOOL; (* AT %MW86300.5 *) (* S368_RS_AX_RH_GR_LATCH_후진5 *)
    S368_RS_AX_RH_SR_LATCH_전진 : BOOL; (* AT %MW86301.0 *) (* S368_RS_AX_RH_SR_LATCH_전진 *)
    S368_RS_AX_RH_SR_LATCH_후진1 : BOOL; (* AT %MW86301.1 *) (* S368_RS_AX_RH_SR_LATCH_후진1 *)
    S368_RS_AX_RH_SR_LATCH_후진2 : BOOL; (* AT %MW86301.2 *) (* S368_RS_AX_RH_SR_LATCH_후진2 *)
    S368_RS_AX_RH_SR_LATCH_후진3 : BOOL; (* AT %MW86301.3 *) (* S368_RS_AX_RH_SR_LATCH_후진3 *)
    S368_RS_AX_RH_SR_LATCH_후진4 : BOOL; (* AT %MW86301.4 *) (* S368_RS_AX_RH_SR_LATCH_후진4 *)
    S368_SOL_AX_HANG_CLP_전진 : BOOL; (* AT %MW96303.12 *) (* S368_SOL_AX_HANG_CLP_전진 *)
    S368_SOL_AX_HANG_CLP_후진 : BOOL; (* AT %MW96303.13 *) (* S368_SOL_AX_HANG_CLP_후진 *)
    S368_SOL_AX_LH_CLAMP_전진 : BOOL; (* AT %MW96303.6 *) (* S368_SOL_AX_LH_CLAMP_전진 *)
    S368_SOL_AX_LH_CLAMP_후진 : BOOL; (* AT %MW96303.7 *) (* S368_SOL_AX_LH_CLAMP_후진 *)
    S368_SOL_AX_LH_GR_LATCH_전진 : BOOL; (* AT %MW96303.2 *) (* S368_SOL_AX_LH_GR_LATCH_전진 *)
    S368_SOL_AX_LH_GR_LATCH_후진 : BOOL; (* AT %MW96303.3 *) (* S368_SOL_AX_LH_GR_LATCH_후진 *)
    S368_SOL_AX_LH_SR_LATCH_전진 : BOOL; (* AT %MW96303.10 *) (* S368_SOL_AX_LH_SR_LATCH_전진 *)
    S368_SOL_AX_LH_SR_LATCH_후진 : BOOL; (* AT %MW96303.11 *) (* S368_SOL_AX_LH_SR_LATCH_후진 *)
    S368_SOL_AX_RH_CLAMP_전진 : BOOL; (* AT %MW96303.4 *) (* S368_SOL_AX_RH_CLAMP_전진 *)
    S368_SOL_AX_RH_CLAMP_후진 : BOOL; (* AT %MW96303.5 *) (* S368_SOL_AX_RH_CLAMP_후진 *)
    S368_SOL_AX_RH_GR_LATCH_전진 : BOOL; (* AT %MW96303.0 *) (* S368_SOL_AX_RH_GR_LATCH_전진 *)
    S368_SOL_AX_RH_GR_LATCH_후진 : BOOL; (* AT %MW96303.1 *) (* S368_SOL_AX_RH_GR_LATCH_후진 *)
    S368_SOL_AX_RH_SR_LATCH_전진 : BOOL; (* AT %MW96303.8 *) (* S368_SOL_AX_RH_SR_LATCH_전진 *)
    S368_SOL_AX_RH_SR_LATCH_후진 : BOOL; (* AT %MW96303.9 *) (* S368_SOL_AX_RH_SR_LATCH_후진 *)
END_VAR
VAR
    INST : ACT_6_CYL;
    S367_RH_AX_LATCH : ACT_6_CYL;
    S368_AX_HANG_CLAMP : ACT_6_CYL;
    S368_LH_AX_CLAMP : ACT_6_CYL;
    S368_LH_AX_LATCH : ACT_6_CYL;
    S368_LH_AX_SR_LAT : ACT_6_CYL;
    S368_RH_AX_CLAMP : ACT_6_CYL;
    S368_RH_AX_SR_LAT : ACT_6_CYL;
    S368_작업_완료 : BOOL;
    S369_AX_HANG_CLAMP : ACT_6_CYL;
END_VAR

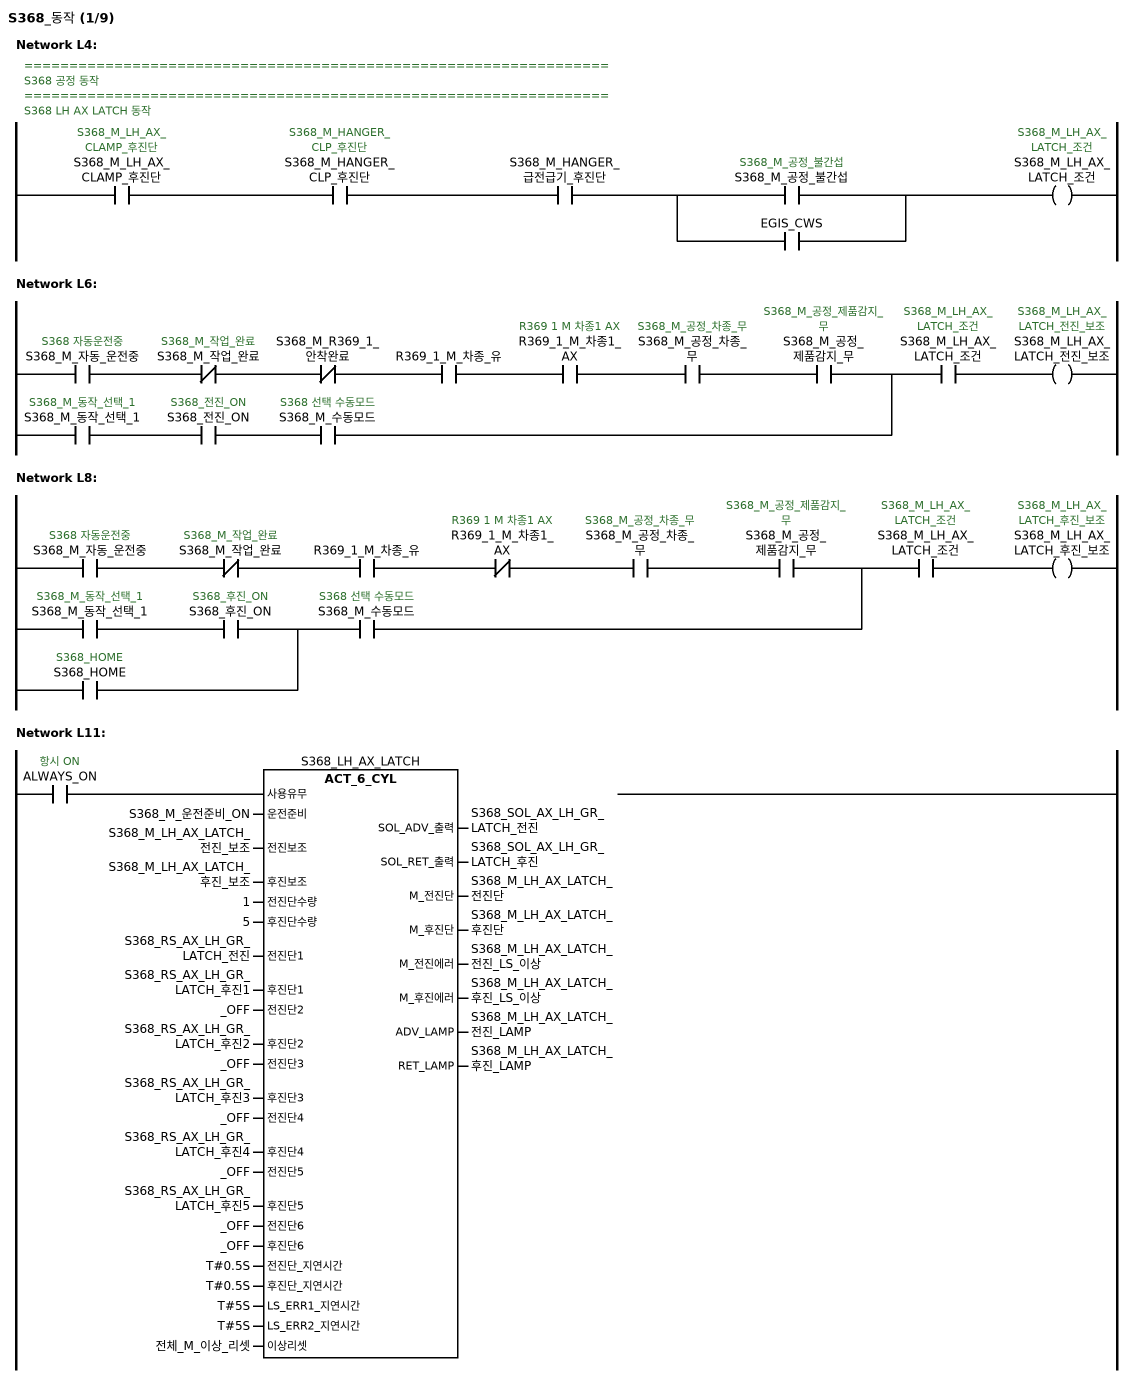
(* ================================================================= *)
(* S368 공정 동작 *)
(* ================================================================= *)
(* S368 LH AX LATCH 동작 *)
(* Rung L4 *)
S368_M_LH_AX_LATCH_조건 := S368_M_LH_AX_CLAMP_후진단 AND S368_M_HANGER_CLP_후진단 AND S368_M_HANGER_급전급기_후진단 AND (S368_M_공정_불간섭 OR EGIS_CWS);
(* Rung L6 *)
S368_M_LH_AX_LATCH_전진_보조 := ((S368_M_자동_운전중 AND NOT S368_M_작업_완료 AND NOT S368_M_R369_1_안착완료 AND R369_1_M_차종_유 AND R369_1_M_차종1_AX AND S368_M_공정_차종_무 AND S368_M_공정_제품감지_무) OR (S368_M_동작_선택_1 AND S368_전진_ON AND S368_M_수동모드)) AND S368_M_LH_AX_LATCH_조건;
(* Rung L8 *)
S368_M_LH_AX_LATCH_후진_보조 := ((S368_M_자동_운전중 AND NOT S368_M_작업_완료 AND R369_1_M_차종_유 AND NOT R369_1_M_차종1_AX AND S368_M_공정_차종_무 AND S368_M_공정_제품감지_무) OR (((S368_M_동작_선택_1 AND S368_후진_ON) OR S368_HOME) AND S368_M_수동모드)) AND S368_M_LH_AX_LATCH_조건;
(* Rung L11 *)
S368_LH_AX_LATCH(사용유무 := ALWAYS_ON, 운전준비 := S368_M_운전준비_ON, 전진보조 := S368_M_LH_AX_LATCH_전진_보조, 후진보조 := S368_M_LH_AX_LATCH_후진_보조, 전진단수량 := 1, 후진단수량 := 5, 전진단1 := S368_RS_AX_LH_GR_LATCH_전진, 후진단1 := S368_RS_AX_LH_GR_LATCH_후진1, 전진단2 := _OFF, 후진단2 := S368_RS_AX_LH_GR_LATCH_후진2, 전진단3 := _OFF, 후진단3 := S368_RS_AX_LH_GR_LATCH_후진3, 전진단4 := _OFF, 후진단4 := S368_RS_AX_LH_GR_LATCH_후진4, 전진단5 := _OFF, 후진단5 := S368_RS_AX_LH_GR_LATCH_후진5, 전진단6 := _OFF, 후진단6 := _OFF, 전진단_지연시간 := T#0.5S, 후진단_지연시간 := T#0.5S, LS_ERR1_지연시간 := T#5S, LS_ERR2_지연시간 := T#5S, 이상리셋 := 전체_M_이상_리셋, SOL_ADV_출력 => S368_SOL_AX_LH_GR_LATCH_전진, SOL_RET_출력 => S368_SOL_AX_LH_GR_LATCH_후진, M_전진단 => S368_M_LH_AX_LATCH_전진단, M_후진단 => S368_M_LH_AX_LATCH_후진단, M_전진에러 => S368_M_LH_AX_LATCH_전진_LS_이상, M_후진에러 => S368_M_LH_AX_LATCH_후진_LS_이상, ADV_LAMP => S368_M_LH_AX_LATCH_전진_LAMP, RET_LAMP => S368_M_LH_AX_LATCH_후진_LAMP);

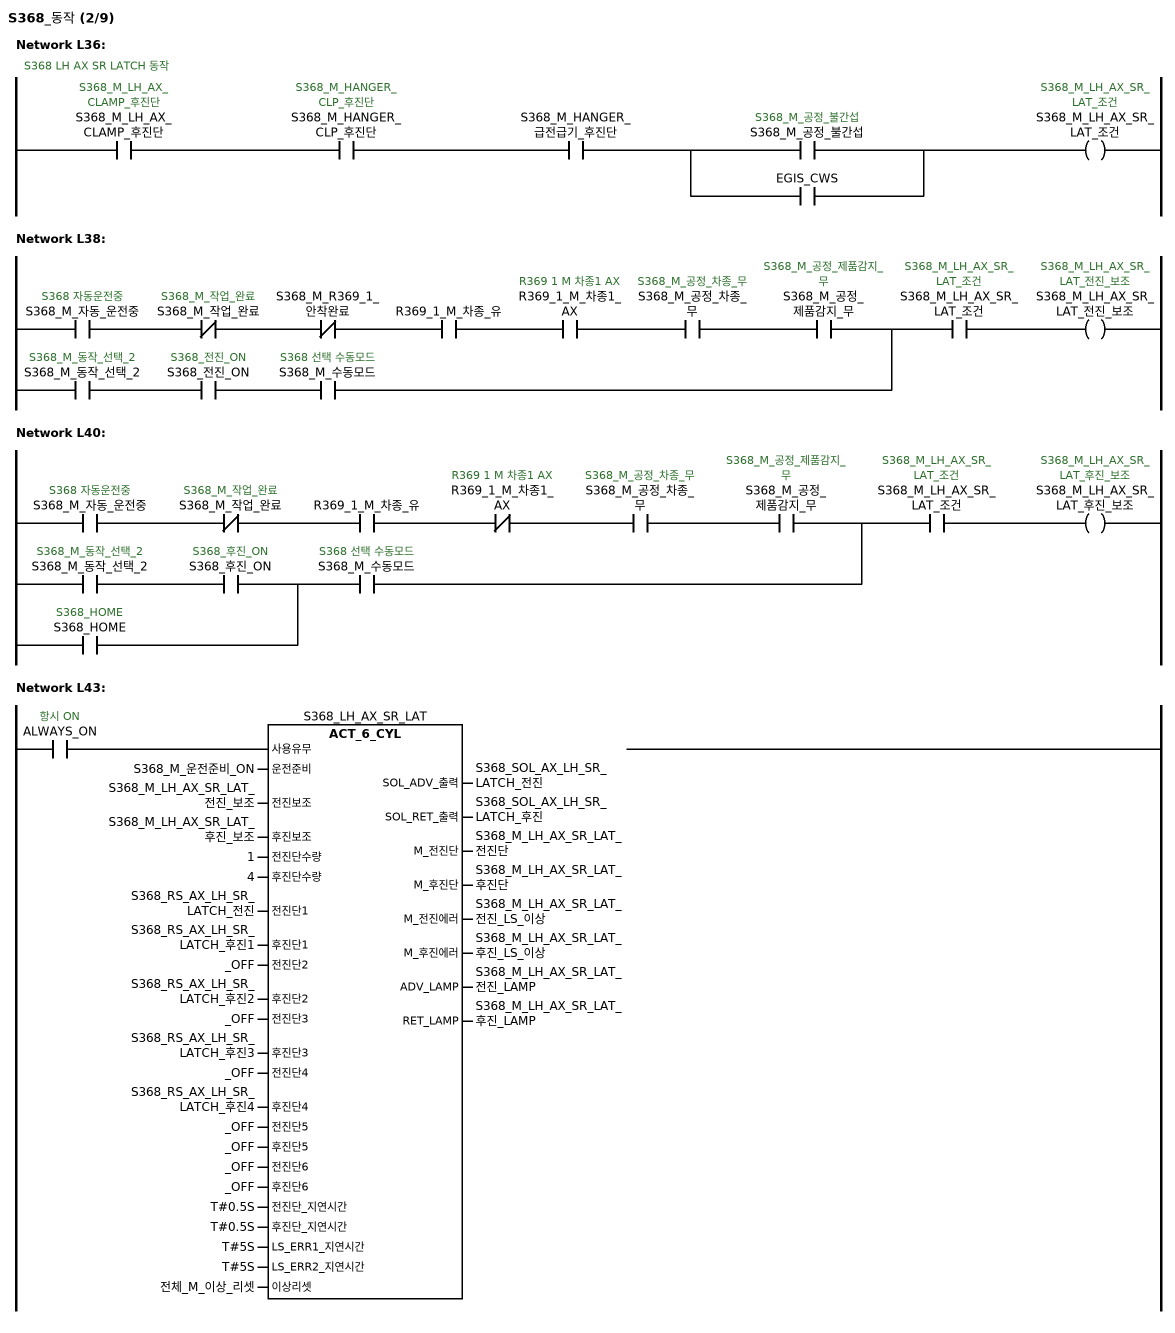
(* S368 LH AX SR LATCH 동작 *)
(* Rung L36 *)
S368_M_LH_AX_SR_LAT_조건 := S368_M_LH_AX_CLAMP_후진단 AND S368_M_HANGER_CLP_후진단 AND S368_M_HANGER_급전급기_후진단 AND (S368_M_공정_불간섭 OR EGIS_CWS);
(* Rung L38 *)
S368_M_LH_AX_SR_LAT_전진_보조 := ((S368_M_자동_운전중 AND NOT S368_M_작업_완료 AND NOT S368_M_R369_1_안착완료 AND R369_1_M_차종_유 AND R369_1_M_차종1_AX AND S368_M_공정_차종_무 AND S368_M_공정_제품감지_무) OR (S368_M_동작_선택_2 AND S368_전진_ON AND S368_M_수동모드)) AND S368_M_LH_AX_SR_LAT_조건;
(* Rung L40 *)
S368_M_LH_AX_SR_LAT_후진_보조 := ((S368_M_자동_운전중 AND NOT S368_M_작업_완료 AND R369_1_M_차종_유 AND NOT R369_1_M_차종1_AX AND S368_M_공정_차종_무 AND S368_M_공정_제품감지_무) OR (((S368_M_동작_선택_2 AND S368_후진_ON) OR S368_HOME) AND S368_M_수동모드)) AND S368_M_LH_AX_SR_LAT_조건;
(* Rung L43 *)
S368_LH_AX_SR_LAT(사용유무 := ALWAYS_ON, 운전준비 := S368_M_운전준비_ON, 전진보조 := S368_M_LH_AX_SR_LAT_전진_보조, 후진보조 := S368_M_LH_AX_SR_LAT_후진_보조, 전진단수량 := 1, 후진단수량 := 4, 전진단1 := S368_RS_AX_LH_SR_LATCH_전진, 후진단1 := S368_RS_AX_LH_SR_LATCH_후진1, 전진단2 := _OFF, 후진단2 := S368_RS_AX_LH_SR_LATCH_후진2, 전진단3 := _OFF, 후진단3 := S368_RS_AX_LH_SR_LATCH_후진3, 전진단4 := _OFF, 후진단4 := S368_RS_AX_LH_SR_LATCH_후진4, 전진단5 := _OFF, 후진단5 := _OFF, 전진단6 := _OFF, 후진단6 := _OFF, 전진단_지연시간 := T#0.5S, 후진단_지연시간 := T#0.5S, LS_ERR1_지연시간 := T#5S, LS_ERR2_지연시간 := T#5S, 이상리셋 := 전체_M_이상_리셋, SOL_ADV_출력 => S368_SOL_AX_LH_SR_LATCH_전진, SOL_RET_출력 => S368_SOL_AX_LH_SR_LATCH_후진, M_전진단 => S368_M_LH_AX_SR_LAT_전진단, M_후진단 => S368_M_LH_AX_SR_LAT_후진단, M_전진에러 => S368_M_LH_AX_SR_LAT_전진_LS_이상, M_후진에러 => S368_M_LH_AX_SR_LAT_후진_LS_이상, ADV_LAMP => S368_M_LH_AX_SR_LAT_전진_LAMP, RET_LAMP => S368_M_LH_AX_SR_LAT_후진_LAMP);

